(* CODESYS project AnimalCT.project
   Title: AnimalCT
   CompiledLibraryCompatibilityVersion: LeadSysStudio V3.5 SP15 Patch 4

Project tree, tasks and I/O mapping:
  Device : MC508, Leadshine Technology Co., Ltd., order no. 508101, version 3.5.15.40
      settings: RetainMode = 0; RetainStartAddr = 20480; RetainEndAddr = 524288; RetainSize = 524288
    application Application
      libraries: Standard, * (System); CAA CiA 405, 3.5.15.0 (CAA Technical Workgroup); CAA SerialCom, 3.5.15.0 (CAA Technical Workgroup); Serial Communication, 3.5.7.0 (3S - Smart Software Solutions GmbH); LS_SysLib, 1.0.0.9 (Leadshine Technology Co.Ltd); CANopenLib, 1.0.0.5 (Leadshine Technology Co.Ltd); CAA Net Base Services, 3.5.15.0 (CAA Technical Workgroup); Network, 3.5.7.0 (3S - Smart Software Solutions GmbH); CANbus, 3.5.7.0 (3S - Smart Software Solutions GmbH); VisuDialogs, * (System); LS_OmronUtils, 1.0.0.2 (Leadshine Technology Co.Ltd); CAN Low Level Communication, 1.0.0.0 (Leadshine Technology Co.Ltd); CAN API, 1.0.0.0 (Leadshine Technology Co.Ltd); CANopenLib, 1.0.0.5 (Leadshine Technology Co.Ltd)
      task Task_Trigger (cyclic, interval 2 ms, priority 1) calls Trigger_HaoboPannel, Entity_IO
      task MainTask (cyclic, interval 5 ms, priority 1) calls PLC_PRG
      task CanOpen (cyclic, interval 2 ms, priority 1) calls Axis_QJ, Axis_XZ
      DTU/
        Axis/
          data type AxisState
          data type AxisCmd
          data type AxisParameter
        TCP/
          data type PLC_SEND
          data type PLC_RECV
          data type Real_TO_Byte_Convert
        data type E_LampCmd
      GVL/
        global variables GVL_SCAN
        global variables GVL_State
      BasicFBs/
        function block Blink [ST]
        function block ASCII_Chart_N [ST]
        function block RC [ST]
        function block Curve_Cs [ST]
        function block ASCII_Chart_P [ST]
        function block MeanValue [ST]
        function block Cut [ST]
        function block String2Byte [ST]
      Refer/
        program POU_CANopen [ST]: A01_MC_AxisConfi, A04_MC_MoveRelative, A02_MC_Power, A09_ODPara, A03_MC_MoveAbsolute, A06_MC_Home, A10_MC_JOG, A11_MC_ReadStatus_CAN, A08_MC_Reset, A07_MC_Stop, A05_MC_MoveVelocity
      trace Trace (task MainTask): Entity_IO.bTriggerOut, Entity_IO.bTriggerHaobo, Entity_IO.bXaryOne, WorkStation_TCP.PLC_RECV1.m_nSocketType
      global variables PersistentVars
      Init/
        program InitMotor [ST]
      visualisation Motor
      program PLC_PRG [SFC]: _a_SelfCheck_active, _a_MoveXZ_entry, _a_QuickScan_exit, T_JUMP_IDLE, _a_ScoutDR_active, _a_Idle_exit, T_DR, _AutoDR_exit, _a_Idle_entry, _a_SelfCheck_exit, _a_Error_entry, T_QuickScan, _AutoDR_active, _a_QuickScan_entry, _a_Error_active, T_AutoDR, _a_CBCTScan_exit, _a_CBCTScan_active, _a_Homing_active, T_MoveXZ, _a_SelfCheck_entry, _a_MoveXZ_exit, T_CBCT, _a_Emergercy_entry, _AutoDR_entry_0, _a_ScoutScan_entry, _a_ScoutScan_exit, _a_ShutDown_entry, _a_Idle_active, _a_Error_exit, _a_ShutDown_active, _a_Homing_entry, _a_CBCTScan_entry, _a_QuickScan_active, _a_Debug_entry, _a_Init_active, _a_ScoutScan_active, _a_Logic_active, _a_MoveXZ_active, _a_SystemInfo_active, _a_Debug_active, _a_ScoutDR_exit, _a_Homing_exit, _a_ScoutDR_entry, T_Scout, _a_Emergercy_active
      Logic/
        program Trigger_HaoboPannel [ST]
        program WorkMode [ST]
        program Trigger_YrayPannel [ST]
      Motor/
        program Axis_XZ [ST]
        program Axis_QJ [ST]
        program Motor_SJ [ST]
      visualisation Entity_IO
      Communication/
        program CTBOX_RS232 [ST]
        program WorkStation_TCP [ST]: APLC_RECV, APLC_SENG
        program XRAY_RS485 [ST]: AXray
      IOs/
        program Entity_IO [ST]
    Resource Usage
    Device Diagnose
    Network Configuration
      LocalBus Config
    CANbus : CANbus, 3S - Smart Software Solutions GmbH, order no. 
      , version 3.5.15.0
        settings: Baudrate = 1000 kbit/s
      CANopen_Manager : CANopen_Manager, 3S - Smart Software Solutions GmbH, version 3.5.15.0
          settings: Manager is Sync consumer = True; ConfigVersion = 50659584
        ASDA_A3_Drive_QJ : ASDA-A3 Drive, Delta Electronics,INC., order no. 0, version Revision=16#02000001, FileVersion=1.1
            settings: NODEIDSAVED = 2; SDO Timeout = 1000000; PDO_Autoconfig = FALSE; EXPERTSETTINGS = False; Sync-General Parameters.Sync-COBID = 16#00000080; Emergency-General Parameters.Emergency COBID = 16#00000082; PDO 16#1400.COBID = 16#00000202; Process by CANopenManager = TRUE; PDO 16#1401.COBID = 16#00000302; Process by CANopenManager = TRUE; PDO 16#1402.COBID = 16#00000402; Process by CANopenManager = TRUE; PDO 16#1403.COBID = 16#00000502; Process by CANopenManager = TRUE; PDO 16#1800.COBID = 16#00000182; PDO 16#1800.Inhibit Time = 20; Process by CANopenManager = TRUE; PDO 16#1801.COBID = 16#00000282; PDO 16#1801.Inhibit Time = 20; Process by CANopenManager = TRUE; PDO 16#1802.COBID = 16#00000382; PDO 16#1802.Inhibit Time = 100; Process by CANopenManager = TRUE; PDO 16#1803.COBID = 16#00000482; PDO 16#1803.Inhibit Time = 100; Process by CANopenManager = TRUE; Heartbeat-Consuming1.Heartbeat-Time = 300 ms; Controlword.Index = 16#6040; Controlword.Subindex = 16#00; Controlword.ObjectLength = 16; Target Position.Index = 16#607A; Target Position.Subindex = 16#00; Target Position.ObjectLength = 32; Modes of operation.Index = 16#6060; Modes of operation.Subindex = 16#00; Modes of operation.ObjectLength = 8; Profile velocity.Index = 16#6081; Profile velocity.Subindex = 16#00; Profile velocity.ObjectLength = 32; Profile acceleration.Index = 16#6083;
              Profile acceleration.Subindex = 16#00; Profile acceleration.ObjectLength = 32; Target velocity.Index = 16#60FF; Target velocity.Subindex = 16#00; Target velocity.ObjectLength = 32; Profile deceleration.Index = 16#6084; Profile deceleration.Subindex = 16#00; Profile deceleration.ObjectLength = 32; Statusword.Index = 16#6041; Statusword.Subindex = 16#00; Statusword.ObjectLength = 16; Modes of operation display.Index = 16#6061; Modes of operation display.Subindex = 16#00; Modes of operation display.ObjectLength = 8; Position actual value.Index = 16#6064; Position actual value.Subindex = 16#00; Position actual value.ObjectLength = 32; Velocity actual value.Index = 16#606C; Velocity actual value.Subindex = 16#00; Velocity actual value.ObjectLength = 32; Digital inputs.Index = 16#60FD; Digital inputs.Subindex = 16#00; Digital inputs.ObjectLength = 32; SDO List.Set communication cycle period.Index = 16#1006; SDO List.Set communication cycle period.Subindex = 16#00; SDO List.Set communication cycle period.Value = 16#000003E8; SDO List.Set communication cycle period.Size = 32; SDO List.Set communication cycle period.AbortIfError = FALSE; SDO List.Set communication cycle period.JumpToLine = FALSE; SDO List.Set communication cycle period.Line = 0; SDO List.Set Guardtime.Index = 16#100C; SDO List.Set Guardtime.Subindex = 16#00; SDO List.Set Guardtime.Value = 16#00000000; SDO List.Set Guardtime.Size = 16; SDO List.Set Guardtime.AbortIfError = FALSE; SDO List.Set Guardtime.JumpToLine = FALSE; SDO List.Set Guardtime.Line = 0; SDO List.Set Lifetime.Index = 16#100D; SDO List.Set Lifetime.Subindex = 16#00; SDO List.Set Lifetime.Value = 16#00000000;
              SDO List.Set Lifetime.Size = 8; SDO List.Set Lifetime.AbortIfError = FALSE; SDO List.Set Lifetime.JumpToLine = FALSE; SDO List.Set Lifetime.Line = 0; SDO List.Set Heartbeat Consumer.Index = 16#1016; SDO List.Set Heartbeat Consumer.Subindex = 16#01; SDO List.Set Heartbeat Consumer.Value = 16#007F012C; SDO List.Set Heartbeat Consumer.Size = 32; SDO List.Set Heartbeat Consumer.AbortIfError = FALSE; SDO List.Set Heartbeat Consumer.JumpToLine = FALSE; SDO List.Set Heartbeat Consumer.Line = 0; SDO List.Set Heartbeat Producer.Index = 16#1017; SDO List.Set Heartbeat Producer.Subindex = 16#00; SDO List.Set Heartbeat Producer.Value = 16#000000C8; SDO List.Set Heartbeat Producer.Size = 16; SDO List.Set Heartbeat Producer.AbortIfError = FALSE; SDO List.Set Heartbeat Producer.JumpToLine = FALSE; SDO List.Set Heartbeat Producer.Line = 0; SDO List.Disable PDO.Index = 16#1400; SDO List.Disable PDO.Subindex = 16#01; SDO List.Disable PDO.Value = 16#80000202; SDO List.Disable PDO.Size = 32; SDO List.Disable PDO.AbortIfError = FALSE; SDO List.Disable PDO.JumpToLine = FALSE; SDO List.Disable PDO.Line = 0; SDO List.Set transmission type.Index = 16#1400; SDO List.Set transmission type.Subindex = 16#02; SDO List.Set transmission type.Value = 16#FF; SDO List.Set transmission type.Size = 8; SDO List.Set transmission type.AbortIfError = FALSE; SDO List.Set transmission type.JumpToLine = FALSE; SDO List.Set transmission type.Line = 0; SDO List.Clear pdo mapping.Index = 16#1600; SDO List.Clear pdo mapping.Subindex = 16#00; SDO List.Clear pdo mapping.Value = 16#0; SDO List.Clear pdo mapping.Size = 8; SDO List.Clear pdo mapping.AbortIfError = FALSE; SDO List.Clear pdo mapping.JumpToLine = FALSE; SDO List.Clear pdo mapping.Line = 0; SDO List.Set Mapping.Index = 16#1600;
              SDO List.Set Mapping.Subindex = 16#01; SDO List.Set Mapping.Value = 16#60400010; SDO List.Set Mapping.Size = 32; SDO List.Set Mapping.AbortIfError = FALSE; SDO List.Set Mapping.JumpToLine = FALSE; SDO List.Set Mapping.Line = 0; SDO List.Set Mapping.Index = 16#1600; SDO List.Set Mapping.Subindex = 16#02; SDO List.Set Mapping.Value = 16#607A0020; SDO List.Set Mapping.Size = 32; SDO List.Set Mapping.AbortIfError = FALSE; SDO List.Set Mapping.JumpToLine = FALSE; SDO List.Set Mapping.Line = 0; SDO List.Set Mapping.Index = 16#1600; SDO List.Set Mapping.Subindex = 16#03; SDO List.Set Mapping.Value = 16#60600008; SDO List.Set Mapping.Size = 32; SDO List.Set Mapping.AbortIfError = FALSE; SDO List.Set Mapping.JumpToLine = FALSE; SDO List.Set Mapping.Line = 0; SDO List.Set number of mappings.Index = 16#1600; SDO List.Set number of mappings.Subindex = 16#00; SDO List.Set number of mappings.Value = 16#03; SDO List.Set number of mappings.Size = 8; SDO List.Set number of mappings.AbortIfError = FALSE; SDO List.Set number of mappings.JumpToLine = FALSE; SDO List.Set number of mappings.Line = 0; SDO List.Set and enable COB-ID.Index = 16#1400; SDO List.Set and enable COB-ID.Subindex = 16#01; SDO List.Set and enable COB-ID.Value = 16#00000202; SDO List.Set and enable COB-ID.Size = 32; SDO List.Set and enable COB-ID.AbortIfError = FALSE; SDO List.Set and enable COB-ID.JumpToLine = FALSE; SDO List.Set and enable COB-ID.Line = 0; SDO List.Set transmission type.Index = 16#1401; SDO List.Set transmission type.Subindex = 16#02; SDO List.Set transmission type.Value = 16#FF; SDO List.Set transmission type.Size = 8; SDO List.Set transmission type.AbortIfError = FALSE; SDO List.Set transmission type.JumpToLine = FALSE;
              SDO List.Set transmission type.Line = 0; SDO List.Clear pdo mapping.Index = 16#1601; SDO List.Clear pdo mapping.Subindex = 16#00; SDO List.Clear pdo mapping.Value = 16#0; SDO List.Clear pdo mapping.Size = 8; SDO List.Clear pdo mapping.AbortIfError = FALSE; SDO List.Clear pdo mapping.JumpToLine = FALSE; SDO List.Clear pdo mapping.Line = 0; SDO List.Set Mapping.Index = 16#1601; SDO List.Set Mapping.Subindex = 16#01; SDO List.Set Mapping.Value = 16#60810020; SDO List.Set Mapping.Size = 32; SDO List.Set Mapping.AbortIfError = FALSE; SDO List.Set Mapping.JumpToLine = FALSE; SDO List.Set Mapping.Line = 0; SDO List.Set Mapping.Index = 16#1601; SDO List.Set Mapping.Subindex = 16#02; SDO List.Set Mapping.Value = 16#60830020; SDO List.Set Mapping.Size = 32; SDO List.Set Mapping.AbortIfError = FALSE; SDO List.Set Mapping.JumpToLine = FALSE; SDO List.Set Mapping.Line = 0; SDO List.Set number of mappings.Index = 16#1601; SDO List.Set number of mappings.Subindex = 16#00; SDO List.Set number of mappings.Value = 16#02; SDO List.Set number of mappings.Size = 8; SDO List.Set number of mappings.AbortIfError = FALSE; SDO List.Set number of mappings.JumpToLine = FALSE; SDO List.Set number of mappings.Line = 0; SDO List.Set and enable COB-ID.Index = 16#1401; SDO List.Set and enable COB-ID.Subindex = 16#01; SDO List.Set and enable COB-ID.Value = 16#00000302; SDO List.Set and enable COB-ID.Size = 32; SDO List.Set and enable COB-ID.AbortIfError = FALSE; SDO List.Set and enable COB-ID.JumpToLine = FALSE; SDO List.Set and enable COB-ID.Line = 0; SDO List.Set transmission type.Index = 16#1402; SDO List.Set transmission type.Subindex = 16#02; SDO List.Set transmission type.Value = 16#FF; SDO List.Set transmission type.Size = 8;
              SDO List.Set transmission type.AbortIfError = FALSE; SDO List.Set transmission type.JumpToLine = FALSE; SDO List.Set transmission type.Line = 0; SDO List.Clear pdo mapping.Index = 16#1602; SDO List.Clear pdo mapping.Subindex = 16#00; SDO List.Clear pdo mapping.Value = 16#0; SDO List.Clear pdo mapping.Size = 8; SDO List.Clear pdo mapping.AbortIfError = FALSE; SDO List.Clear pdo mapping.JumpToLine = FALSE; SDO List.Clear pdo mapping.Line = 0; SDO List.Set Mapping.Index = 16#1602; SDO List.Set Mapping.Subindex = 16#01; SDO List.Set Mapping.Value = 16#60FF0020; SDO List.Set Mapping.Size = 32; SDO List.Set Mapping.AbortIfError = FALSE; SDO List.Set Mapping.JumpToLine = FALSE; SDO List.Set Mapping.Line = 0; SDO List.Set number of mappings.Index = 16#1602; SDO List.Set number of mappings.Subindex = 16#00; SDO List.Set number of mappings.Value = 16#01; SDO List.Set number of mappings.Size = 8; SDO List.Set number of mappings.AbortIfError = FALSE; SDO List.Set number of mappings.JumpToLine = FALSE; SDO List.Set number of mappings.Line = 0; SDO List.Set and enable COB-ID.Index = 16#1402; SDO List.Set and enable COB-ID.Subindex = 16#01; SDO List.Set and enable COB-ID.Value = 16#00000402; SDO List.Set and enable COB-ID.Size = 32; SDO List.Set and enable COB-ID.AbortIfError = FALSE; SDO List.Set and enable COB-ID.JumpToLine = FALSE; SDO List.Set and enable COB-ID.Line = 0; SDO List.Set transmission type.Index = 16#1403; SDO List.Set transmission type.Subindex = 16#02; SDO List.Set transmission type.Value = 16#FF; SDO List.Set transmission type.Size = 8; SDO List.Set transmission type.AbortIfError = FALSE; SDO List.Set transmission type.JumpToLine = FALSE; SDO List.Set transmission type.Line = 0; SDO List.Clear pdo mapping.Index = 16#1603; SDO List.Clear pdo mapping.Subindex = 16#00;
              SDO List.Clear pdo mapping.Value = 16#0; SDO List.Clear pdo mapping.Size = 8; SDO List.Clear pdo mapping.AbortIfError = FALSE; SDO List.Clear pdo mapping.JumpToLine = FALSE; SDO List.Clear pdo mapping.Line = 0; SDO List.Set Mapping.Index = 16#1603; SDO List.Set Mapping.Subindex = 16#01; SDO List.Set Mapping.Value = 16#60840020; SDO List.Set Mapping.Size = 32; SDO List.Set Mapping.AbortIfError = FALSE; SDO List.Set Mapping.JumpToLine = FALSE; SDO List.Set Mapping.Line = 0; SDO List.Set number of mappings.Index = 16#1603; SDO List.Set number of mappings.Subindex = 16#00; SDO List.Set number of mappings.Value = 16#01; SDO List.Set number of mappings.Size = 8; SDO List.Set number of mappings.AbortIfError = FALSE; SDO List.Set number of mappings.JumpToLine = FALSE; SDO List.Set number of mappings.Line = 0; SDO List.Set and enable COB-ID.Index = 16#1403; SDO List.Set and enable COB-ID.Subindex = 16#01; SDO List.Set and enable COB-ID.Value = 16#00000502; SDO List.Set and enable COB-ID.Size = 32; SDO List.Set and enable COB-ID.AbortIfError = FALSE; SDO List.Set and enable COB-ID.JumpToLine = FALSE; SDO List.Set and enable COB-ID.Line = 0; SDO List.Disable PDO.Index = 16#1800; SDO List.Disable PDO.Subindex = 16#01; SDO List.Disable PDO.Value = 16#80000182; SDO List.Disable PDO.Size = 32; SDO List.Disable PDO.AbortIfError = FALSE; SDO List.Disable PDO.JumpToLine = FALSE; SDO List.Disable PDO.Line = 0; SDO List.Set transmission type.Index = 16#1800; SDO List.Set transmission type.Subindex = 16#02; SDO List.Set transmission type.Value = 16#FF; SDO List.Set transmission type.Size = 8; SDO List.Set transmission type.AbortIfError = FALSE; SDO List.Set transmission type.JumpToLine = FALSE; SDO List.Set transmission type.Line = 0;
              SDO List.Set inhibit time.Index = 16#1800; SDO List.Set inhibit time.Subindex = 16#03; SDO List.Set inhibit time.Value = 16#0014; SDO List.Set inhibit time.Size = 16; SDO List.Set inhibit time.AbortIfError = FALSE; SDO List.Set inhibit time.JumpToLine = FALSE; SDO List.Set inhibit time.Line = 0; SDO List.Set event time.Index = 16#1800; SDO List.Set event time.Subindex = 16#05; SDO List.Set event time.Value = 16#0000; SDO List.Set event time.Size = 16; SDO List.Set event time.AbortIfError = FALSE; SDO List.Set event time.JumpToLine = FALSE; SDO List.Set event time.Line = 0; SDO List.Clear pdo mapping.Index = 16#1A00; SDO List.Clear pdo mapping.Subindex = 16#00; SDO List.Clear pdo mapping.Value = 16#0; SDO List.Clear pdo mapping.Size = 8; SDO List.Clear pdo mapping.AbortIfError = FALSE; SDO List.Clear pdo mapping.JumpToLine = FALSE; SDO List.Clear pdo mapping.Line = 0; SDO List.Set Mapping.Index = 16#1A00; SDO List.Set Mapping.Subindex = 16#01; SDO List.Set Mapping.Value = 16#60410010; SDO List.Set Mapping.Size = 32; SDO List.Set Mapping.AbortIfError = FALSE; SDO List.Set Mapping.JumpToLine = FALSE; SDO List.Set Mapping.Line = 0; SDO List.Set number of mappings.Index = 16#1A00; SDO List.Set number of mappings.Subindex = 16#00; SDO List.Set number of mappings.Value = 16#01; SDO List.Set number of mappings.Size = 8; SDO List.Set number of mappings.AbortIfError = FALSE; SDO List.Set number of mappings.JumpToLine = FALSE; SDO List.Set number of mappings.Line = 0; SDO List.Set and enable COB-ID.Index = 16#1800; SDO List.Set and enable COB-ID.Subindex = 16#01; SDO List.Set and enable COB-ID.Value = 16#00000182; SDO List.Set and enable COB-ID.Size = 32; SDO List.Set and enable COB-ID.AbortIfError = FALSE;
              SDO List.Set and enable COB-ID.JumpToLine = FALSE; SDO List.Set and enable COB-ID.Line = 0; SDO List.Set transmission type.Index = 16#1801; SDO List.Set transmission type.Subindex = 16#02; SDO List.Set transmission type.Value = 16#FF; SDO List.Set transmission type.Size = 8; SDO List.Set transmission type.AbortIfError = FALSE; SDO List.Set transmission type.JumpToLine = FALSE; SDO List.Set transmission type.Line = 0; SDO List.Set inhibit time.Index = 16#1801; SDO List.Set inhibit time.Subindex = 16#03; SDO List.Set inhibit time.Value = 16#0014; SDO List.Set inhibit time.Size = 16; SDO List.Set inhibit time.AbortIfError = FALSE; SDO List.Set inhibit time.JumpToLine = FALSE; SDO List.Set inhibit time.Line = 0; SDO List.Set event time.Index = 16#1801; SDO List.Set event time.Subindex = 16#05; SDO List.Set event time.Value = 16#0000; SDO List.Set event time.Size = 16; SDO List.Set event time.AbortIfError = FALSE; SDO List.Set event time.JumpToLine = FALSE; SDO List.Set event time.Line = 0; SDO List.Clear pdo mapping.Index = 16#1A01; SDO List.Clear pdo mapping.Subindex = 16#00; SDO List.Clear pdo mapping.Value = 16#0; SDO List.Clear pdo mapping.Size = 8; SDO List.Clear pdo mapping.AbortIfError = FALSE; SDO List.Clear pdo mapping.JumpToLine = FALSE; SDO List.Clear pdo mapping.Line = 0; SDO List.Set Mapping.Index = 16#1A01; SDO List.Set Mapping.Subindex = 16#01; SDO List.Set Mapping.Value = 16#60610008; SDO List.Set Mapping.Size = 32; SDO List.Set Mapping.AbortIfError = FALSE; SDO List.Set Mapping.JumpToLine = FALSE; SDO List.Set Mapping.Line = 0; SDO List.Set number of mappings.Index = 16#1A01; SDO List.Set number of mappings.Subindex = 16#00; SDO List.Set number of mappings.Value = 16#01;
              SDO List.Set number of mappings.Size = 8; SDO List.Set number of mappings.AbortIfError = FALSE; SDO List.Set number of mappings.JumpToLine = FALSE; SDO List.Set number of mappings.Line = 0; SDO List.Set and enable COB-ID.Index = 16#1801; SDO List.Set and enable COB-ID.Subindex = 16#01; SDO List.Set and enable COB-ID.Value = 16#00000282; SDO List.Set and enable COB-ID.Size = 32; SDO List.Set and enable COB-ID.AbortIfError = FALSE; SDO List.Set and enable COB-ID.JumpToLine = FALSE; SDO List.Set and enable COB-ID.Line = 0; SDO List.Set transmission type.Index = 16#1802; SDO List.Set transmission type.Subindex = 16#02; SDO List.Set transmission type.Value = 16#FF; SDO List.Set transmission type.Size = 8; SDO List.Set transmission type.AbortIfError = FALSE; SDO List.Set transmission type.JumpToLine = FALSE; SDO List.Set transmission type.Line = 0; SDO List.Set inhibit time.Index = 16#1802; SDO List.Set inhibit time.Subindex = 16#03; SDO List.Set inhibit time.Value = 16#0064; SDO List.Set inhibit time.Size = 16; SDO List.Set inhibit time.AbortIfError = FALSE; SDO List.Set inhibit time.JumpToLine = FALSE; SDO List.Set inhibit time.Line = 0; SDO List.Set event time.Index = 16#1802; SDO List.Set event time.Subindex = 16#05; SDO List.Set event time.Value = 16#0000; SDO List.Set event time.Size = 16; SDO List.Set event time.AbortIfError = FALSE; SDO List.Set event time.JumpToLine = FALSE; SDO List.Set event time.Line = 0; SDO List.Clear pdo mapping.Index = 16#1A02; SDO List.Clear pdo mapping.Subindex = 16#00; SDO List.Clear pdo mapping.Value = 16#0; SDO List.Clear pdo mapping.Size = 8; SDO List.Clear pdo mapping.AbortIfError = FALSE; SDO List.Clear pdo mapping.JumpToLine = FALSE; SDO List.Clear pdo mapping.Line = 0; SDO List.Set Mapping.Index = 16#1A02;
              SDO List.Set Mapping.Subindex = 16#01; SDO List.Set Mapping.Value = 16#60640020; SDO List.Set Mapping.Size = 32; SDO List.Set Mapping.AbortIfError = FALSE; SDO List.Set Mapping.JumpToLine = FALSE; SDO List.Set Mapping.Line = 0; SDO List.Set Mapping.Index = 16#1A02; SDO List.Set Mapping.Subindex = 16#02; SDO List.Set Mapping.Value = 16#606C0020; SDO List.Set Mapping.Size = 32; SDO List.Set Mapping.AbortIfError = FALSE; SDO List.Set Mapping.JumpToLine = FALSE; SDO List.Set Mapping.Line = 0; SDO List.Set number of mappings.Index = 16#1A02; SDO List.Set number of mappings.Subindex = 16#00; SDO List.Set number of mappings.Value = 16#02; SDO List.Set number of mappings.Size = 8; SDO List.Set number of mappings.AbortIfError = FALSE; SDO List.Set number of mappings.JumpToLine = FALSE; SDO List.Set number of mappings.Line = 0; SDO List.Set and enable COB-ID.Index = 16#1802; SDO List.Set and enable COB-ID.Subindex = 16#01; SDO List.Set and enable COB-ID.Value = 16#00000382; SDO List.Set and enable COB-ID.Size = 32; SDO List.Set and enable COB-ID.AbortIfError = FALSE; SDO List.Set and enable COB-ID.JumpToLine = FALSE; SDO List.Set and enable COB-ID.Line = 0; SDO List.Set transmission type.Index = 16#1803; SDO List.Set transmission type.Subindex = 16#02; SDO List.Set transmission type.Value = 16#FF; SDO List.Set transmission type.Size = 8; SDO List.Set transmission type.AbortIfError = FALSE; SDO List.Set transmission type.JumpToLine = FALSE; SDO List.Set transmission type.Line = 0; SDO List.Set inhibit time.Index = 16#1803; SDO List.Set inhibit time.Subindex = 16#03; SDO List.Set inhibit time.Value = 16#0064; SDO List.Set inhibit time.Size = 16; SDO List.Set inhibit time.AbortIfError = FALSE; SDO List.Set inhibit time.JumpToLine = FALSE;
              SDO List.Set inhibit time.Line = 0; SDO List.Set event time.Index = 16#1803; SDO List.Set event time.Subindex = 16#05; SDO List.Set event time.Value = 16#0000; SDO List.Set event time.Size = 16; SDO List.Set event time.AbortIfError = FALSE; SDO List.Set event time.JumpToLine = FALSE; SDO List.Set event time.Line = 0; SDO List.Clear pdo mapping.Index = 16#1A03; SDO List.Clear pdo mapping.Subindex = 16#00; SDO List.Clear pdo mapping.Value = 16#0; SDO List.Clear pdo mapping.Size = 8; SDO List.Clear pdo mapping.AbortIfError = FALSE; SDO List.Clear pdo mapping.JumpToLine = FALSE; SDO List.Clear pdo mapping.Line = 0; SDO List.Set Mapping.Index = 16#1A03; SDO List.Set Mapping.Subindex = 16#01; SDO List.Set Mapping.Value = 16#60FD0020; SDO List.Set Mapping.Size = 32; SDO List.Set Mapping.AbortIfError = FALSE; SDO List.Set Mapping.JumpToLine = FALSE; SDO List.Set Mapping.Line = 0; SDO List.Set number of mappings.Index = 16#1A03; SDO List.Set number of mappings.Subindex = 16#00; SDO List.Set number of mappings.Value = 16#01; SDO List.Set number of mappings.Size = 8; SDO List.Set number of mappings.AbortIfError = FALSE; SDO List.Set number of mappings.JumpToLine = FALSE; SDO List.Set number of mappings.Line = 0; SDO List.Set and enable COB-ID.Index = 16#1803; SDO List.Set and enable COB-ID.Subindex = 16#01; SDO List.Set and enable COB-ID.Value = 16#00000482; SDO List.Set and enable COB-ID.Size = 32; SDO List.Set and enable COB-ID.AbortIfError = FALSE; SDO List.Set and enable COB-ID.JumpToLine = FALSE; SDO List.Set and enable COB-ID.Line = 0; SDO List.Homing method.Index = 16#6098; SDO List.Homing method.Subindex = 16#00; SDO List.Homing method.Value = 16#0000000D; SDO List.Homing method.Size = 8;
              SDO List.Homing method.AbortIfError = FALSE; SDO List.Homing method.JumpToLine = FALSE; SDO List.Homing method.Line = 0; SDO List.Speed during search for switch.Index = 16#6099; SDO List.Speed during search for switch.Subindex = 16#01; SDO List.Speed during search for switch.Value = 5000; SDO List.Speed during search for switch.Size = 32; SDO List.Speed during search for switch.AbortIfError = FALSE; SDO List.Speed during search for switch.JumpToLine = FALSE; SDO List.Speed during search for switch.Line = 0; SDO List.Speed during search for zero.Index = 16#6099; SDO List.Speed during search for zero.Subindex = 16#02; SDO List.Speed during search for zero.Value = 800; SDO List.Speed during search for zero.Size = 32; SDO List.Speed during search for zero.AbortIfError = FALSE; SDO List.Speed during search for zero.JumpToLine = FALSE; SDO List.Speed during search for zero.Line = 0; ConfigVersion = 50659584
            input  QJ_ActPos : DINT  // Position actual value
            input  QJ_ActVel : DINT  // Velocity actual value
            input  bForeMotorMin1 : BOOL  // Digital inputs.Bit0
            input  bForeMotorMax1 : BOOL  // Digital inputs.Bit1
            unmapped channels: Controlword, Target Position, Modes of operation, Profile velocity, Profile acceleration, Target velocity, Profile deceleration, Statusword, Modes of operation display, Digital inputs
        ASDA_A3_Drive_XZ : ASDA-A3 Drive, Delta Electronics,INC., order no. 0, version Revision=16#02000001, FileVersion=1.1
            settings: NODEIDSAVED = 1; SDO Timeout = 1000000; PDO_Autoconfig = FALSE; EXPERTSETTINGS = False; Sync-General Parameters.Sync-COBID = 16#00000080; Sync-General Parameters.Communication Cycle Period = 1000 usec; PDO 16#1400.COBID = 16#00000201; Process by CANopenManager = TRUE; PDO 16#1401.COBID = 16#00000301; Process by CANopenManager = TRUE; PDO 16#1402.COBID = 16#00000401; Process by CANopenManager = TRUE; PDO 16#1403.COBID = 16#00000501; Process by CANopenManager = TRUE; PDO 16#1800.COBID = 16#00000181; PDO 16#1800.Inhibit Time = 20; Process by CANopenManager = TRUE; PDO 16#1801.COBID = 16#00000281; PDO 16#1801.Inhibit Time = 20; Process by CANopenManager = TRUE; PDO 16#1802.COBID = 16#00000381; PDO 16#1802.Inhibit Time = 100; Process by CANopenManager = TRUE; PDO 16#1803.COBID = 16#00000481; PDO 16#1803.Inhibit Time = 100; Process by CANopenManager = TRUE; Heartbeat-Consuming1.Heartbeat-Time = 300 ms; Controlword.Index = 16#6040; Controlword.Subindex = 16#00; Controlword.ObjectLength = 16; Target Position.Index = 16#607A; Target Position.Subindex = 16#00; Target Position.ObjectLength = 32; Modes of operation.Index = 16#6060; Modes of operation.Subindex = 16#00; Modes of operation.ObjectLength = 8; Profile velocity.Index = 16#6081; Profile velocity.Subindex = 16#00; Profile velocity.ObjectLength = 32; Profile acceleration.Index = 16#6083;
              Profile acceleration.Subindex = 16#00; Profile acceleration.ObjectLength = 32; Target velocity.Index = 16#60FF; Target velocity.Subindex = 16#00; Target velocity.ObjectLength = 32; Profile deceleration.Index = 16#6084; Profile deceleration.Subindex = 16#00; Profile deceleration.ObjectLength = 32; Statusword.Index = 16#6041; Statusword.Subindex = 16#00; Statusword.ObjectLength = 16; Modes of operation display.Index = 16#6061; Modes of operation display.Subindex = 16#00; Modes of operation display.ObjectLength = 8; Position actual value.Index = 16#6064; Position actual value.Subindex = 16#00; Position actual value.ObjectLength = 32; Velocity actual value.Index = 16#606C; Velocity actual value.Subindex = 16#00; Velocity actual value.ObjectLength = 32; Digital inputs.Index = 16#60FD; Digital inputs.Subindex = 16#00; Digital inputs.ObjectLength = 32; SDO List.Set communication cycle period.Index = 16#1006; SDO List.Set communication cycle period.Subindex = 16#00; SDO List.Set communication cycle period.Value = 16#000003E8; SDO List.Set communication cycle period.Size = 32; SDO List.Set communication cycle period.AbortIfError = FALSE; SDO List.Set communication cycle period.JumpToLine = FALSE; SDO List.Set communication cycle period.Line = 0; SDO List.Set Guardtime.Index = 16#100C; SDO List.Set Guardtime.Subindex = 16#00; SDO List.Set Guardtime.Value = 16#00000000; SDO List.Set Guardtime.Size = 16; SDO List.Set Guardtime.AbortIfError = FALSE; SDO List.Set Guardtime.JumpToLine = FALSE; SDO List.Set Guardtime.Line = 0; SDO List.Set Lifetime.Index = 16#100D; SDO List.Set Lifetime.Subindex = 16#00; SDO List.Set Lifetime.Value = 16#00000000;
              SDO List.Set Lifetime.Size = 8; SDO List.Set Lifetime.AbortIfError = FALSE; SDO List.Set Lifetime.JumpToLine = FALSE; SDO List.Set Lifetime.Line = 0; SDO List.Set Heartbeat Consumer.Index = 16#1016; SDO List.Set Heartbeat Consumer.Subindex = 16#01; SDO List.Set Heartbeat Consumer.Value = 16#007F012C; SDO List.Set Heartbeat Consumer.Size = 32; SDO List.Set Heartbeat Consumer.AbortIfError = FALSE; SDO List.Set Heartbeat Consumer.JumpToLine = FALSE; SDO List.Set Heartbeat Consumer.Line = 0; SDO List.Set Heartbeat Producer.Index = 16#1017; SDO List.Set Heartbeat Producer.Subindex = 16#00; SDO List.Set Heartbeat Producer.Value = 16#000000C8; SDO List.Set Heartbeat Producer.Size = 16; SDO List.Set Heartbeat Producer.AbortIfError = FALSE; SDO List.Set Heartbeat Producer.JumpToLine = FALSE; SDO List.Set Heartbeat Producer.Line = 0; SDO List.Disable PDO.Index = 16#1400; SDO List.Disable PDO.Subindex = 16#01; SDO List.Disable PDO.Value = 16#80000201; SDO List.Disable PDO.Size = 32; SDO List.Disable PDO.AbortIfError = FALSE; SDO List.Disable PDO.JumpToLine = FALSE; SDO List.Disable PDO.Line = 0; SDO List.Set transmission type.Index = 16#1400; SDO List.Set transmission type.Subindex = 16#02; SDO List.Set transmission type.Value = 16#FF; SDO List.Set transmission type.Size = 8; SDO List.Set transmission type.AbortIfError = FALSE; SDO List.Set transmission type.JumpToLine = FALSE; SDO List.Set transmission type.Line = 0; SDO List.Clear pdo mapping.Index = 16#1600; SDO List.Clear pdo mapping.Subindex = 16#00; SDO List.Clear pdo mapping.Value = 16#0; SDO List.Clear pdo mapping.Size = 8; SDO List.Clear pdo mapping.AbortIfError = FALSE; SDO List.Clear pdo mapping.JumpToLine = FALSE; SDO List.Clear pdo mapping.Line = 0; SDO List.Set Mapping.Index = 16#1600;
              SDO List.Set Mapping.Subindex = 16#01; SDO List.Set Mapping.Value = 16#60400010; SDO List.Set Mapping.Size = 32; SDO List.Set Mapping.AbortIfError = FALSE; SDO List.Set Mapping.JumpToLine = FALSE; SDO List.Set Mapping.Line = 0; SDO List.Set Mapping.Index = 16#1600; SDO List.Set Mapping.Subindex = 16#02; SDO List.Set Mapping.Value = 16#607A0020; SDO List.Set Mapping.Size = 32; SDO List.Set Mapping.AbortIfError = FALSE; SDO List.Set Mapping.JumpToLine = FALSE; SDO List.Set Mapping.Line = 0; SDO List.Set Mapping.Index = 16#1600; SDO List.Set Mapping.Subindex = 16#03; SDO List.Set Mapping.Value = 16#60600008; SDO List.Set Mapping.Size = 32; SDO List.Set Mapping.AbortIfError = FALSE; SDO List.Set Mapping.JumpToLine = FALSE; SDO List.Set Mapping.Line = 0; SDO List.Set number of mappings.Index = 16#1600; SDO List.Set number of mappings.Subindex = 16#00; SDO List.Set number of mappings.Value = 16#03; SDO List.Set number of mappings.Size = 8; SDO List.Set number of mappings.AbortIfError = FALSE; SDO List.Set number of mappings.JumpToLine = FALSE; SDO List.Set number of mappings.Line = 0; SDO List.Set and enable COB-ID.Index = 16#1400; SDO List.Set and enable COB-ID.Subindex = 16#01; SDO List.Set and enable COB-ID.Value = 16#00000201; SDO List.Set and enable COB-ID.Size = 32; SDO List.Set and enable COB-ID.AbortIfError = FALSE; SDO List.Set and enable COB-ID.JumpToLine = FALSE; SDO List.Set and enable COB-ID.Line = 0; SDO List.Set transmission type.Index = 16#1401; SDO List.Set transmission type.Subindex = 16#02; SDO List.Set transmission type.Value = 16#FF; SDO List.Set transmission type.Size = 8; SDO List.Set transmission type.AbortIfError = FALSE; SDO List.Set transmission type.JumpToLine = FALSE;
              SDO List.Set transmission type.Line = 0; SDO List.Clear pdo mapping.Index = 16#1601; SDO List.Clear pdo mapping.Subindex = 16#00; SDO List.Clear pdo mapping.Value = 16#0; SDO List.Clear pdo mapping.Size = 8; SDO List.Clear pdo mapping.AbortIfError = FALSE; SDO List.Clear pdo mapping.JumpToLine = FALSE; SDO List.Clear pdo mapping.Line = 0; SDO List.Set Mapping.Index = 16#1601; SDO List.Set Mapping.Subindex = 16#01; SDO List.Set Mapping.Value = 16#60810020; SDO List.Set Mapping.Size = 32; SDO List.Set Mapping.AbortIfError = FALSE; SDO List.Set Mapping.JumpToLine = FALSE; SDO List.Set Mapping.Line = 0; SDO List.Set Mapping.Index = 16#1601; SDO List.Set Mapping.Subindex = 16#02; SDO List.Set Mapping.Value = 16#60830020; SDO List.Set Mapping.Size = 32; SDO List.Set Mapping.AbortIfError = FALSE; SDO List.Set Mapping.JumpToLine = FALSE; SDO List.Set Mapping.Line = 0; SDO List.Set number of mappings.Index = 16#1601; SDO List.Set number of mappings.Subindex = 16#00; SDO List.Set number of mappings.Value = 16#02; SDO List.Set number of mappings.Size = 8; SDO List.Set number of mappings.AbortIfError = FALSE; SDO List.Set number of mappings.JumpToLine = FALSE; SDO List.Set number of mappings.Line = 0; SDO List.Set and enable COB-ID.Index = 16#1401; SDO List.Set and enable COB-ID.Subindex = 16#01; SDO List.Set and enable COB-ID.Value = 16#00000301; SDO List.Set and enable COB-ID.Size = 32; SDO List.Set and enable COB-ID.AbortIfError = FALSE; SDO List.Set and enable COB-ID.JumpToLine = FALSE; SDO List.Set and enable COB-ID.Line = 0; SDO List.Set transmission type.Index = 16#1402; SDO List.Set transmission type.Subindex = 16#02; SDO List.Set transmission type.Value = 16#FF; SDO List.Set transmission type.Size = 8;
              SDO List.Set transmission type.AbortIfError = FALSE; SDO List.Set transmission type.JumpToLine = FALSE; SDO List.Set transmission type.Line = 0; SDO List.Clear pdo mapping.Index = 16#1602; SDO List.Clear pdo mapping.Subindex = 16#00; SDO List.Clear pdo mapping.Value = 16#0; SDO List.Clear pdo mapping.Size = 8; SDO List.Clear pdo mapping.AbortIfError = FALSE; SDO List.Clear pdo mapping.JumpToLine = FALSE; SDO List.Clear pdo mapping.Line = 0; SDO List.Set Mapping.Index = 16#1602; SDO List.Set Mapping.Subindex = 16#01; SDO List.Set Mapping.Value = 16#60FF0020; SDO List.Set Mapping.Size = 32; SDO List.Set Mapping.AbortIfError = FALSE; SDO List.Set Mapping.JumpToLine = FALSE; SDO List.Set Mapping.Line = 0; SDO List.Set number of mappings.Index = 16#1602; SDO List.Set number of mappings.Subindex = 16#00; SDO List.Set number of mappings.Value = 16#01; SDO List.Set number of mappings.Size = 8; SDO List.Set number of mappings.AbortIfError = FALSE; SDO List.Set number of mappings.JumpToLine = FALSE; SDO List.Set number of mappings.Line = 0; SDO List.Set and enable COB-ID.Index = 16#1402; SDO List.Set and enable COB-ID.Subindex = 16#01; SDO List.Set and enable COB-ID.Value = 16#00000401; SDO List.Set and enable COB-ID.Size = 32; SDO List.Set and enable COB-ID.AbortIfError = FALSE; SDO List.Set and enable COB-ID.JumpToLine = FALSE; SDO List.Set and enable COB-ID.Line = 0; SDO List.Set transmission type.Index = 16#1403; SDO List.Set transmission type.Subindex = 16#02; SDO List.Set transmission type.Value = 16#FF; SDO List.Set transmission type.Size = 8; SDO List.Set transmission type.AbortIfError = FALSE; SDO List.Set transmission type.JumpToLine = FALSE; SDO List.Set transmission type.Line = 0; SDO List.Clear pdo mapping.Index = 16#1603; SDO List.Clear pdo mapping.Subindex = 16#00;
              SDO List.Clear pdo mapping.Value = 16#0; SDO List.Clear pdo mapping.Size = 8; SDO List.Clear pdo mapping.AbortIfError = FALSE; SDO List.Clear pdo mapping.JumpToLine = FALSE; SDO List.Clear pdo mapping.Line = 0; SDO List.Set Mapping.Index = 16#1603; SDO List.Set Mapping.Subindex = 16#01; SDO List.Set Mapping.Value = 16#60840020; SDO List.Set Mapping.Size = 32; SDO List.Set Mapping.AbortIfError = FALSE; SDO List.Set Mapping.JumpToLine = FALSE; SDO List.Set Mapping.Line = 0; SDO List.Set number of mappings.Index = 16#1603; SDO List.Set number of mappings.Subindex = 16#00; SDO List.Set number of mappings.Value = 16#01; SDO List.Set number of mappings.Size = 8; SDO List.Set number of mappings.AbortIfError = FALSE; SDO List.Set number of mappings.JumpToLine = FALSE; SDO List.Set number of mappings.Line = 0; SDO List.Set and enable COB-ID.Index = 16#1403; SDO List.Set and enable COB-ID.Subindex = 16#01; SDO List.Set and enable COB-ID.Value = 16#00000501; SDO List.Set and enable COB-ID.Size = 32; SDO List.Set and enable COB-ID.AbortIfError = FALSE; SDO List.Set and enable COB-ID.JumpToLine = FALSE; SDO List.Set and enable COB-ID.Line = 0; SDO List.Disable PDO.Index = 16#1800; SDO List.Disable PDO.Subindex = 16#01; SDO List.Disable PDO.Value = 16#80000181; SDO List.Disable PDO.Size = 32; SDO List.Disable PDO.AbortIfError = FALSE; SDO List.Disable PDO.JumpToLine = FALSE; SDO List.Disable PDO.Line = 0; SDO List.Set transmission type.Index = 16#1800; SDO List.Set transmission type.Subindex = 16#02; SDO List.Set transmission type.Value = 16#FF; SDO List.Set transmission type.Size = 8; SDO List.Set transmission type.AbortIfError = FALSE; SDO List.Set transmission type.JumpToLine = FALSE; SDO List.Set transmission type.Line = 0;
              SDO List.Set inhibit time.Index = 16#1800; SDO List.Set inhibit time.Subindex = 16#03; SDO List.Set inhibit time.Value = 16#0014; SDO List.Set inhibit time.Size = 16; SDO List.Set inhibit time.AbortIfError = FALSE; SDO List.Set inhibit time.JumpToLine = FALSE; SDO List.Set inhibit time.Line = 0; SDO List.Set event time.Index = 16#1800; SDO List.Set event time.Subindex = 16#05; SDO List.Set event time.Value = 16#0000; SDO List.Set event time.Size = 16; SDO List.Set event time.AbortIfError = FALSE; SDO List.Set event time.JumpToLine = FALSE; SDO List.Set event time.Line = 0; SDO List.Clear pdo mapping.Index = 16#1A00; SDO List.Clear pdo mapping.Subindex = 16#00; SDO List.Clear pdo mapping.Value = 16#0; SDO List.Clear pdo mapping.Size = 8; SDO List.Clear pdo mapping.AbortIfError = FALSE; SDO List.Clear pdo mapping.JumpToLine = FALSE; SDO List.Clear pdo mapping.Line = 0; SDO List.Set Mapping.Index = 16#1A00; SDO List.Set Mapping.Subindex = 16#01; SDO List.Set Mapping.Value = 16#60410010; SDO List.Set Mapping.Size = 32; SDO List.Set Mapping.AbortIfError = FALSE; SDO List.Set Mapping.JumpToLine = FALSE; SDO List.Set Mapping.Line = 0; SDO List.Set number of mappings.Index = 16#1A00; SDO List.Set number of mappings.Subindex = 16#00; SDO List.Set number of mappings.Value = 16#01; SDO List.Set number of mappings.Size = 8; SDO List.Set number of mappings.AbortIfError = FALSE; SDO List.Set number of mappings.JumpToLine = FALSE; SDO List.Set number of mappings.Line = 0; SDO List.Set and enable COB-ID.Index = 16#1800; SDO List.Set and enable COB-ID.Subindex = 16#01; SDO List.Set and enable COB-ID.Value = 16#00000181; SDO List.Set and enable COB-ID.Size = 32; SDO List.Set and enable COB-ID.AbortIfError = FALSE;
              SDO List.Set and enable COB-ID.JumpToLine = FALSE; SDO List.Set and enable COB-ID.Line = 0; SDO List.Set transmission type.Index = 16#1801; SDO List.Set transmission type.Subindex = 16#02; SDO List.Set transmission type.Value = 16#FF; SDO List.Set transmission type.Size = 8; SDO List.Set transmission type.AbortIfError = FALSE; SDO List.Set transmission type.JumpToLine = FALSE; SDO List.Set transmission type.Line = 0; SDO List.Set inhibit time.Index = 16#1801; SDO List.Set inhibit time.Subindex = 16#03; SDO List.Set inhibit time.Value = 16#0014; SDO List.Set inhibit time.Size = 16; SDO List.Set inhibit time.AbortIfError = FALSE; SDO List.Set inhibit time.JumpToLine = FALSE; SDO List.Set inhibit time.Line = 0; SDO List.Set event time.Index = 16#1801; SDO List.Set event time.Subindex = 16#05; SDO List.Set event time.Value = 16#0000; SDO List.Set event time.Size = 16; SDO List.Set event time.AbortIfError = FALSE; SDO List.Set event time.JumpToLine = FALSE; SDO List.Set event time.Line = 0; SDO List.Clear pdo mapping.Index = 16#1A01; SDO List.Clear pdo mapping.Subindex = 16#00; SDO List.Clear pdo mapping.Value = 16#0; SDO List.Clear pdo mapping.Size = 8; SDO List.Clear pdo mapping.AbortIfError = FALSE; SDO List.Clear pdo mapping.JumpToLine = FALSE; SDO List.Clear pdo mapping.Line = 0; SDO List.Set Mapping.Index = 16#1A01; SDO List.Set Mapping.Subindex = 16#01; SDO List.Set Mapping.Value = 16#60610008; SDO List.Set Mapping.Size = 32; SDO List.Set Mapping.AbortIfError = FALSE; SDO List.Set Mapping.JumpToLine = FALSE; SDO List.Set Mapping.Line = 0; SDO List.Set number of mappings.Index = 16#1A01; SDO List.Set number of mappings.Subindex = 16#00; SDO List.Set number of mappings.Value = 16#01;
              SDO List.Set number of mappings.Size = 8; SDO List.Set number of mappings.AbortIfError = FALSE; SDO List.Set number of mappings.JumpToLine = FALSE; SDO List.Set number of mappings.Line = 0; SDO List.Set and enable COB-ID.Index = 16#1801; SDO List.Set and enable COB-ID.Subindex = 16#01; SDO List.Set and enable COB-ID.Value = 16#00000281; SDO List.Set and enable COB-ID.Size = 32; SDO List.Set and enable COB-ID.AbortIfError = FALSE; SDO List.Set and enable COB-ID.JumpToLine = FALSE; SDO List.Set and enable COB-ID.Line = 0; SDO List.Set transmission type.Index = 16#1802; SDO List.Set transmission type.Subindex = 16#02; SDO List.Set transmission type.Value = 16#FF; SDO List.Set transmission type.Size = 8; SDO List.Set transmission type.AbortIfError = FALSE; SDO List.Set transmission type.JumpToLine = FALSE; SDO List.Set transmission type.Line = 0; SDO List.Set inhibit time.Index = 16#1802; SDO List.Set inhibit time.Subindex = 16#03; SDO List.Set inhibit time.Value = 16#0064; SDO List.Set inhibit time.Size = 16; SDO List.Set inhibit time.AbortIfError = FALSE; SDO List.Set inhibit time.JumpToLine = FALSE; SDO List.Set inhibit time.Line = 0; SDO List.Set event time.Index = 16#1802; SDO List.Set event time.Subindex = 16#05; SDO List.Set event time.Value = 16#0000; SDO List.Set event time.Size = 16; SDO List.Set event time.AbortIfError = FALSE; SDO List.Set event time.JumpToLine = FALSE; SDO List.Set event time.Line = 0; SDO List.Clear pdo mapping.Index = 16#1A02; SDO List.Clear pdo mapping.Subindex = 16#00; SDO List.Clear pdo mapping.Value = 16#0; SDO List.Clear pdo mapping.Size = 8; SDO List.Clear pdo mapping.AbortIfError = FALSE; SDO List.Clear pdo mapping.JumpToLine = FALSE; SDO List.Clear pdo mapping.Line = 0; SDO List.Set Mapping.Index = 16#1A02;
              SDO List.Set Mapping.Subindex = 16#01; SDO List.Set Mapping.Value = 16#60640020; SDO List.Set Mapping.Size = 32; SDO List.Set Mapping.AbortIfError = FALSE; SDO List.Set Mapping.JumpToLine = FALSE; SDO List.Set Mapping.Line = 0; SDO List.Set Mapping.Index = 16#1A02; SDO List.Set Mapping.Subindex = 16#02; SDO List.Set Mapping.Value = 16#606C0020; SDO List.Set Mapping.Size = 32; SDO List.Set Mapping.AbortIfError = FALSE; SDO List.Set Mapping.JumpToLine = FALSE; SDO List.Set Mapping.Line = 0; SDO List.Set number of mappings.Index = 16#1A02; SDO List.Set number of mappings.Subindex = 16#00; SDO List.Set number of mappings.Value = 16#02; SDO List.Set number of mappings.Size = 8; SDO List.Set number of mappings.AbortIfError = FALSE; SDO List.Set number of mappings.JumpToLine = FALSE; SDO List.Set number of mappings.Line = 0; SDO List.Set and enable COB-ID.Index = 16#1802; SDO List.Set and enable COB-ID.Subindex = 16#01; SDO List.Set and enable COB-ID.Value = 16#00000381; SDO List.Set and enable COB-ID.Size = 32; SDO List.Set and enable COB-ID.AbortIfError = FALSE; SDO List.Set and enable COB-ID.JumpToLine = FALSE; SDO List.Set and enable COB-ID.Line = 0; SDO List.Set transmission type.Index = 16#1803; SDO List.Set transmission type.Subindex = 16#02; SDO List.Set transmission type.Value = 16#FF; SDO List.Set transmission type.Size = 8; SDO List.Set transmission type.AbortIfError = FALSE; SDO List.Set transmission type.JumpToLine = FALSE; SDO List.Set transmission type.Line = 0; SDO List.Set inhibit time.Index = 16#1803; SDO List.Set inhibit time.Subindex = 16#03; SDO List.Set inhibit time.Value = 16#0064; SDO List.Set inhibit time.Size = 16; SDO List.Set inhibit time.AbortIfError = FALSE; SDO List.Set inhibit time.JumpToLine = FALSE;
              SDO List.Set inhibit time.Line = 0; SDO List.Set event time.Index = 16#1803; SDO List.Set event time.Subindex = 16#05; SDO List.Set event time.Value = 16#0000; SDO List.Set event time.Size = 16; SDO List.Set event time.AbortIfError = FALSE; SDO List.Set event time.JumpToLine = FALSE; SDO List.Set event time.Line = 0; SDO List.Clear pdo mapping.Index = 16#1A03; SDO List.Clear pdo mapping.Subindex = 16#00; SDO List.Clear pdo mapping.Value = 16#0; SDO List.Clear pdo mapping.Size = 8; SDO List.Clear pdo mapping.AbortIfError = FALSE; SDO List.Clear pdo mapping.JumpToLine = FALSE; SDO List.Clear pdo mapping.Line = 0; SDO List.Set Mapping.Index = 16#1A03; SDO List.Set Mapping.Subindex = 16#01; SDO List.Set Mapping.Value = 16#60FD0020; SDO List.Set Mapping.Size = 32; SDO List.Set Mapping.AbortIfError = FALSE; SDO List.Set Mapping.JumpToLine = FALSE; SDO List.Set Mapping.Line = 0; SDO List.Set number of mappings.Index = 16#1A03; SDO List.Set number of mappings.Subindex = 16#00; SDO List.Set number of mappings.Value = 16#01; SDO List.Set number of mappings.Size = 8; SDO List.Set number of mappings.AbortIfError = FALSE; SDO List.Set number of mappings.JumpToLine = FALSE; SDO List.Set number of mappings.Line = 0; SDO List.Set and enable COB-ID.Index = 16#1803; SDO List.Set and enable COB-ID.Subindex = 16#01; SDO List.Set and enable COB-ID.Value = 16#00000481; SDO List.Set and enable COB-ID.Size = 32; SDO List.Set and enable COB-ID.AbortIfError = FALSE; SDO List.Set and enable COB-ID.JumpToLine = FALSE; SDO List.Set and enable COB-ID.Line = 0; SDO List.Homing method.Index = 16#6098; SDO List.Homing method.Subindex = 16#00; SDO List.Homing method.Value = 16#0000000D; SDO List.Homing method.Size = 8;
              SDO List.Homing method.AbortIfError = FALSE; SDO List.Homing method.JumpToLine = FALSE; SDO List.Homing method.Line = 0; SDO List.Speed during search for switch.Index = 16#6099; SDO List.Speed during search for switch.Subindex = 16#01; SDO List.Speed during search for switch.Value = 10000; SDO List.Speed during search for switch.Size = 32; SDO List.Speed during search for switch.AbortIfError = FALSE; SDO List.Speed during search for switch.JumpToLine = FALSE; SDO List.Speed during search for switch.Line = 0; SDO List.Speed during search for zero.Index = 16#6099; SDO List.Speed during search for zero.Subindex = 16#02; SDO List.Speed during search for zero.Value = 1600; SDO List.Speed during search for zero.Size = 32; SDO List.Speed during search for zero.AbortIfError = FALSE; SDO List.Speed during search for zero.JumpToLine = FALSE; SDO List.Speed during search for zero.Line = 0; ConfigVersion = 50659584
            input  XZ_ActPos : DINT  // Position actual value
            input  XZ_ActVel : DINT  // Velocity actual value
            input  bRotateMotorMin1 : BOOL  // Digital inputs.Bit0
            input  bRotateMotorMax1 : BOOL  // Digital inputs.Bit1
            unmapped channels: Controlword, Target Position, Modes of operation, Profile velocity, Profile acceleration, Target velocity, Profile deceleration, Statusword, Modes of operation display, Digital inputs
    LocalBus_Master_Module : LocalBus Master, Leadshine Technology Co., Ltd., version 3.5.15.40
      PM_3200 : PM_3200, Leadshine Technology Co., Ltd., version 3.5.15.40
          settings: 位置号 = 0
          unmapped channels: ErrorCode, INPUT_0, INPUT_1
      PM0016R : PM0016R, Leadshine Technology Co., Ltd., version 3.5.15.40
          settings: 位置号 = 1
          unmapped channels: ErrorCode, OUTPUT_0
      PM_A0400_IV : PM_A0400_IV, Leadshine Technology Co., Ltd., version 3.5.15.40
          settings: 位置号 = 2; AD0 config.Data_Buffer = 5; AD1 config.Data_Buffer = 5; AD2 config.Data_Buffer = 5; AD3 config.Data_Buffer = 5
          unmapped channels: ErrorCode, ADValue, AnalogDiagnose
    Free_Protocol_RS232_COM : Free Protocol RS232 COM, Leadshine Technology Co., Ltd., version 3.5.15.40
        settings: Vendor.Baudrate = 19200; Vendor.Parity = 2; max send data count = 20; max receive data count = 20; com interval = 25
        unmapped channels: receive control, receive data size, send control, send data size, send data buffer, error status, error id, actual receive data size, actual send data size, receive data
    High_Speed_IO_Module : High Speed IO, Leadshine Technology Co., Ltd., version 3.5.15.40
        settings: HS_IO_Mode_0.High In IO Mode 4 = 196611; HS_IO_Mode_0.High In IO Mode 5 = 196611; Counter_Mask = 48; Ioin_Mask = 1792; HS counter 6.Counter_SetWorkMode = 2; InputFilter Para.Time_In8 = 10; InputFilter Para.Time_In9 = 10; InputFilter Para.Time_In10 = 10
        unmapped channels: Genral_IO_IN, Genral_IO_Out
    SoftMotion General Axis Pool
    Free_Protocol_RS485_COM : Free Protocol RS485 COM, Leadshine Technology Co., Ltd., version 3.5.15.40
        settings: Vendor.Baudrate = 19200; Vendor.Parity = 2; max send data count = 10; max receive data count = 10; com interval = 50
        unmapped channels: receive control, receive data size, send control, send data size, send data buffer, error status, error id, actual receive data size, actual send data size, receive data
  text list GlobalTextList
*)

// Device/Application/DTU/TCP/PLC_SEND
TYPE PLC_SEND:
	STRUCT
		m_nSocketType		:UDINT;	//心跳指令，默认为3，留待判断连接状态。
		m_nCurrentAngle		:REAL;	//为设备当前的旋转角度，单位为角度制下的单位，为度。数精度为1度；
		m_nBedHeight		:REAL;	//为床高，单位为毫米，数据范围为0 - 2000mm；
		m_nBedMovePos		:REAL;	//为床移动距离，以床与探测板的垂直面交线为起点，单位为毫米，数据范围为0 - 3000mm；
		m_nExpStates		:UDINT;	//为曝光状态，枚举值，0:idle（空闲） 1:prep（训机） 2: ready（训机结束，准备完成，可以出束） 3: XrayOn（出射线） 4:XrayOff（关射线） 5 error；
		m_nExpCount			:UDINT;	//为曝光的次数，对应曝光的图像张数；
		m_nFocus			:UDINT;	//焦点大小，0为大焦点 1为小焦点， 焦点具体对应的值由plc设置；
		m_nMHuValue			:REAL;	//热容量，单位MHu ，实际热容量*100得到，实际热容量为小数；
		m_nDirectionState	:UDINT;	//当前旋转状态，默认值-1， 0为正转，1为反转，停止为-1
		m_nMoveState		:UDINT;	//起始、终止状态， 默认值-1， 0为当前扫描方案（与常规意义不同，注意区别）处于准备好状态，可以准备扫描；1为当前扫描方案结束，运动过程中值为-1
		m_nError			:UDINT;	//错误码使用，由王（风杰）工具体阐述内容
		m_fSpeed			:REAL;	//为设备的旋转速度，单位为度/秒，精度0.01度/秒；
		m_fKv				:UDINT;	//管电压，单位为kv（千伏），精度1；
		m_fMA				:REAL;	//管电流，单位为mA（毫安），精度0.1；
		m_fMs				:REAL;	//曝光时间，单位为ms（毫秒），精度0.01；
		m_nSamplingRate		:UDINT;	//采样率，有3个选项：2400帧/圈；1200帧/圈；600帧/圈
		m_nScanProType		:UDINT;	//执行扫描方案的类型，0为自动扫描，1为手动扫描，2为无设置意义的值，默认值为2
		PLC_State			:UDINT;	//PLC状态
		XRAY_State			:UDINT;	//X射线源状态
		AxisErrorID			:UDINT;	//电机错误标志位，含2个伺服电机
	END_STRUCT
END_TYPE

// Device/Application/DTU/TCP/PLC_RECV
TYPE PLC_RECV :
	STRUCT
		m_nSocketType		:UDINT;//0为连接判断信息使用，1为发送设备的有具体意义是参数信息。
      	m_nExpId 			:UDINT;//扫描方式 0为不扫描， 1为 2D 扫描，根据默认帧频曝光设定帧数； 2为CBCT扫描；
       	m_nAngleStart 		:REAL;//为曝光起始位置，在2D和多次曝光情况下，机架旋转到m_nAngleStart位置后再开始曝光，机架不动；CBCT状态下，机架旋转到m_nAngleStart位置后开始曝光，机架运动至m_nAngleEnd位置；最小值为0。
      	m_nAngleEnd  		:REAL;//为曝光的终止位置，在2D和多次曝光情况下不使用；在CBCT状态下，机架的运动终止位置；最小值为0，最大值为360。
      	m_nRotateBegin  	:REAL;//为旋转的起始位置（考虑加速过程）
      	m_nRotateEnd  		:REAL;//为旋转的终止位置（考虑减速过程）
      	m_nKv  				:UDINT;//设置的管电压值，单位为kv，正整数；
      	m_nMA  				:REAL;//设置的管电流值，单位为mA，正整数；
      	m_nMS 				:REAL;//设置一次曝光的时间，单位为ms（毫秒）；设置一次曝光的时间，单位为us（微秒）；精度为1
       	m_nFocus 			:UDINT;//焦点大小设置，枚举值，0为大焦点， 1小焦点；
      	m_nAcquireFrame 	:UDINT;//总帧数，正整数；
      	m_nFramePerCirCle	:UDINT;//每圈获得的帧数，正整数，帧/圈；
      	m_nMoveToward  		:UDINT;//扫描方向，0为不移动，1为进床方向，2为出床方向；
     	m_nScanUseType  	:UDINT;//轴扫还是螺旋扫，0为轴扫，1为螺旋扫；
      	m_nMoveStep  		:REAL;//步进长度，轴扫时使用，单位为mm（毫米）；
     	m_nPitchValue   	:REAL;//螺距长度，螺旋扫时使用，单位为mm（毫米）；
      	m_nCircleCount  	:UDINT;//旋转总圈数，由起始角度和终止角度计算获得，正整数。
      	m_nControlState 	:UDINT;//控制状态 0为正常 1为中止扫描， 2为退出扫描，默认为0
       	m_fScanTop 			:REAL;//扫描上界，以动物趴卧头朝里的方向为基准，从脚至头方向为正方向。单位为毫米，精度为0.01；
       	m_fScanBottom 		:REAL;//扫描下界，以动物趴卧头朝里的方向为基准，从脚至头方向为正方向。单位为毫米，精度为0.01；
		m_fSecondPerCicle	:UDINT;//一圈多少秒
      	m_nSamplingRate  	:UDINT;//采样率，有3个选项：2400帧/圈；1200帧/圈；600帧/圈
       	m_nPrepareState 	:UDINT;//是否亮灯1为亮5灯，0 为不亮5灯
        m_nScanMoveType		:UDINT;//扫描模式 0为手动扫描，1为自动扫描，2为子床位扫描
       	m_nCircleIndex 		:UDINT;//当前第几圈
       	m_nPLCMaCoeff 		:REAL;//灯丝电压值
      	m_nLastMsg  		:UDINT;//CBCT扫描最后一次标志位
       	yuliu_1 			:UDINT;//预留
        yuliu_2				:UDINT;//预留
       	yuliu_3 			:UDINT;//预留一共30个数据
	END_STRUCT
END_TYPE

// Device/Application/DTU/E_LampCmd
{attribute 'qualified_only'}
{attribute 'strict'}
TYPE E_LampCmd :
(
	常亮	:=66,
	慢闪	:=22,
	快闪	:=33,
	关闭 	:=55
);
END_TYPE

// Device/Application/DTU/TCP/Real_TO_Byte_Convert
	(*共用体，2个16位WORD和转换为REAL类型*)
	TYPE Real_TO_Byte_Convert :
	UNION
		rData:REAL;					//32字节
		wByte:ARRAY[0..3] OF BYTE;  //8位字节
	END_UNION
	END_TYPE

// Device/Application/DTU/Axis/AxisState
TYPE AxisState :
STRUCT
	bNetState	:BOOL;//网络状态
	bStandStill	:BOOL;//静止状态
	bPowering	:BOOL;//使能状态
	bHoming		:BOOL;//回零状态
	bErrStop	:BOOL;//停止错误
	bStopState	:BOOL;//停止状态
	bAxisErr	:BOOL;//轴故障
	bPowerOff	:BOOL;//轴使能中
	bContinuousMotion:BOOL;//连续运动状态
	bDisCreteMition:BOOL;//离散运动状态
	bSynchronizedMotion:BOOL;//同步运动中
	
	bAxisGoAbsDone	:BOOL;//绝对定位完成10ms后自动复位
	bAxisGoRelDone	:BOOL;//相对定位完成10ms后自动复位
	bResetDone		:BOOL;//复位完成
	
	rActPosition	:REAL; 	//实际位置
	rActVelocity	:REAL; 	//实际速度
	rActTorque		:REAL;	//实际力矩
	rAcc			:REAL;	//加速度数值
	ErrorID			:UDINT;//故障代码
	
END_STRUCT
END_TYPE


(*
	dActPosition	:DINT; 	//实际位置
	dActVelocity	:DINT; 	//实际速度
	dActTorque		:DINT;	//实际力矩
	dAcc			:DINT;	//加速度数值
*)

// Device/Application/DTU/Axis/AxisCmd
TYPE AxisCmd :
STRUCT
	bPower	: BOOL;	//上电使能
	bHome	: BOOL;	//上升沿触发，10ms后自动复位，请勿一致强制ON
	bJogP	: BOOL;	//正向点动
 	bJogN	: BOOL;	//反向点动
	bAbs	: BOOL;	//上升沿触发，10ms后自动复位，请勿一致强制ON
	bRel	: BOOL;	//上升沿触发，10ms后自动复位，请勿一致强制ON
	bVel	: BOOL;  //速度模式 	
	bStop	: BOOL;	//停止
	bReset	: BOOL;//上升沿触发，10ms后自动复位，请勿一致强制ON
	bSetPos	:BOOL;//设置轴当前位置,home
	bSetPosH:BOOL;//setPos
	AxisPara: AxisParameter;
	bSetHomePara:BOOL;//设置回零参数
END_STRUCT
END_TYPE

// Device/Application/DTU/Axis/AxisParameter
TYPE AxisParameter :
STRUCT
	AxisNodeID			: USINT;	
	rZeroOffset			: REAL;//回原点偏移
	rAbsPosition		: REAL;//AxisGoAbs位置
	rAbsVelocity		: REAL;	//AxisGoAbs速度
	rRelVelocity		: REAL;//AxisGoRel速度
	rRelPosition		: REAL;//AxisGoRel位置
	rVelVelocity		: REAL;//AxisVGo速度
	rAccDec				: REAL;//加减速
	rJogVelocity		: REAL;//点动加减速度默认为点动速度10倍
	rSetPosition		: REAL;//设置轴当前位置变量
	
	iHomeMode		:USINT;
	rHomeHighSpeed	:REAL;
	rHomeLowSpeed	:REAL;
	rHomeAcc		:REAL;
END_STRUCT
END_TYPE


(*	
STRUCT
	AxisNodeID			: USINT;	
	dZeroOffset			: UDINT;//回原点偏移
	dAbsPosition		: DINT;//AxisGoAbs位置
	dAbsVelocity		: UDINT;	//AxisGoAbs速度
	dRelVelocity		: UDINT;//AxisGoRel速度
	dRelPosition		: DINT;//AxisGoRel位置
	dVelVelocity		: DINT;//AxisVGo速度
	dAccDec				: UDINT;//加减速
	dJogVelocity		: DINT;//点动加减速度默认为点动速度10倍
	dSetPosition		: UDINT;//设置轴当前位置变量
	
	iHomeMode		:USINT;
	dHomeHighSpeed	:UDINT;
	dHomeLowSpeed	:UDINT;
	dHomeAcc		:UDINT;
END_STRUCT
*)

// Device/Application/GVL/GVL_SCAN
{attribute 'qualified_only'}
VAR_GLOBAL
		bEnableScout: BOOL;//开启定位像自动曝光3次
		bEnableTrigger: BOOL;
		bJumpScan:BOOL;
END_VAR

// Device/Application/PersistentVars
{attribute 'qualified_only'}
VAR_GLOBAL PERSISTENT RETAIN
END_VAR

// Device/Application/GVL/GVL_State
{attribute 'qualified_only'}
VAR_GLOBAL
		iPLC_State:BYTE;
		
		iXray_State:BYTE; 
		
		bEnable_CTBOX:BOOL;
		
		bBooting:BOOL;
		
		bScoutSecond:BOOL;
END_VAR

// Device/Application/Logic/Trigger_HaoboPannel
PROGRAM Trigger_HaoboPannel
VAR
	count:BYTE;
	booting:BOOL:=TRUE;
	iHopePulse:UINT;
	EncoderNum:UDINT;
	EncoderNum1:DINT;
	iValidTrigger:UINT;
	NumTrigger:BYTE:=4;
	NumTrigger1:BYTE:=28; //DR扫，固定角度曝光28次
	
	TOF_Trig,TOF_Scout:Standard.TOF;
	Blink_Scout:Blink;
	F_TRIG1,F_TRIG2:Standard.F_TRIG;
	R_TRIG1,R_TRIG2:Standard.R_TRIG;
	
	iStartTrigger:UDINT;		//记录开始扫描的起始位置，编码器数值
	iStartTrigger1:DINT;		//记录开始扫描的起始位置，编码器数值
	DB_EncoderNum:UDINT;		//差值
	DB_EncoderNum1:DINT;		//差值
	bTiggerEnable:BOOL;
	R_TRIG_EnableHaobo1,R_TRIG_EnableHaobo2:R_TRIG;
	TON1,TON2:TON;
END_VAR

VAR_INPUT
	iSamplingRate:UINT;
	bEnableTrigger:BOOL;
	bEnableScout:BOOL;
END_VAR

VAR_OUTPUT	
	iActNumPulse:UINT;//有效触发次数
	bScoutPulse:BOOL;
END_VAR

(*README*)
(*脉冲触发信号处理,探测器触发勾选0.Polarity_Param 2.i_HVG_Request 下降沿触发 ，不勾选是上升沿触发*)

(*0.心跳*)
	count:=count+1;
	
(*1.初始化函数*)
	IF booting THEN
		booting:=FALSE;
	END_IF
	
(*2.获取上位机发送的采样率*)//
	iSamplingRate:=UDINT_TO_UINT(WorkStation_TCP.PLC_RECV1.m_nSamplingRate);//采样率，有4个选项：2400帧/圈；1200帧/圈；600帧/圈,360帧/圈 recv[21]
	
(*3.处理多少个脉冲输出一个trigger*)
	CASE iSamplingRate OF 
		360:
			iHopePulse:=360;
		600:
			iHopePulse:=216;//215
		1200:
			iHopePulse:=108;
		2400:
			iHopePulse:=54;//52
		ELSE
			iHopePulse:=360;
	END_CASE
	
(*4.获取旋转编码器的数值*)
	EncoderNum1:=Entity_IO.iEncoderPulse;
	
(*6.开启相对位置，记录开始位置*)	
	R_TRIG2(CLK:=GVL_SCAN.bEnableTrigger , Q=> );
	IF R_TRIG2.Q THEN
		iStartTrigger1:=EncoderNum1;
	END_IF
	
(*6.主逻辑，分2个工作模式，1是根据CBCT角度旋转触发，一个是根据定位像连续触发三次，次数可设*)
	TOF_Trig(IN:= GVL_SCAN.bEnableTrigger, PT:=T#1S , Q=> , ET=> 	);	//使能触发
	TOF_Scout(IN:= GVL_SCAN.bEnableScout,  PT:=T#3S , Q=> , ET=> 	);	//定位像自动触发标志
	
	IF GVL_SCAN.bEnableTrigger AND Entity_IO.bXaryOne THEN
		(*---------------------------处理相对脉冲来作为触发--------------------------------------*)
		DB_EncoderNum1:=ABS(EncoderNum1-iStartTrigger1);
		iValidTrigger:=DINT_TO_UINT(DB_EncoderNum1 MOD iHopePulse);
		
		(*--------------------------CBCT扫描，根据角度输出曝光指令-------------------------------*)
		IF GVL_State.iPLC_State=60 THEN
			(*加时间滤波，经分析，发现增量编码器有跳变的情况出现*)
			(*1.10ms判断*)
			TON1(IN:=Entity_IO.bTriggerOut , PT:=T#12MS , Q=> );
			R_TRIG_EnableHaobo1(CLK:=TON1.Q , Q=> );
			R_TRIG_EnableHaobo2(CLK:=Entity_IO.bTriggerOut , Q=> );
			IF R_TRIG_EnableHaobo1.Q THEN
				bTiggerEnable:=TRUE;
			END_IF
			(*2.出射线后才会出图*)
			IF R_TRIG_EnableHaobo2.Q THEN
				bTiggerEnable:=FALSE;
			END_IF
			(*3.正常出射线出图*)
			IF (iActNumPulse)<=(iSamplingRate+2) THEN
				IF (iValidTrigger)<=1*iHopePulse / 3 THEN  //1/3的占空比，这个时间要和上位机下发的扫描时间对应
					Entity_IO.bTriggerOut:=TRUE;
					Entity_IO.bTriggerHaobo:=FALSE;
				ELSE
					Entity_IO.bTriggerOut:=FALSE;
					Entity_IO.bTriggerHaobo:=bTiggerEnable;
				END_IF
			ELSE
				Entity_IO.bTriggerOut:=FALSE;
				Entity_IO.bTriggerHaobo:=FALSE;
			END_IF
			
			(*-----------------------计数器清零操作-----------------------*)
			IF PLC_PRG.Step_CBCT<=70 THEN
				iActNumPulse:=0;
				Entity_IO.bTriggerOut:=FALSE;
				Entity_IO.bTriggerHaobo:=FALSE;
				bTiggerEnable:=FALSE;
			END_IF
		END_IF	
		(*-------------------------定位像扫描，固定角度直接曝光4次--------------------------------*)
		IF GVL_State.iPLC_State=50 THEN
			IF TOF_Scout.Q=TRUE THEN
			(*-----------------三个以内正常输出------曝光4次----------------------*)
				IF iActNumPulse<NumTrigger THEN
					Blink_Scout(ENABLE:= TRUE, TIMELOW:=T#40MS , TIMEHIGH:=T#40MS , OUT=> );	//TIMEHIGH 的时间要小于曝光时间，当前曝光时间是10ms
					Entity_IO.bTriggerOut:=Blink_Scout.OUT;
					Entity_IO.bTriggerHaobo:=NOT(Blink_Scout.OUT);
					bScoutPulse:=TRUE;			//定位像曝光中
				ELSE
					Blink_Scout(ENABLE:= FALSE);
					Entity_IO.bTriggerOut:=FALSE;
					Entity_IO.bTriggerHaobo:=FALSE;
					bScoutPulse:=FALSE;
				END_IF
			ELSE
				Blink_Scout(ENABLE:= FALSE);
				Entity_IO.bTriggerOut:=FALSE;
				Entity_IO.bTriggerHaobo:=FALSE;
				bScoutPulse:=FALSE;
			END_IF
		END_IF
		
		(*-------------------------DR扫描，固定角度直接曝光28次-------------新增DR扫，固定角度曝光33次0616-----------------*)
		IF GVL_State.iPLC_State=55 OR GVL_State.iPLC_State=58 THEN
			IF TOF_Scout.Q=TRUE THEN
			(*-----------------28个以内正常输出------曝光28次----------------------*)
				IF iActNumPulse<NumTrigger1 THEN
					Blink_Scout(ENABLE:= TRUE, TIMELOW:=T#40MS , TIMEHIGH:=T#40MS , OUT=> );	//TIMEHIGH 的时间要小于曝光时间，当前曝光时间是10ms
					Entity_IO.bTriggerOut:=Blink_Scout.OUT;
					Entity_IO.bTriggerHaobo:=NOT(Blink_Scout.OUT);
					bScoutPulse:=TRUE;			//定位像曝光中
				ELSE
					Blink_Scout(ENABLE:= FALSE);
					Entity_IO.bTriggerOut:=FALSE;
					Entity_IO.bTriggerHaobo:=FALSE;
					bScoutPulse:=FALSE;
				END_IF
			ELSE
				Blink_Scout(ENABLE:= FALSE);
				Entity_IO.bTriggerOut:=FALSE;
				Entity_IO.bTriggerHaobo:=FALSE;
				bScoutPulse:=FALSE;
			END_IF
		END_IF
	ELSE
		bTiggerEnable:=FALSE;
		Entity_IO.bTriggerOut:=FALSE;
		Entity_IO.bTriggerHaobo:=FALSE;
	END_IF
	
	(*-----------------计数一共有多少个脉冲输出--------------------*)
	F_TRIG2(CLK:=(Entity_IO.bTriggerHaobo) 
			AND (GVL_State.iPLC_State=50 OR GVL_State.iPLC_State=60 OR GVL_State.iPLC_State=55 OR GVL_State.iPLC_State=65 OR GVL_State.iPLC_State=58) 
			AND (PLC_PRG.Step_Scout<>42 OR PLC_PRG.Step_DR<>42)  , Q=> );
	IF F_TRIG2.Q THEN					(*计数一共输出多少脉冲*)
		iActNumPulse:=iActNumPulse+1;
	END_IF;
	
(*8.计数器清零*)	
	IF GVL_State.iPLC_State=50 THEN
		(*-----------------------计数器清零操作-----------------------*)
		IF PLC_PRG.Step_Scout<=42 OR PLC_PRG.Step_Scout>=70 THEN
			iActNumPulse:=0;
			Entity_IO.bTriggerOut:=FALSE;
			Entity_IO.bTriggerHaobo:=FALSE;
		END_IF
	ELSIF GVL_State.iPLC_State=55 THEN
		IF PLC_PRG.Step_DR<=42 OR PLC_PRG.Step_DR>=70 THEN
			iActNumPulse:=0;
			Entity_IO.bTriggerOut:=FALSE;
			Entity_IO.bTriggerHaobo:=FALSE;
		END_IF
	ELSIF GVL_State.iPLC_State=60 THEN
		(*-----------------------计数器清零操作-----------------------*)
		IF PLC_PRG.Step_CBCT<=70 THEN
			iActNumPulse:=0;
			Entity_IO.bTriggerOut:=FALSE;
			Entity_IO.bTriggerHaobo:=FALSE;
		END_IF
	ELSIF GVL_State.iPLC_State=58 THEN
		(*-----------------------计数器清零操作-----------------------*)
		IF PLC_PRG.Step_AutoDR<=70 THEN
			iActNumPulse:=0;
			Entity_IO.bTriggerOut:=FALSE;
			Entity_IO.bTriggerHaobo:=FALSE;
		END_IF
	ELSIF GVL_State.iPLC_State=40 THEN
		iActNumPulse:=0;
	END_IF

END_PROGRAM

// Device/Application/Communication/WorkStation_TCP
PROGRAM WorkStation_TCP
VAR
	count:BYTE;
	BOOTING:BOOL:=TRUE;
	TCP_Client_1: NBS.TCP_Client;
	TCP_Server_1: NBS.TCP_Server;
	TCP_Connection_1: NBS.TCP_Connection;
	TCP_Read_1: NBS.TCP_Read;
	TCP_Write_1:NBS.TCP_Write;
	IP:NBS.IP_ADDR;
	ServeruiPort:UINT:=8900;
	xTCP_Client_Enable:BOOL;
	hServer:CAA.HANDLE;
	hConn:CAA.HANDLE;
	
	abyWriteData:ARRAY[0..79] OF BYTE;
	abyReadData:ARRAY[0..119] OF BYTE;
	TON1,TON2:TON;BLINK1:Blink;
	TOF1:TOF;//延迟赋值socket 0
	
	RealByte1	:ARRAY[0..12] OF Real_TO_Byte_Convert;
	RealByte2	:ARRAY[0..12] OF Real_TO_Byte_Convert;
	
	bSetServerIP:BOOL;
	iServerIP1,iServerIP2,iServerIP3,iServerIP4:INT;
	TEMP_IP1,TEMP_IP2,TEMP_IP3,TEMP_IP4,TEMP_IP5:STRING;
	
	PLC_RECV_TEMP:PLC_RECV;//增加缓存
END_VAR

VAR_INPUT
	PLC_SEND1:PLC_SEND;
END_VAR

VAR_OUTPUT	
	PLC_RECV1:PLC_RECV;
	Socket:UDINT;
END_VAR

(*-------------------README----------------------*)
(*0.与上位机通讯并进行数据解析功能*)
(*1.PLC是客户机，IP：192.168.8.100：8899*)	//远程主机
(*2.工作站是服务器，IP：192.168.8.188：8900*)
	
(*0.心跳*)
	count:=count+1;
	
	IF BOOTING THEN  //有风险，可能无法写入数值了 iServerIP4<>0
		IP.sAddr:='192.168.10.20';
		BOOTING:=FALSE;
	END_IF
	
	IF hConn=0 THEN
		BLINK1(ENABLE:=TRUE , TIMELOW:=T#2S , TIMEHIGH:=T#4S , OUT=>xTCP_Client_Enable );
	ELSE
		BLINK1(ENABLE:=FALSE);
		xTCP_Client_Enable:=TRUE;
	END_IF
	
(*0.1 设置服务器IP及端口号*)
	IF bSetServerIP THEN
		TEMP_IP1:=Standard.CONCAT(INT_TO_STRING(iServerIP1),'.');
		TEMP_IP2:=Standard.CONCAT(INT_TO_STRING(iServerIP2),'.');
		TEMP_IP3:=Standard.CONCAT(INT_TO_STRING(iServerIP3),'.');
		TEMP_IP4:=Standard.CONCAT(TEMP_IP3,INT_TO_STRING(iServerIP4));
		TEMP_IP5:=Standard.CONCAT(TEMP_IP1,TEMP_IP2);
		IP.sAddr:=Standard.CONCAT(TEMP_IP5,TEMP_IP4);
		ServeruiPort:=ServeruiPort;
	END_IF
	
(*1.与服务器建立连接*)
	TCP_Connection_1(	
				xEnable:= xTCP_Client_Enable, 
				hServer:= hServer,
				xDone=> , 
				xBusy=> , 
				xError=> ,  
				eError=> , 
				xActive=> , 
				hConnection=> );
	
(*2.客户机设置*)
	TCP_Client_1(
				xEnable:= xTCP_Client_Enable , 
				xDone=> , 
				xBusy=> , 
				xError=> , 
				udiTimeOut:=500000 , 
				ipAddr:=IP , 	//客户端所连接的服务器IP地址
				uiPort:= ServeruiPort, //客户端所连接的服务器端口号
				eError=> , 
				xActive=> , 
				hConnection=>hConn );
				
(*3.读取数据*)
	TCP_Read_1(
				xEnable:=TON1.Q AND TCP_Client_1.xBusy , 
				xDone=> , 
				xBusy=> , 
				xError=> , 
				hConnection:= hConn, 
				szSize:= 120, 
				pData:=ADR(abyReadData) , 
				eError=> , 
				xReady=> , 
				szCount=> );
				
(*4.写入数据并发送*)
	TCP_Write_1(
				xExecute:= TON1.Q AND TCP_Client_1.xBusy, 
				udiTimeOut:= 500000, 
				xDone=> , 
				xBusy=> , 
				xError=> , 
				hConnection:= hConn, 
				szSize:= 80, 
				pData:= ADR(abyWriteData), 
				eError=> );
				
(*5.设计发送和接收周期*)				
	TON1(IN:=NOT TON1.Q , PT:=T#500MS , Q=> , ET=> );
	
(*6.启动发送和接收数据*)
	APLC_RECV();
	APLC_SENG();

ACTION APLC_RECV:

(*----------------------PLC接收数据---------------------------*)//大端接收
(*1.//0为连接判断信息使用，1为发送设备的有具体意义是参数信息*)
	PLC_RECV_TEMP.m_nSocketType	:=BYTE_TO_UDINT(abyReadData[0])+ROL(BYTE_TO_UDINT(abyReadData[1]),8)+ROL(BYTE_TO_UDINT(abyReadData[2]),16)+ROL(BYTE_TO_UDINT(abyReadData[3]),24);
	
(*2.//扫描方式 0为不扫描， 1为定位像扫描； 2为CBCT扫描；3为DR扫描，4为快速扫描，5为旋转电机走到零位*)
	PLC_RECV_TEMP.m_nExpId		:=BYTE_TO_UDINT(abyReadData[4])+ROL(BYTE_TO_UDINT(abyReadData[5]),8)+ROL(BYTE_TO_UDINT(abyReadData[6]),16)+ROL(BYTE_TO_UDINT(abyReadData[7]),24);
	
(*3.//为曝光起始位置，在2D和多次曝光情况下，机架旋转到m_nAngleStart位置后再开始曝光，机架不动；CBCT状态下，机架旋转到m_nAngleStart位置后开始曝光，机架运动至m_nAngleEnd位置；最小值为0。*)
	RealByte2[0].wByte[0]:=abyReadData[8];
	RealByte2[0].wByte[1]:=abyReadData[9];
	RealByte2[0].wByte[2]:=abyReadData[10];
	RealByte2[0].wByte[3]:=abyReadData[11];
	PLC_RECV_TEMP.m_nAngleStart	:=RealByte2[0].rData;

(*4.//为曝光的终止位置，在2D和多次曝光情况下不使用；在CBCT状态下，机架的运动终止位置；最小值为0，最大值为360。*)
	RealByte2[1].wByte[0]:=abyReadData[12];
	RealByte2[1].wByte[1]:=abyReadData[13];
	RealByte2[1].wByte[2]:=abyReadData[14];
	RealByte2[1].wByte[3]:=abyReadData[15];
	PLC_RECV_TEMP.m_nAngleEnd	:=RealByte2[1].rData;

(*5.//为旋转的起始位置（考虑加速过程）*)
	RealByte2[2].wByte[0]:=abyReadData[16];
	RealByte2[2].wByte[1]:=abyReadData[17];
	RealByte2[2].wByte[2]:=abyReadData[18];
	RealByte2[2].wByte[3]:=abyReadData[19];
	PLC_RECV_TEMP.m_nRotateBegin	:=RealByte2[2].rData;
	
(*6.//为旋转的终止位置（考虑减速过程）*)
	RealByte2[3].wByte[0]:=abyReadData[20];
	RealByte2[3].wByte[1]:=abyReadData[21];
	RealByte2[3].wByte[2]:=abyReadData[22];
	RealByte2[3].wByte[3]:=abyReadData[23];
	PLC_RECV_TEMP.m_nRotateEnd	:=RealByte2[3].rData;

(*7.//设置的管电压值，单位为kv，正整数；*)
	PLC_RECV_TEMP.m_nKv	:=BYTE_TO_UDINT(abyReadData[24])+ROL(BYTE_TO_UDINT(abyReadData[25]),8)+ROL(BYTE_TO_UDINT(abyReadData[26]),16)+ROL(BYTE_TO_UDINT(abyReadData[27]),24);

(*8.//设置的管电流值，单位为mA，正整数；*)
	RealByte2[5].wByte[0]:=abyReadData[28];
	RealByte2[5].wByte[1]:=abyReadData[29];
	RealByte2[5].wByte[2]:=abyReadData[30];
	RealByte2[5].wByte[3]:=abyReadData[31];
	PLC_RECV_TEMP.m_nMA	:=RealByte2[5].rData;

(*9.//设置一次曝光的时间，单位为MS（毫秒）；*)
	RealByte2[6].wByte[0]:=abyReadData[32];
	RealByte2[6].wByte[1]:=abyReadData[33];
	RealByte2[6].wByte[2]:=abyReadData[34];
	RealByte2[6].wByte[3]:=abyReadData[35];
	PLC_RECV_TEMP.m_nMS	:=RealByte2[6].rData;

(*10.//焦点大小设置，枚举值，0为大焦点， 1小焦点；*)
	PLC_RECV_TEMP.m_nFocus:=BYTE_TO_UDINT(abyReadData[36]);
	
(*11.//总帧数，正整数；*)
	PLC_RECV_TEMP.m_nAcquireFrame 	:=BYTE_TO_UDINT(abyReadData[40])+ROL(BYTE_TO_UDINT(abyReadData[41]),8)+ROL(BYTE_TO_UDINT(abyReadData[42]),16)+ROL(BYTE_TO_UDINT(abyReadData[43]),24);	
	
(*12.//每圈获得的帧数，正整数，帧/圈；*)	
	PLC_RECV_TEMP.m_nFramePerCirCle	:=BYTE_TO_UDINT(abyReadData[44])+ROL(BYTE_TO_UDINT(abyReadData[45]),8)+ROL(BYTE_TO_UDINT(abyReadData[46]),16)+ROL(BYTE_TO_UDINT(abyReadData[47]),24);	
	
(*13.扫描方向，0为不移动，1为进床方向，2为出床方向；*)	
	PLC_RECV_TEMP.m_nMoveToward		:=BYTE_TO_UDINT(abyReadData[48])+ROL(BYTE_TO_UDINT(abyReadData[49]),8)+ROL(BYTE_TO_UDINT(abyReadData[50]),16)+ROL(BYTE_TO_UDINT(abyReadData[51]),24);
	
(*14.//轴扫还是螺旋扫，0为轴扫，1为螺旋扫；*)
	PLC_RECV_TEMP.m_nScanUseType 	:=BYTE_TO_UDINT(abyReadData[52])+ROL(BYTE_TO_UDINT(abyReadData[53]),8)+ROL(BYTE_TO_UDINT(abyReadData[54]),16)+ROL(BYTE_TO_UDINT(abyReadData[55]),24);
	
	
(*15//步进长度，轴扫时使用，单位为mm（毫米）；*)
	RealByte2[4].wByte[0]:=abyReadData[56];
	RealByte2[4].wByte[1]:=abyReadData[57];
	RealByte2[4].wByte[2]:=abyReadData[58];
	RealByte2[4].wByte[3]:=abyReadData[59];
	PLC_RECV_TEMP.m_nMoveStep:=RealByte2[4].rData;
	
(*16//螺距长度，螺旋扫时使用，单位为mm（毫米）；*)
	RealByte2[7].wByte[0]:=abyReadData[60];
	RealByte2[7].wByte[1]:=abyReadData[61];
	RealByte2[7].wByte[2]:=abyReadData[62];
	RealByte2[7].wByte[3]:=abyReadData[63];
	PLC_RECV_TEMP.m_nPitchValue	:=RealByte2[7].rData;
	
(*17//旋转总圈数，由起始角度和终止角度计算获得，正整数。*)
	PLC_RECV_TEMP.m_nCircleCount  	:=BYTE_TO_UDINT(abyReadData[64])+ROL(BYTE_TO_UDINT(abyReadData[65]),8)+ROL(BYTE_TO_UDINT(abyReadData[66]),16)+ROL(BYTE_TO_UDINT(abyReadData[67]),24);
	
(*18//控制状态 0为正常 1为中止扫描， 2为退出扫描，默认为0*)
	PLC_RECV_TEMP.m_nControlState  	:=BYTE_TO_UDINT(abyReadData[68])+ROL(BYTE_TO_UDINT(abyReadData[69]),8)+ROL(BYTE_TO_UDINT(abyReadData[70]),16)+ROL(BYTE_TO_UDINT(abyReadData[71]),24);

(*19//扫描上界，以动物趴卧头朝里的方向为基准，从脚至头方向为正方向。单位为毫米，精度为0.01；*)
	RealByte2[8].wByte[0]:=abyReadData[72];
	RealByte2[8].wByte[1]:=abyReadData[73];
	RealByte2[8].wByte[2]:=abyReadData[74];
	RealByte2[8].wByte[3]:=abyReadData[75];
	PLC_RECV_TEMP.m_fScanTop	:=RealByte2[8].rData;//零点偏移
	
(*20///扫描下界，以动物趴卧头朝里的方向为基准，从脚至头方向为正方向。单位为毫米，精度为0.01；*)
	RealByte2[9].wByte[0]:=abyReadData[76];
	RealByte2[9].wByte[1]:=abyReadData[77];
	RealByte2[9].wByte[2]:=abyReadData[78];
	RealByte2[9].wByte[3]:=abyReadData[79];
	PLC_RECV_TEMP.m_fScanBottom	:=RealByte2[9].rData;//零点偏移;
	
(*21////一圈多少秒*)
	PLC_RECV_TEMP.m_fSecondPerCicle  :=BYTE_TO_UDINT(abyReadData[80])+ROL(BYTE_TO_UDINT(abyReadData[81]),8)+ROL(BYTE_TO_UDINT(abyReadData[82]),16)+ROL(BYTE_TO_UDINT(abyReadData[83]),24);
		
(*22//采样率，有3个选项：2400帧/圈；1200帧/圈；600帧/圈*)
	PLC_RECV_TEMP.m_nSamplingRate  	:=BYTE_TO_UDINT(abyReadData[84])+ROL(BYTE_TO_UDINT(abyReadData[85]),8)+ROL(BYTE_TO_UDINT(abyReadData[86]),16)+ROL(BYTE_TO_UDINT(abyReadData[87]),24);	

(*23//是否亮灯1为亮5灯，0 为不亮5灯*)
	PLC_RECV_TEMP.m_nPrepareState  	:=BYTE_TO_UDINT(abyReadData[88])+ROL(BYTE_TO_UDINT(abyReadData[89]),8)+ROL(BYTE_TO_UDINT(abyReadData[90]),16)+ROL(BYTE_TO_UDINT(abyReadData[91]),24);

(*24////扫描模式 0为手动扫描，1为自动扫描，2为子床位扫描*)
	PLC_RECV_TEMP.m_nScanMoveType  	:=BYTE_TO_UDINT(abyReadData[92])+ROL(BYTE_TO_UDINT(abyReadData[93]),8)+ROL(BYTE_TO_UDINT(abyReadData[94]),16)+ROL(BYTE_TO_UDINT(abyReadData[95]),24);

(*25//当前第几圈*)
	PLC_RECV_TEMP.m_nCircleIndex  	:=BYTE_TO_UDINT(abyReadData[96])+ROL(BYTE_TO_UDINT(abyReadData[97]),8)+ROL(BYTE_TO_UDINT(abyReadData[98]),16)+ROL(BYTE_TO_UDINT(abyReadData[99]),24);
		
(*26//灯丝电压值*)
	RealByte2[10].wByte[0]:=abyReadData[100];
	RealByte2[10].wByte[1]:=abyReadData[101];
	RealByte2[10].wByte[2]:=abyReadData[102];
	RealByte2[10].wByte[3]:=abyReadData[103];
	PLC_RECV_TEMP.m_nPLCMaCoeff	:=RealByte2[10].rData;	

(*27//CBCT扫描最后一次标志位*)
	PLC_RECV_TEMP.m_nLastMsg  	:=BYTE_TO_UDINT(abyReadData[104])+ROL(BYTE_TO_UDINT(abyReadData[105]),8)+ROL(BYTE_TO_UDINT(abyReadData[106]),16)+ROL(BYTE_TO_UDINT(abyReadData[107]),24);
	
(*28//预留*)
	PLC_RECV_TEMP.yuliu_1	:=BYTE_TO_UDINT(abyReadData[108])+ROL(BYTE_TO_UDINT(abyReadData[109]),8)+ROL(BYTE_TO_UDINT(abyReadData[110]),16)+ROL(BYTE_TO_UDINT(abyReadData[111]),24);//预留//预留一共30个数据
	PLC_RECV_TEMP.yuliu_2	:=BYTE_TO_UDINT(abyReadData[112])+ROL(BYTE_TO_UDINT(abyReadData[113]),8)+ROL(BYTE_TO_UDINT(abyReadData[114]),16)+ROL(BYTE_TO_UDINT(abyReadData[115]),24);//预留//预留一共30个数据
	PLC_RECV_TEMP.yuliu_3	:=BYTE_TO_UDINT(abyReadData[116])+ROL(BYTE_TO_UDINT(abyReadData[117]),8)+ROL(BYTE_TO_UDINT(abyReadData[118]),16)+ROL(BYTE_TO_UDINT(abyReadData[119]),24);//预留//预留一共30个数据


(*---------------------------------------缓存处理------------------------------*)
Socket:=PLC_RECV_TEMP.m_nSocketType;
IF PLC_RECV_TEMP.m_nSocketType=1 THEN
    PLC_RECV1:=PLC_RECV_TEMP;
	TOF1(IN:=FALSE);
ELSE
	TOF1(IN:=TRUE , PT:=T#1S, Q=> , ET=> );
	IF TOF1.Q THEN
		PLC_RECV1.m_nSocketType		:=	PLC_RECV_TEMP.m_nSocketType	;
	ELSE
		PLC_RECV1.m_nSocketType		:=	PLC_RECV1.m_nSocketType	;
	END_IF
	
	PLC_RECV1.m_nExpId 			:=  PLC_RECV1.m_nExpId 			;      
	PLC_RECV1.m_nAngleStart 	:=	PLC_RECV1.m_nAngleStart 	;   
	PLC_RECV1.m_nAngleEnd  		:=	PLC_RECV1.m_nAngleEnd  		;   
	PLC_RECV1.m_nRotateBegin  	:=  PLC_RECV1.m_nRotateBegin  	; 
	PLC_RECV1.m_nRotateEnd  	:=	PLC_RECV1.m_nRotateEnd  	;   
	PLC_RECV1.m_nKv  			:=	PLC_RECV1.m_nKv  			;       
	PLC_RECV1.m_nMA  			:=	PLC_RECV1.m_nMA  			;        
	PLC_RECV1.m_nMS 			:=	PLC_RECV1.m_nMS 			;        
	PLC_RECV1.m_nFocus 			:=  PLC_RECV1.m_nFocus 			;     
	PLC_RECV1.m_nAcquireFrame 	:=  PLC_RECV1.m_nAcquireFrame 	;
	PLC_RECV1.m_nFramePerCirCle	:=  PLC_RECV1.m_nFramePerCirCle	;
	PLC_RECV1.m_nMoveToward  	:=	PLC_RECV1.m_nMoveToward  	 ;
	PLC_RECV1.m_nScanUseType  	:=  PLC_RECV1.m_nScanUseType  	 ;
	PLC_RECV1.m_nMoveStep  		:=  PLC_RECV1.m_nMoveStep  		 ;  
	PLC_RECV1.m_nPitchValue   	:=  PLC_RECV1.m_nPitchValue   	 ;
	PLC_RECV1.m_nCircleCount  	:=  PLC_RECV1.m_nCircleCount  	 ;
	PLC_RECV1.m_nControlState 	:=  PLC_RECV1.m_nControlState 	 ;
	PLC_RECV1.m_fScanTop 		:=	PLC_RECV1.m_fScanTop 		 ;    
	PLC_RECV1.m_fScanBottom 	:=	PLC_RECV1.m_fScanBottom 	 ;  
	PLC_RECV1.m_fSecondPerCicle	:=  PLC_RECV1.m_fSecondPerCicle	;
	PLC_RECV1.m_nSamplingRate  	:=  PLC_RECV1.m_nSamplingRate  	;
	PLC_RECV1.m_nPrepareState 	:=  PLC_RECV1.m_nPrepareState 	 ;
	PLC_RECV1.m_nScanMoveType	:=	PLC_RECV1.m_nScanMoveType	;  
	PLC_RECV1.m_nCircleIndex 	:=	PLC_RECV1.m_nCircleIndex 	;  
	PLC_RECV1.m_nPLCMaCoeff 	:=	PLC_RECV1.m_nPLCMaCoeff 	 ;  
	PLC_RECV1.m_nLastMsg  		:=  PLC_RECV1.m_nLastMsg  		;    
	PLC_RECV1.yuliu_1 			:=  PLC_RECV1.yuliu_1 			;       
	PLC_RECV1.yuliu_2			:=	PLC_RECV1.yuliu_2			 ;       
	PLC_RECV1.yuliu_3 			:=  PLC_RECV1.yuliu_3 			 ;      	
END_IF
END_ACTION

ACTION APLC_SENG:

(*---------------------------------PLC发送数据------------------------------------*)//大端发送机制
(*第一部分，发送数据赋值,待补充*)
	IF PLC_RECV1.m_nSocketType=1 THEN
    	PLC_SEND1.m_nSocketType	  := 1;//心跳指令，默认为3，留待判断连接状态。
	ELSE
    	PLC_SEND1.m_nSocketType	  := 3;//心跳指令，默认为3，留待判断连接状态。
	END_IF                                                                            
	PLC_SEND1.m_nCurrentAngle	:= Axis_XZ.XZ_AxisState.rActPosition;//为设备当前的旋转角度，单位为角度制下的单位，为度。数精度为1度；                                                               
	PLC_SEND1.m_nBedHeight		:= Entity_IO.rRealPos; //为床高，单位为毫米，数据范围为0 - 2000mm；                                                                 
	PLC_SEND1.m_nBedMovePos		:= Axis_QJ.QJ_AxisState.rActPosition;//为床移动距离，以床与探测板的垂直面交线为起点，单位为毫米，数据范围为0 - 3000mm；//增加了偏移                                                 
//	PLC_SEND1.m_nExpStates		:= 22;//为曝光状态，枚举值，0:idle（空闲） 1:prep（训机） 2: ready（训机结束，准备完成，可以出束） 3: XrayOn（出射线） 4:XrayOff（关射线） 5 error；
	PLC_SEND1.m_nExpCount		:= Trigger_HaoboPannel.iActNumPulse;//为曝光的次数，对应曝光的图像张数；                                                                              
//	WorkStation_TCP.PLC_SEND1.m_nFocus			:= XRAY_RS485.Feedback_nFocus;//焦点大小，0为大焦点 1为小焦点， 焦点具体对应的值由plc设置；        //修改为按键提示                                                      
	PLC_SEND1.m_nMHuValue		:= XRAY_RS485.Feedback_nMHuValue;//热容量，单位MHu ，实际热容量*100得到，实际热容量为小数；                                                               
//	PLC_SEND1.m_nDirectionState	:= 22;//当前旋转状态，默认值-1， 0为正转，1为反转，停止为-1                                                                  
//	PLC_SEND1.m_nMoveState		:= 22;//起始、终止状态， 默认值-1， 0为当前扫描方案（与常规意义不同，注意区别）处于准备好状态，可以准备扫描；1为当前扫描方案结束，运动过程中值为-1                      
	PLC_SEND1.m_nError			:= XRAY_RS485.iAlarmNum;//错误码使用，由王（风杰）工具体阐述内容                                                                            
	PLC_SEND1.m_fSpeed			:= Axis_XZ.XZ_AxisState.rActVelocity;//为设备的旋转速度，单位为度/秒，精度0.01度/秒；                                                                     
	PLC_SEND1.m_fKv				:= XRAY_RS485.Feedback_Kv;//管电压，单位为kv（千伏），精度0.01；                                                                          
	PLC_SEND1.m_fMA				:= XRAY_RS485.Feedback_mA;//管电流，单位为mA（毫安），精度0.01；                                                                          
	PLC_SEND1.m_fMs				:= XRAY_RS485.Feedback_ms;//曝光时间，单位为ms（毫秒），精度0.01；                                                                         
	PLC_SEND1.m_nSamplingRate	:= PLC_RECV1.m_nFramePerCirCle;//采样率，有3个选项：2400帧/圈；1200帧/圈；600帧/圈                                                               
//	PLC_SEND1.m_nScanProType	:= 22;//执行扫描方案的类型，0为自动扫描，1为手动扫描，2为无设置意义的值，默认值为2                                                        
	PLC_SEND1.PLC_State			:= GVL_State.iPLC_State;//PLC状态机状态                                                                                             
	PLC_SEND1.XRAY_State		:= GVL_State.iXray_State;//射线源状态                                                                                     
	PLC_SEND1.AxisErrorID		:= Axis_QJ.QJ_AxisState.ErrorID+Axis_XZ.XZ_AxisState.ErrorID*65536; //电机错误报警位,各占16位 
                                                                                   
(*第二部分，发送数据发送*)
(*1,//心跳指令，默认为3，留待判断连接状态。*)
	abyWriteData[3]:=UDINT_TO_BYTE(ROR((PLC_SEND1.m_nSocketType AND 16#FF000000),24));
	abyWriteData[2]:=UDINT_TO_BYTE(ROR((PLC_SEND1.m_nSocketType AND 16#FF0000),16));
	abyWriteData[1]:=UDINT_TO_BYTE(ROR((PLC_SEND1.m_nSocketType AND 16#FF00),8));
	abyWriteData[0]:=UDINT_TO_BYTE(PLC_SEND1.m_nSocketType);
	
(*2//为设备当前的旋转角度，单位为角度制下的单位，为度，数精度为1度*)
	RealByte1[0].rData:=PLC_SEND1.m_nCurrentAngle;	
	abyWriteData[4]:=RealByte1[0].wByte[0];
	abyWriteData[5]:=RealByte1[0].wByte[1];
	abyWriteData[6]:=RealByte1[0].wByte[2];
	abyWriteData[7]:=RealByte1[0].wByte[3];
	
(*3//为床高，单位为毫米，数据范围为0 - 2000mm；*)
	RealByte1[1].rData:=PLC_SEND1.m_nBedHeight;	
	abyWriteData[8]:=RealByte1[1].wByte[0];
	abyWriteData[9]:=RealByte1[1].wByte[1];
	abyWriteData[10]:=RealByte1[1].wByte[2];
	abyWriteData[11]:=RealByte1[1].wByte[3];
	
(*4//为床移动距离，以床与探测板的垂直面交线为起点，单位为毫米，数据范围为0 - 3000mm；*)
	RealByte1[2].rData:=PLC_SEND1.m_nBedMovePos;	
	abyWriteData[12]:=RealByte1[2].wByte[0];
	abyWriteData[13]:=RealByte1[2].wByte[1];
	abyWriteData[14]:=RealByte1[2].wByte[2];
	abyWriteData[15]:=RealByte1[2].wByte[3];
	
(*5//为曝光状态，枚举值，0:idle（空闲） 1:prep（训机） 2: ready（训机结束，准备完成，可以出束） 3: XrayOn（出射线） 4:XrayOff（关射线） 5 error；*)
	abyWriteData[19]:=UDINT_TO_BYTE(ROR((PLC_SEND1.m_nExpStates AND 16#FF000000),24));
	abyWriteData[18]:=UDINT_TO_BYTE(ROR((PLC_SEND1.m_nExpStates AND 16#FF0000),16));
	abyWriteData[17]:=UDINT_TO_BYTE(ROR((PLC_SEND1.m_nExpStates AND 16#FF00),8));
	abyWriteData[16]:=UDINT_TO_BYTE(PLC_SEND1.m_nExpStates);
	
(*6//为曝光的次数，对应曝光的图像张数*)
	abyWriteData[23]:=UDINT_TO_BYTE(ROR((PLC_SEND1.m_nExpCount AND 16#FF000000),24));
	abyWriteData[22]:=UDINT_TO_BYTE(ROR((PLC_SEND1.m_nExpCount AND 16#FF0000),16));
	abyWriteData[21]:=UDINT_TO_BYTE(ROR((PLC_SEND1.m_nExpCount AND 16#FF00),8));
	abyWriteData[20]:=UDINT_TO_BYTE(PLC_SEND1.m_nExpCount AND 16#FF);
	
(*7//焦点大小，0为大焦点 1为小焦点， 焦点具体对应的值由plc设置；*)
	abyWriteData[27]:=UDINT_TO_BYTE(ROR((PLC_SEND1.m_nFocus AND 16#FF000000),24));
	abyWriteData[26]:=UDINT_TO_BYTE(ROR((PLC_SEND1.m_nFocus AND 16#FF0000),16));
	abyWriteData[25]:=UDINT_TO_BYTE(ROR((PLC_SEND1.m_nFocus AND 16#FF00),8));
	abyWriteData[24]:=UDINT_TO_BYTE(PLC_SEND1.m_nFocus);

(*8////热容量，单位MHu ，实际热容量*100得到，实际热容量为小数；*)
	RealByte1[3].rData:=PLC_SEND1.m_nMHuValue;	
	abyWriteData[28]:=RealByte1[3].wByte[0];
	abyWriteData[29]:=RealByte1[3].wByte[1];
	abyWriteData[30]:=RealByte1[3].wByte[2];
	abyWriteData[31]:=RealByte1[3].wByte[3];

(*9.;//当前旋转状态，默认值0， 1为正转，2为反转，停止为0*)	
	abyWriteData[35]:=UDINT_TO_BYTE(ROR((PLC_SEND1.m_nDirectionState AND 16#FF000000),24));
	abyWriteData[34]:=UDINT_TO_BYTE(ROR((PLC_SEND1.m_nDirectionState AND 16#FF0000),16));
	abyWriteData[33]:=UDINT_TO_BYTE(ROR((PLC_SEND1.m_nDirectionState AND 16#FF00),8));
	abyWriteData[32]:=UDINT_TO_BYTE(PLC_SEND1.m_nDirectionState);
	
(*10.起始、终止状态， 默认值0， 1为当前扫描方案（与常规意义不同，注意区别）处于准备好状态，可以准备扫描；2为当前扫描方案结束，运动过程中值为0*)
	abyWriteData[39]:=UDINT_TO_BYTE(ROR((PLC_SEND1.m_nMoveState AND 16#FF000000),24));
	abyWriteData[38]:=UDINT_TO_BYTE(ROR((PLC_SEND1.m_nMoveState AND 16#FF0000),16));
	abyWriteData[37]:=UDINT_TO_BYTE(ROR((PLC_SEND1.m_nMoveState AND 16#FF00),8));
	abyWriteData[36]:=UDINT_TO_BYTE(PLC_SEND1.m_nMoveState);
	
(*11.//错误码使用*)
	abyWriteData[43]:=UDINT_TO_BYTE(ROR((PLC_SEND1.m_nError AND 16#FF000000),24));
	abyWriteData[42]:=UDINT_TO_BYTE(ROR((PLC_SEND1.m_nError AND 16#FF0000),16));
	abyWriteData[41]:=UDINT_TO_BYTE(ROR((PLC_SEND1.m_nError AND 16#FF00),8));
	abyWriteData[40]:=UDINT_TO_BYTE(PLC_SEND1.m_nError AND 16#FF);//旋转电机错误码
	
(*12.//为设备的旋转速度，单位为度/秒，精度0.01度/秒；*)
	RealByte1[4].rData:=PLC_SEND1.m_fSpeed;	
	abyWriteData[44]:=RealByte1[4].wByte[0];
	abyWriteData[45]:=RealByte1[4].wByte[1];
	abyWriteData[46]:=RealByte1[4].wByte[2];
	abyWriteData[47]:=RealByte1[4].wByte[3];
	
(*13.//管电压，单位为kv（千伏），精度1；*)
	abyWriteData[51]:=UDINT_TO_BYTE(ROR((PLC_SEND1.m_fKv AND 16#FF000000),24));
	abyWriteData[50]:=UDINT_TO_BYTE(ROR((PLC_SEND1.m_fKv AND 16#FF0000),16));
	abyWriteData[49]:=UDINT_TO_BYTE(ROR((PLC_SEND1.m_fKv AND 16#FF00),8));
	abyWriteData[48]:=UDINT_TO_BYTE(PLC_SEND1.m_fKv AND 16#FF);
	
(*14.//管电流，单位为mA（毫安），精度0.1*)
	RealByte1[6].rData:=PLC_SEND1.m_fMA;	
	abyWriteData[52]:=RealByte1[6].wByte[0];
	abyWriteData[53]:=RealByte1[6].wByte[1];
	abyWriteData[54]:=RealByte1[6].wByte[2];
	abyWriteData[55]:=RealByte1[6].wByte[3];

(*15.//曝光时间，单位为ms（毫秒），精度0.01；*)
	RealByte1[7].rData:=PLC_SEND1.m_fMs;	
	abyWriteData[56]:=RealByte1[7].wByte[0];
	abyWriteData[57]:=RealByte1[7].wByte[1];
	abyWriteData[58]:=RealByte1[7].wByte[2];
	abyWriteData[59]:=RealByte1[7].wByte[3];
	
(*16.//采样率，有3个选项：2400帧/圈；1200帧/圈；600帧/圈*)
	abyWriteData[63]:=UDINT_TO_BYTE(ROR((PLC_SEND1.m_nSamplingRate AND 16#FF000000),24));
	abyWriteData[62]:=UDINT_TO_BYTE(ROR((PLC_SEND1.m_nSamplingRate AND 16#FF0000),16));
	abyWriteData[61]:=UDINT_TO_BYTE(ROR((PLC_SEND1.m_nSamplingRate AND 16#FF00),8));
	abyWriteData[60]:=UDINT_TO_BYTE(PLC_SEND1.m_nSamplingRate AND 16#FF);
	
(*17.//执行扫描方案的类型，0为自动扫描，1为手动扫描，2为无设置意义的值，默认值为2*)
	abyWriteData[67]:=UDINT_TO_BYTE(ROR((PLC_SEND1.m_nScanProType AND 16#FF000000),24));
	abyWriteData[66]:=UDINT_TO_BYTE(ROR((PLC_SEND1.m_nScanProType AND 16#FF0000),16));
	abyWriteData[65]:=UDINT_TO_BYTE(ROR((PLC_SEND1.m_nScanProType AND 16#FF00),8));
	abyWriteData[64]:=UDINT_TO_BYTE(PLC_SEND1.m_nScanProType AND 16#FF);
	
(*18.//PLC工作状态*)
	abyWriteData[71]:=UDINT_TO_BYTE(ROR((PLC_SEND1.PLC_State AND 16#FF000000),24));
	abyWriteData[70]:=UDINT_TO_BYTE(ROR((PLC_SEND1.PLC_State AND 16#FF0000),16));//
	abyWriteData[69]:=UDINT_TO_BYTE(ROR((PLC_SEND1.PLC_State AND 16#FF00),8));	///
	abyWriteData[68]:=UDINT_TO_BYTE(PLC_SEND1.PLC_State AND 16#FF);				//PLC状态机
	
(*19.//XRAY状态*)
	abyWriteData[75]:=UDINT_TO_BYTE(ROR((PLC_SEND1.XRAY_State AND 16#FF000000),24));
	abyWriteData[74]:=UDINT_TO_BYTE(ROR((PLC_SEND1.XRAY_State AND 16#FF0000),16));  
	abyWriteData[73]:=UDINT_TO_BYTE(ROR((PLC_SEND1.XRAY_State AND 16#FF00),8));     
	abyWriteData[72]:=UDINT_TO_BYTE(PLC_SEND1.XRAY_State AND 16#FF);  //射线源状态机              
	
(*20.//电机错误码*)
	abyWriteData[79]:=UDINT_TO_BYTE(ROR((PLC_SEND1.AxisErrorID AND 16#FF000000),24));//旋转电机故障码
	abyWriteData[78]:=UDINT_TO_BYTE(ROR((PLC_SEND1.AxisErrorID AND 16#FF0000),16));//旋转电机故障码
	abyWriteData[77]:=UDINT_TO_BYTE(ROR((PLC_SEND1.AxisErrorID AND 16#FF00),8));//前进电机故障码
	abyWriteData[76]:=UDINT_TO_BYTE(PLC_SEND1.AxisErrorID AND 16#FF);//前进电机故障码
	
	
	
(*	TEST
	PLC_SEND1.m_nSocketType	  	:= 1;//心跳指令，默认为3，留待判断连接状态。                                                                            
	PLC_SEND1.m_nCurrentAngle	:= 2.1;//为设备当前的旋转角度，单位为角度制下的单位，为度。数精度为1度；                                                               
	PLC_SEND1.m_nBedHeight		:= 3.2;//为床高，单位为毫米，数据范围为0 - 2000mm；                                                                  
	PLC_SEND1.m_nBedMovePos		:= 4.3;//为床移动距离，以床与探测板的垂直面交线为起点，单位为毫米，数据范围为0 - 3000mm；                                                  
	PLC_SEND1.m_nExpStates		:= 5;//为曝光状态，枚举值，0:idle（空闲） 1:prep（训机） 2: ready（训机结束，准备完成，可以出束） 3: XrayOn（出射线） 4:XrayOff（关射线） 5 error；
	PLC_SEND1.m_nExpCount		:= 6;//为曝光的次数，对应曝光的图像张数；                                                                              
	PLC_SEND1.m_nFocus			:= 7;//焦点大小，0为大焦点 1为小焦点， 焦点具体对应的值由plc设置；                                                              
	PLC_SEND1.m_nMHuValue		:= 8.1;//热容量，单位MHu ，实际热容量*100得到，实际热容量为小数；                                                               
	PLC_SEND1.m_nDirectionState	:= 9;//当前旋转状态，默认值-1， 0为正转，1为反转，停止为-1                                                                  
	PLC_SEND1.m_nMoveState		:= 10;//起始、终止状态， 默认值-1， 0为当前扫描方案（与常规意义不同，注意区别）处于准备好状态，可以准备扫描；1为当前扫描方案结束，运动过程中值为-1                      
	PLC_SEND1.m_nError			:= 11;//错误码使用，由王（风杰）工具体阐述内容                                                                            
	PLC_SEND1.m_fSpeed			:= 12.2;//为设备的旋转速度，单位为度/秒，精度0.01度/秒；                                                                     
	PLC_SEND1.m_fKv				:= 13;//管电压，单位为kv（千伏），精度0.01；                                                                          
	PLC_SEND1.m_fMA				:= 14.3;//管电流，单位为mA（毫安），精度0.01；                                                                          
	PLC_SEND1.m_fMs				:= 15.3;//曝光时间，单位为ms（毫秒），精度0.01；                                                                         
	PLC_SEND1.m_nSamplingRate	:= 16;//采样率，有3个选项：2400帧/圈；1200帧/圈；600帧/圈                                                               
	PLC_SEND1.m_nScanProType	:= 17;//执行扫描方案的类型，0为自动扫描，1为手动扫描，2为无设置意义的值，默认值为2                                                        
	PLC_SEND1.PLC_State			:= GVL_State.iPLC_State;//PLC状态机状态                                                                                             
	PLC_SEND1.XRAY_State		:= 18;//电机错误报警位,各占16位                                                                                             
	PLC_SEND1.AxisErrorID		:= Axis_QJ.QJ_AxisState.ErrorID+Axis_XZ.XZ_AxisState.ErrorID*65536;//一共20个数据 
*)
END_ACTION

END_PROGRAM

// Device/Application/BasicFBs/Blink
FUNCTION_BLOCK Blink
(* Function block to simulate a turn signal *)
VAR_INPUT
	ENABLE:BOOL;		(* TRUE:run Blink, FALSE: OUT keeps its value*)
	TIMELOW:TIME;		(* Time for OUT=FALSE *)
	TIMEHIGH:TIME;		(* Time for OUT=TRUE *)
END_VAR
VAR_OUTPUT
	OUT:BOOL;			(* output variable, starting with FALSE *)
END_VAR
VAR
	CLOCK:TP;
END_VAR

(*======================== READ_ME ==============================*)
(*功能块：“闪烁”                                               *)
(***输出周期和占空比一定的矩形波                                 *)
(*=========================== END ===============================*)
		CLOCK( );							
	IF CLOCK.Q=FALSE AND ENABLE THEN			
		CLOCK(IN:=FALSE);							
		IF OUT=FALSE THEN
			CLOCK.PT:=TIMEHIGH;
		ELSE
			CLOCK.PT:=TIMELOW;
		END_IF;
		OUT := NOT OUT;									
		CLOCK(IN:=TRUE);
	ELSIF ENABLE=0 THEN	
		OUT :=0;					
	END_IF;

END_FUNCTION_BLOCK

// Device/Application/Motor/Axis_XZ
PROGRAM Axis_XZ
VAR
	fbMC_AxisConfi		:	MC_AxisConfi_CAN;
	fbMC_Power			:	MC_Power_CAN;
	fbMC_Jog			: 	MC_Jog_CAN;
	fbMC_Stop			: 	MC_STOP_CAN;	
	fbMC_Home			:	MC_HOME_CAN;
	fbMC_Reset			:	MC_Reset_CAN;
	fbMC_MoveAbsolute	: 	MC_MoveAbsoluteIme_CAN;
	fbMC_MoveRelative	: 	MC_MoveRelativeIme_CAN;
	fbMC_ReadStatus		:	MC_ReadStatus_CAN;
	fbMC_HomePara		:	MC_HomeSetPara_CAN;
	count:BYTE;
	
	ControlWord 		AT%QW2 : UINT ;  //ControlWord地址  //地址再核实
	StatusWord  		AT%IW14: UINT ;  //StatusWord地址

	XZ_Addr		: POINTER TO _3SCOS.CANRemoteDevice_Diag;   	//从站ISV2_CAN6040的地址
	XZ_State 	:_3SCOS.DEVICE_STATE;    						//从站ISV2_CAN6040状态
	XZ_NodeID	: BYTE;  										//从站ISV2_CAN6040的节点ID
	
	ASDA_A3_Drive_XZ:Str_LTCANopenAxis;
	
	(*要转换的中间变量*)
	dZeroOffset			: UDINT;//回原点偏移
	dAbsPosition		: DINT;//AxisGoAbs位置
	dAbsVelocity		: UDINT;	//AxisGoAbs速度
	dRelVelocity		: UDINT;//AxisGoRel速度
	dRelPosition		: DINT;//AxisGoRel位置
	dVelVelocity		: DINT;//AxisVGo速度
	dAccDec				: UDINT;//加减速
	dJogVelocity		: DINT;//点动加减速度默认为点动速度10倍
	dSetPosition		: UDINT;//设置轴当前位置变量
	dHomeHighSpeed		:UDINT;
	dHomeLowSpeed		:UDINT;
	dHomeAcc			:UDINT;
	rSpeedRotio			:REAL;
	rEncoderRatio:REAL;
	r1:REAL:=50.00000;
	r2:REAL:=22.00000;
	r3:REAL:=340.0000;
	r4:REAL:=21.00000;
	r5:REAL:=48.00000;
END_VAR

VAR_INPUT
	XZ_AxisCmd			:AxisCmd;
END_VAR

VAR_OUTPUT	
	XZ_AxisState 		:AxisState;
END_VAR

(*--------------README----------*)
(*旋转电机运动子程序*)

(*-----------------Readme-------------------*)
(*前进电机运动子程序*)

(*0.心跳*)
	count:=count+1;
	
(*1.设置轴参数指令*)
	fbMC_AxisConfi(
					Axis:= ASDA_A3_Drive_XZ, 
					Enable:= TRUE, 
					NetWork:= 0, 
					NodeID:= 1, //核实ID是否是2
					ControlWord_Address:= ADR(ControlWord), 
					StatusWord_Address:= ADR(StatusWord), 
					Done=> , 
					StateMachine=> , 
					StatusWord=> , 
					Error=> , 
					ErrorID=> );
					
(*2.判断电机轴状态*)
	fbMC_ReadStatus(Axis:= ASDA_A3_Drive_XZ, Enable:= TRUE , //周期刷新
					valid=> , 
					Busy=> , 
					Error=> XZ_AxisState.bAxisErr,   	//轴错误
					ErrorID=> XZ_AxisState.ErrorID,  	//错误ID
					ErrorStop=>XZ_AxisState.bErrStop , 	//轴停止
					Disabled=> XZ_AxisState.bPowerOff, 	//轴未使能
					stopping=> XZ_AxisState.bStopState, //轴紧急停止
					Homing=>XZ_AxisState.bHoming , 		//回零中
					Standstill=> XZ_AxisState.bStandStill, //使能中
					DiscreteMotion=> XZ_AxisState.bDisCreteMition, 		//离散运动中
					ContinuousMotion=>XZ_AxisState.bContinuousMotion );	//持续运动中
					
	// 可通过 ISV2_CAN6040.CANopenState 状态监测从站 ISV2_CAN6040 是否掉线
	XZ_Addr :=ADR(ASDA_A3_Drive_XZ);
	XZ_State := XZ_Addr^.CANopenState;
	XZ_NodeID:= XZ_Addr^.NodeID ;
					
(*3 读取轴当前位置、速度*)//这里要加上数据转换
	IF r4<>0 AND r5<>0 THEN
		rSpeedRotio:=r1*r2*r3/r4/r5;
	END_IF;
	
	IF rSpeedRotio<>0 THEN
		XZ_AxisState.rActPosition:=LREAL_TO_REAL((DINT_TO_LREAL(XZ_ActPos)/349/rSpeedRotio)*360+21.75);  //改了这值一定要改下面的反馈偏移，切记   //位置反馈的UU值/350（一圈）  *360°  /总速比
		XZ_AxisState.rActVelocity:=DINT_TO_REAL(XZ_ActVel)*6/10/rSpeedRotio;
	END_IF;
	
(*4.使能*)
	fbMC_Power(Axis:= ASDA_A3_Drive_XZ, Enable:= XZ_AxisCmd.bPower, Done=> XZ_AxisState.bPowering, Busy=> , Error=> , ErrorID=> );
	
(*5.回零*)
(*5.1 回零参数*)
	fbMC_HomePara(	Axis:= ASDA_A3_Drive_XZ, 
					Exec:= XZ_AxisCmd.bSetHomePara, 
					HomeMode:=XZ_AxisCmd.AxisPara.iHomeMode , 
					HomeHighSpeed:=dHomeHighSpeed , 
					HomeLowSpeed:= dHomeLowSpeed , 
					Acceleration:= dHomeAcc , 
					Done=> , 
					Busy=> , 
					Error=> , 
					Error_CANopenKenel=> , 
					Error_SDO=> );
					
(*5.2 执行回零命令*)
	fbMC_Home(Axis:=  ASDA_A3_Drive_XZ, Execute:=XZ_AxisCmd.bHome , Position:=dSetPosition);
	

(*6.速度模式*)
(*空*)

(*7.轴绝对运动*)
	fbMC_MoveAbsolute(	Axis:=ASDA_A3_Drive_XZ,Execute:=XZ_AxisCmd.bAbs AND (NOT XZ_AxisState.bStopState),
						Position:=dAbsPosition,
						Velocity:=dAbsVelocity,
						Acceleration:=dAccDec,
						Deceleration:=dAccDec,);
						
(*8.轴相对运动*)
	fbMC_MoveRelative(	Axis:=ASDA_A3_Drive_XZ, Execute:=XZ_AxisCmd.bRel , 
						Distance:= dRelPosition,
						Velocity:=dRelVelocity,
						Acceleration:=dAccDec,Deceleration:=dAccDec,); 
						
(*9.轴点动*)
	fbMC_Jog(	Axis:= ASDA_A3_Drive_XZ, 
				JogForward:=  XZ_AxisCmd.bJogP AND (NOT XZ_AxisCmd.bJogN), 
				JogBackword:=  XZ_AxisCmd.bJogN AND (NOT XZ_AxisCmd.bJogP), 
				Velocity:= dJogVelocity, 
				Acceleration:= dAccDec, 
				Deceleration:=dAccDec,);

(*10.轴停止*)
	fbMC_Stop(	Axis:=ASDA_A3_Drive_XZ,
				Execute:= XZ_AxisCmd.bStop);		
				
	IF fbMC_Stop.Done OR fbMC_Stop.Error THEN
		XZ_AxisCmd.bStop:=FALSE;
	END_IF

(*11.轴复位*)
	fbMC_Reset(	Axis:=ASDA_A3_Drive_XZ,
				Execute:=XZ_AxisCmd.bReset,
				Done=>XZ_AxisState.bResetDone);

				
(*------------------------------------单位换算----------特别重要----------------------*)	
(*因CANOPEN电机功能块只能进行脉冲控制，所以需要增加单位换算逻辑*)
	(*8000*48/50/22*)
	IF rSpeedRotio<>0 THEN		
		dZeroOffset		:=REAL_TO_UDINT((XZ_AxisCmd.AxisPara.rSetPosition-21.75)*rSpeedRotio*349/360);		//回原点偏移
		dAbsPosition	:=REAL_TO_DINT((XZ_AxisCmd.AxisPara.rAbsPosition-21.75)*rSpeedRotio*349/360);		//AxisGoAbs位置
		dAbsVelocity	:=REAL_TO_UDINT(XZ_AxisCmd.AxisPara.rAbsVelocity*rSpeedRotio*349/360);		//AxisGoAbs速度rAbsVelocity
		dRelVelocity	:=REAL_TO_UDINT(XZ_AxisCmd.AxisPara.rRelVelocity*rSpeedRotio*349/360);		//AxisGoRel速度rRelVelocity rRelVelocity
		dRelPosition	:=REAL_TO_DINT(XZ_AxisCmd.AxisPara.rRelPosition*rSpeedRotio*349/360);		//AxisGoRel位置 rRelPosition
		dVelVelocity	:=REAL_TO_DINT(XZ_AxisCmd.AxisPara.rVelVelocity*100);		//AxisVGo速度
		dAccDec			:=REAL_TO_UDINT(XZ_AxisCmd.AxisPara.rAccDec*rSpeedRotio);			//加减速 *1
		dJogVelocity	:=REAL_TO_DINT(XZ_AxisCmd.AxisPara.rJogVelocity*rSpeedRotio*10/6);		//点动加减速度默认为点动速度10倍
		dSetPosition	:=REAL_TO_UDINT((XZ_AxisCmd.AxisPara.rSetPosition-21.75)*rSpeedRotio*349/360);		//设置轴当前位置变量    rSetPosition                                                         
		dHomeHighSpeed	:=REAL_TO_UDINT(XZ_AxisCmd.AxisPara.rHomeHighSpeed*100);	
		dHomeLowSpeed	:=REAL_TO_UDINT(XZ_AxisCmd.AxisPara.rHomeLowSpeed*100);	
		dHomeAcc		:=REAL_TO_UDINT(XZ_AxisCmd.AxisPara.rHomeAcc*100);				                                                            
	END_IF;

END_PROGRAM

// Device/Application/IOs/Entity_IO
PROGRAM Entity_IO
VAR
	(*0.MC508本体IO,16DI@16DO*)
	//12路200KHz/4路1KHz
	DIB0 AT %IX0.0:BOOL;	DIB1 AT %IX0.1:BOOL;	DIB2 AT %IX0.2:BOOL;	DIB3 AT %IX0.3:BOOL;
	DIB4 AT %IX0.4:BOOL;	DIB5 AT %IX0.5:BOOL;	DIB6 AT %IX0.6:BOOL;	DIB7 AT %IX0.7:BOOL;
	DIB8 AT %IX1.0:BOOL;	DIB9 AT %IX1.1:BOOL;	DIB10 AT %IX1.2:BOOL;	DIB11 AT %IX1.3:BOOL;
	DIB12 AT %IX1.4:BOOL;	DIB13 AT %IX1.5:BOOL;	DIB14 AT %IX1.6:BOOL;	DIB15 AT %IX1.7:BOOL;
	//12路200KHz/4路10KHz
	DOB0 AT %QX0.0:BOOL;	DOB1 AT %QX0.1:BOOL;	DOB2 AT %QX0.2:BOOL;	DOB3 AT %QX0.3:BOOL;
	DOB4 AT %QX0.4:BOOL;	DOB5 AT %QX0.5:BOOL;	DOB6 AT %QX0.6:BOOL;	DOB7 AT %QX0.7:BOOL;
	DOB8 AT %QX1.0:BOOL;	DOB9 AT %QX1.1:BOOL;	DOB10 AT %QX1.2:BOOL;	DOB11 AT %QX1.3:BOOL;
	DOB12 AT %QX1.4:BOOL;	DOB13 AT %QX1.5:BOOL;	DOB14 AT %QX1.6:BOOL;	DOB15 AT %QX1.7:BOOL;
	
	(*1.PM3200 32路DI输入*)
	DIX0 AT %IX4.0:BOOL;DIX1 AT %IX4.1:BOOL;DIX2 AT %IX4.2:BOOL;DIX3 AT %IX4.3:BOOL;
	DIX4 AT %IX4.4:BOOL;DIX5 AT %IX4.5:BOOL;DIX6 AT %IX4.6:BOOL;DIX7 AT %IX4.7:BOOL;
	DIX8 AT %IX5.0:BOOL;DIX9 AT %IX5.1:BOOL;DIX10 AT %IX5.2:BOOL;DIX11 AT %IX5.3:BOOL;
	DIX12 AT %IX5.4:BOOL;DIX13 AT %IX5.5:BOOL;DIX14 AT %IX5.6:BOOL;DIX15 AT %IX5.7:BOOL;
	DIX16 AT %IX6.0:BOOL;DIX17 AT %IX6.1:BOOL;DIX18 AT %IX6.2:BOOL;DIX19 AT %IX6.3:BOOL;
	DIX20 AT %IX6.4:BOOL;DIX21 AT %IX6.5:BOOL;DIX22 AT %IX6.6:BOOL;DIX23 AT %IX6.7:BOOL;
	DIX24 AT %IX7.0:BOOL;DIX25 AT %IX7.1:BOOL;DIX26 AT %IX7.2:BOOL;DIX27 AT %IX7.3:BOOL;
	DIX28 AT %IX7.4:BOOL;DIX29 AT %IX7.5:BOOL;DIX30 AT %IX7.6:BOOL;DIX31 AT %IX7.7:BOOL;
	
	(*2.PM0016-R 16路开关量输出*)
	DOX0 AT %QX2.0:BOOL;DOX1 AT %QX2.1:BOOL;DOX2 AT %QX2.2:BOOL;DOX3 AT %QX2.3:BOOL;
	DOX4 AT %QX2.4:BOOL;DOX5 AT %QX2.5:BOOL;DOX6 AT %QX2.6:BOOL;DOX7 AT %QX2.7:BOOL;
	DOX8 AT %QX3.0:BOOL;DOX9 AT %QX3.1:BOOL;DOX10 AT %QX3.2:BOOL;DOX11 AT %QX3.3:BOOL;
	DOX12 AT %QX3.4:BOOL;DOX13 AT %QX3.5:BOOL;DOX14 AT %QX3.6:BOOL;DOX15 AT %QX3.7:BOOL;
	
	(*3.PM-A0400-IV扩展模块AI*)
	AIX0 AT %IW6:INT;		AIX1 AT %IW7:INT;		AIX2 AT %IW8:INT;		AIX3 AT %IW9:INT;
	
	(*4.内部变量*)
	count: BYTE;
	AIX0_TEMP:INT;
	LS_Counter_0,LS_Counter_1			:LS_Counter;  	//计数器指令实例化
	LS_PresetValue_0,LS_PresetValue_1	:LS_PresetValue;//计数器预设值
	bCalibrate:BOOL;//升降电机标定
	rZeroPos_TEMP:INT;
	
END_VAR

VAR_INPUT
	bLeftPannel_LED1,bLeftPannel_LED2,bRightPannel_LED1,bRightPannel_LED2: BOOL;//LED灯
	bXaryOne,bXaryTwo:BOOL;//X射线一档二档信号
	bLaserOut:BOOL;//激光灯控制
	bTriggerOut:BOOL;				//射线源Trigger信号
	bTriggerHaobo:BOOL;				//昊博trigger
	bTriggerPannel:BOOL;			//探测器trigger-4
	bTriggerPannel_NOT:BOOL;//探测器trigger-14
	bUpMotorPos,bUpMotorNeg:BOOL;	//升降电机上升下降控制
	bDelayPower:BOOL;				//延迟断电继电器输出
	bLightYellow:BOOL;				//出束黄色指示灯控制
	bBrakeOut:BOOL;					//前进电机抱闸控制
END_VAR

VAR_OUTPUT	
	(*左右面板输入*)
	LeftPannel_BedUp,LeftPannel_BedDown,LeftPannel_BedFore,LeftPannel_BedBack,LeftPannel_LaserButton,LeftPannel_DistanceMove,LeftPannel_RecordPos,LeftPannel_MoveRecordPos: BOOL;
	RightPannel_BedUp,RightPannel_BedDown,RightPannel_BedFore,RightPannel_BedBack,RightPannel_LaserButton,RightPannel_DistanceMove,RightPannel_RecordPos,RightPannel_MoveRecordPos: BOOL;
	(*前进电机和旋转电机限位*)
	bForeMotorMin,bForeMotorMax,bRotateMotorMin,bRotateMotorMax,bUpMotorMin,bUpMotorZero: BOOL;
	(*急停和门连锁及钥匙开关*)
	bEmergencyStop,bDoorLock,bKeySwitch,bForceBrake:BOOL;
	(*PLC本体输入*)
	bXrayOutState:BOOL;//射线源二档信号
	bXrayBuckey:BOOL;//射线源Buckey信号
	bXray2,bXray3,bXray4:BOOL;//预留经过12V转24V模块后给PLC板的信号
	iEncoderPulse,iEncoderZ:DINT;(*编码器脉冲信号，4倍频率*)
	rRealPos	:REAL;//升降电机位置实际数值
	bXrayFeedback:BOOL;
END_VAR

(*----------------------README--------------------*)
(*0.心跳*)
	count:=count+1;

(*1.左和右PANNEL面板输入*)
	LeftPannel_BedUp		:=DIX3;//床升
	LeftPannel_BedDown		:=DIX4;//床降
	LeftPannel_BedFore		:=DIX5;//床进
	LeftPannel_BedBack		:=DIX2;//床出
	LeftPannel_LaserButton	:=DIX1;//激光灯开关 
	LeftPannel_DistanceMove	:=DIX7;//固定距离进床
	LeftPannel_RecordPos	:=DIX0;//记录预设位置
	LeftPannel_MoveRecordPos:=DIX6;//运动到预设位置
	
	RightPannel_BedUp		:=DIX11;//床升     
	RightPannel_BedDown		:=DIX12;//床降     
	RightPannel_BedFore		:=DIX13;//床进     
	RightPannel_BedBack		:=DIX10;//床出     
	RightPannel_LaserButton	:=DIX15;//激光灯开关  
	RightPannel_DistanceMove:=DIX9; //固定距离进床 
	RightPannel_RecordPos	:=DIX14;//记录预设位置 
	RightPannel_MoveRecordPos:=DIX8;//运动到预设位置
	
(*2.Pannel面板指示灯，左下角D10是LED1,右下角D11是LED2*)
	DOB0:=bTriggerOut	;		//射线源触发信号
	DOB1:=bTriggerHaobo	;		//射线源触发信号
	
	DOB6:=bTriggerPannel	;	//射线源触发信号-14
	DOB7:=bTriggerPannel_NOT;	//射线源触发信号-4

	DOB8:=bLeftPannel_LED1;		//左面板LED1灯，对应激光灯按钮
	DOB9:=bLeftPannel_LED2;		//左面板LED2灯，对应固定距离进床
	DOB10:=bRightPannel_LED1;	//右面板LED1灯，对应固定距离进床
	DOB11:=bRightPannel_LED2;	//右面板LED2灯，对应激光灯按钮


(*3.限位信号及急停门连锁信号*)
	(*以下4个限位信号只能接入驱动器，不支持同时接入PLC，PLC获取开关信息从PDO中获得*)
	bForeMotorMin	:=bForeMotorMin1;//前进电机最小限位
	bForeMotorMax	:=bForeMotorMax1;//前进电机最大限位
	bRotateMotorMin	:=bRotateMotorMin1;//旋转电机最小限位DI1-
	bRotateMotorMax	:=bRotateMotorMax1;//旋转电机最大限位DI2-
	bDoorLock		:=DIX20;//门连锁信号
	bEmergencyStop	:=NOT(DIX21);//急停停止信号
	bUpMotorZero	:=NOT(DIX22);//升降电机上限位，零位信号
	bUpMotorMin		:=NOT(DIX23);//升降电机下限位，下限位信号
	bForceBrake		:=DIX24;//抱闸强制打开信号
	bKeySwitch		:=DIX25;//钥匙开关开机信号
	bXrayFeedback	:=DIX26;//透视信号反馈信号（过门）

(*4.PLC本体输入*)
	bXray2			:=DIB0;	//射线源出射线指示
	bXrayBuckey		:=DIB1;	//射线源Start指示
	bXrayOutState	:=DIB2;	//预留经过12V转24V模块后给PLC板的信号
	bXray3			:=DIB3;
	
(*5.编码器信号输入，4倍频率*)
	LS_Counter_0(xEnable:=TRUE , eChannel:= 4 , xValid=> , xError=> , eErrorID=> , diValue=>iEncoderPulse );
	LS_Counter_1(xEnable:=TRUE , eChannel:= 5 , xValid=> , xError=> , eErrorID=> , diValue=>iEncoderZ );
	(*LS_PresetValue_1(xExecute:= , eChannel:= , eTriggerEdge:= , diPresetValue:= , xDone=> , xBusy=> , xError=> , eErrorID=> );*)

(*6.模拟量采集输入*)
	IF AIX0<=0 THEN
		AIX0_TEMP:=0;
	ELSIF AIX0>=32000 THEN
		AIX0_TEMP:=32000;
	ELSE
		AIX0_TEMP:=AIX0;
	END_IF

	(*6.1.标定*)
	IF bCalibrate THEN 
		rZeroPos_TEMP:=LIMIT(0 ,AIX0 ,32000);
		bCalibrate:=FALSE;
	END_IF
	
	(*6.2.计算实际高度*)
	rRealPos:=400*INT_TO_REAL(AIX0-rZeroPos_TEMP)/INT_TO_REAL(32000-rZeroPos_TEMP);
	
(*7.开关量输出管脚分配*)
	DOX0:=bUpMotorPos	;		//电机上升控制
	DOX1:=bUpMotorNeg	;		//电机下降控制
	DOX2:=bLightYellow	;		//出束黄色指示灯控制
	DOX4:=bXaryOne		;		//X射线透视启动信号
	DOX5:=bLaserOut	  	;		//激光灯输出
	DOX8:=bDelayPower	;		//延迟断电继电器控制
	DOX9:=bBrakeOut	 	;		//抱闸控制

(*8.黄色报警等逻辑*)	
	IF bXaryOne THEN
		bLightYellow:=TRUE;
	ELSE
		bLightYellow:=FALSE;
	END_IF

END_PROGRAM

// Device/Application/Motor/Axis_QJ
PROGRAM Axis_QJ
VAR
	fbMC_AxisConfi		:	MC_AxisConfi_CAN;
	fbMC_Power			:	MC_Power_CAN;
	fbMC_Jog			: 	MC_Jog_CAN;
	fbMC_Stop			: 	MC_STOP_CAN;	
	fbMC_Home			:	MC_HOME_CAN;
	fbMC_Reset			:	MC_Reset_CAN;
	fbMC_MoveAbsolute	: 	MC_MoveAbsoluteIme_CAN;
	fbMC_MoveRelative	: 	MC_MoveRelativeIme_CAN;
	fbMC_ReadStatus		:	MC_ReadStatus_CAN;
	fbMC_HomePara		:	MC_HomeSetPara_CAN;
	fbMC_SetPosition	:	MC_SetPosition;
	
	count:BYTE;
	
	(*要转换的中间变量*)
	dZeroOffset			: UDINT;//回原点偏移
	dAbsPosition		: DINT;//AxisGoAbs位置
	dAbsVelocity		: UDINT;	//AxisGoAbs速度
	dRelVelocity		: UDINT;//AxisGoRel速度
	dRelPosition		: DINT;//AxisGoRel位置
	dVelVelocity		: DINT;//AxisVGo速度
	dAccDec				: UDINT;//加减速
	dJogVelocity		: DINT;//点动加减速度默认为点动速度10倍
	dSetPosition		: UDINT;//设置轴当前位置变量
	dHomeHighSpeed		:UDINT;
	dHomeLowSpeed		:UDINT;
	dHomeAcc			:UDINT;
	
	ControlWord 		AT%QW16 : UINT ;  //ControlWord地址  //地址再核实
	StatusWord  		AT%IW22 : UINT ;  //StatusWord地址

	QJ_Addr		: POINTER TO _3SCOS.CANRemoteDevice_Diag;   	//从站ISV2_CAN6040的地址
	QJ_State 	:_3SCOS.DEVICE_STATE;    						//从站ISV2_CAN6040状态
	QJ_NodeID	: BYTE;  										//从站ISV2_CAN6040的节点ID

	ASDA_A3_Drive_QJ		:Str_LTCANopenAxis;		
END_VAR

VAR_INPUT
	QJ_AxisCmd			:AxisCmd;
END_VAR

VAR_OUTPUT	
	QJ_AxisState 		:AxisState;
END_VAR

(*-----------------Readme-------------------*)
(*前进电机运动子程序,注意增加抱闸控制*)

(*0.心跳*)
	count:=count+1;
	
(*1.设置轴参数指令*)
	fbMC_AxisConfi(
					Axis:= ASDA_A3_Drive_QJ, 
					Enable:= TRUE, 
					NetWork:= 0, 
					NodeID:= 2, //核实ID是否是2
					ControlWord_Address:= ADR(ControlWord), 
					StatusWord_Address:= ADR(StatusWord), 
					Done=> , 
					StateMachine=> , 
					StatusWord=> , 
					Error=> , 
					ErrorID=> );
					
(*2.判断电机轴状态*)
	fbMC_ReadStatus(Axis:= ASDA_A3_Drive_QJ, Enable:= TRUE , //周期刷新
					valid=> , 
					Busy=> , 
					Error=> QJ_AxisState.bAxisErr,   //轴错误
					ErrorID=> QJ_AxisState.ErrorID,  //错误ID
					ErrorStop=>QJ_AxisState.bErrStop , //轴停止
					Disabled=> QJ_AxisState.bPowerOff, //轴未使能
					stopping=> QJ_AxisState.bStopState, //轴紧急停止
					Homing=>QJ_AxisState.bHoming , 			//回零中
					Standstill=> QJ_AxisState.bStandStill, //使能中
					DiscreteMotion=> QJ_AxisState.bDisCreteMition, 		//离散运动中
					ContinuousMotion=>QJ_AxisState.bContinuousMotion );	//持续运动中
					
	// 可通过 ISV2_CAN6040.CANopenState 状态监测从站 ISV2_CAN6040 是否掉线
	QJ_Addr :=ADR(ASDA_A3_Drive_QJ);
	QJ_State := QJ_Addr^.CANopenState;
	QJ_NodeID:= QJ_Addr^.NodeID ;
					
(*3 读取轴当前位置、速度*)
	QJ_AxisState.rActPosition:=DINT_TO_REAL(QJ_ActPos)*10/8000+150.00;//改了这值一定要改下面的反馈偏移，切记      //最终要转换为实际的数据，而不是脉冲数据  10-螺距。8000-第二编码器一圈数值
	QJ_AxisState.rActVelocity:=DINT_TO_REAL(QJ_ActVel)/120;//最终要转换为实际的数据，而不是脉冲数据  *2（速比）*10螺距/8000脉冲
				
(*4.使能*)
	fbMC_Power(Axis:= ASDA_A3_Drive_QJ, Enable:= QJ_AxisCmd.bPower, Done=> QJ_AxisState.bPowering, Busy=> , Error=> , ErrorID=> );
	
(*5.回零*)
(*5.1 回零参数*)
	fbMC_HomePara(	Axis:= ASDA_A3_Drive_QJ, 
					Exec:= QJ_AxisCmd.bSetHomePara, 
					HomeMode:=35,//QJ_AxisCmd.AxisPara.iHomeMode , 
					HomeHighSpeed:=30,//dHomeHighSpeed , 
					HomeLowSpeed:= 10,//dHomeLowSpeed , 
					Acceleration:= 50,//dHomeAcc , 
					Done=> , 
					Busy=> , 
					Error=> , 
					Error_CANopenKenel=> , 
					Error_SDO=> );


(*5.2 执行回零命令*)
	fbMC_Home(Axis:=  ASDA_A3_Drive_QJ, Execute:=QJ_AxisCmd.bHome , Position:=dSetPosition);

(*6.速度模式*)
(*空*)

(*7.轴绝对运动*)
	fbMC_MoveAbsolute(	Axis:=ASDA_A3_Drive_QJ,Execute:=QJ_AxisCmd.bAbs ,//AND (NOT QJ_AxisState.bStopState),
						Position:=dAbsPosition,
						Velocity:=dAbsVelocity,
						Acceleration:=dAccDec,
						Deceleration:=dAccDec,);
						
(*8.轴相对运动*)
	fbMC_MoveRelative(	Axis:=ASDA_A3_Drive_QJ, Execute:= QJ_AxisCmd.bRel , 
						Distance:= dRelPosition,
						Velocity:= dRelVelocity,
						Acceleration:=dAccDec,Deceleration:=dAccDec,); 
						
(*9.轴点动*)
	fbMC_Jog(	Axis:= ASDA_A3_Drive_QJ, 
				JogForward:=  QJ_AxisCmd.bJogP AND (NOT QJ_AxisCmd.bJogN) ,
				JogBackword:=  QJ_AxisCmd.bJogN AND (NOT QJ_AxisCmd.bJogP), 
				Velocity:= dJogVelocity, 
				Acceleration:= dAccDec, 
				Deceleration:= dAccDec,);

(*10.轴停止*)
	fbMC_Stop(	Axis:=ASDA_A3_Drive_QJ,
				Execute:= QJ_AxisCmd.bStop);		
				
	IF fbMC_Stop.Done OR fbMC_Stop.Error THEN
		QJ_AxisCmd.bStop:=FALSE;
	END_IF

(*11.轴复位*)
	fbMC_Reset(	Axis:=ASDA_A3_Drive_QJ,
				Execute:=QJ_AxisCmd.bReset,
				Done=>QJ_AxisState.bResetDone);		
	
(*------------------------------------单位换算--------------------------------*)	//只有位置控制是脉冲，其他是0.1rpm 100000 4000
(*因CANOPEN电机功能块只能进行脉冲控制，所以需要增加单位换算逻辑*)
	dZeroOffset		:=REAL_TO_UDINT((QJ_AxisCmd.AxisPara.rSetPosition-150))*800;		//回原点偏移
	dAbsPosition	:=REAL_TO_DINT((QJ_AxisCmd.AxisPara.rAbsPosition-150))*800;		//AxisGoAbs位置
	dAbsVelocity	:=REAL_TO_UDINT(QJ_AxisCmd.AxisPara.rAbsVelocity)*800;		//AxisGoAbs速度
	dRelVelocity	:=REAL_TO_UDINT(QJ_AxisCmd.AxisPara.rRelVelocity)*800;		//AxisGoRel速度
	dRelPosition	:=REAL_TO_DINT(QJ_AxisCmd.AxisPara.rRelPosition)*800;		//AxisGoRel位置
	dVelVelocity	:=REAL_TO_DINT(QJ_AxisCmd.AxisPara.rVelVelocity*60);		//AxisVGo速度
	dAccDec			:=REAL_TO_UDINT(QJ_AxisCmd.AxisPara.rAccDec)*36;			//加减速
	dJogVelocity	:=REAL_TO_DINT(QJ_AxisCmd.AxisPara.rJogVelocity*120);		//点动加减速度默认为点动速度10倍，最小0.1rpm
	dSetPosition	:=REAL_TO_UDINT(QJ_AxisCmd.AxisPara.rSetPosition)*800;		//设置轴当前位置变量                                                             
	dHomeHighSpeed	:=REAL_TO_UDINT(QJ_AxisCmd.AxisPara.rHomeHighSpeed)*60;	
	dHomeLowSpeed	:=REAL_TO_UDINT(QJ_AxisCmd.AxisPara.rHomeLowSpeed)*60;	
	dHomeAcc		:=REAL_TO_UDINT(QJ_AxisCmd.AxisPara.rHomeAcc)*3600;

END_PROGRAM

// Device/Application/Communication/XRAY_RS485
PROGRAM XRAY_RS485
VAR
	Open_0: COM.Open;Hulala:BOOL;
	Write_0: COM.Write;
	Read_0: COM.Read;
	Close_0: COM.Close;
	xOpen_Exe:BOOL;
	hComHandle:CAA.HANDLE;
	byWrite2:ARRAY [0..3] OF BYTE;
	byWrite3:ARRAY [0..4] OF BYTE;
	byWrite4:ARRAY [0..5] OF BYTE;
	byWrite5:ARRAY [0..6] OF BYTE;
	byWrite6:ARRAY [0..7] OF BYTE;
	byWrite7:ARRAY [0..8] OF BYTE;
	byWrite8:ARRAY [0..9] OF BYTE;
	byWrite9:ARRAY [0..10] OF BYTE;
	xWrite_Exe:BOOL;
	xRead_Exe:BOOL;
    byReadData:ARRAY [0..39] OF BYTE;
    xClose_Exe:BOOL;
	aParamsB19200 : ARRAY [1..7] OF COM.PARAMETER := [
    (udiParameterId := COM.CAA_Parameter_Constants.udiPort,udiValue := 3), 					//指令端口2,3,4,5分别对应硬件接口com2、com0、com1、com3
    (udiParameterId := COM.CAA_Parameter_Constants.udiBaudrate,udiValue := 19200),			//波特率，设置为19200
    (udiParameterId := COM.CAA_Parameter_Constants.udiParity,udiValue := COM.PARITY.NONE),	//校验，设置为无校验
    (udiParameterId := COM.CAA_Parameter_Constants.udiStopBits,udiValue := COM.STOPBIT.ONESTOPBIT),//停止位，1位
    (udiParameterId := COM.CAA_Parameter_Constants.udiTimeout,udiValue := 500),				//超时时间，设置成500ms
    (udiParameterId := COM.CAA_Parameter_Constants.udiByteSize,udiValue := 8),				//数据位
    (udiParameterId := COM.CAA_Parameter_Constants.udiBinary, udiValue := 1)				//二进制参数，启用二进制模式
];		
	TON1,TON2:Standard.TON;
	bSend:BOOL;
	iSize	:INT;
	String2Byte1:String2Byte;
	sSendString:STRING;//
	BLINK1,BLINK2:Blink;
//	Main_Step,Init_Step,DefaultPara_Step,Standby_Step,Rad_Step,Lookup_Step:UINT;
	sRecvString:ARRAY [0..9] OF STRING;	
	sRecvByte:ARRAY [0..39] OF BYTE;	
	i:INT;
	RecvNum,RecvNum1:INT;
	ASCII_Chart_N1:ARRAY [0..9] OF ASCII_Chart_N;
	sRecvStringA1,sRecvStringA2,sRecvStringA3,sRecvStringA4:STRING;
	sRecvStringA5,sRecvStringA6,sRecvStringA7,sRecvStringA0:STRING;
	R_TRIG1:Standard.R_TRIG;
	R30_0,R30_1,R30_2,R30_3,R30_4,R30_5,R30_6:Standard.R_TRIG;
	R10,R20,R30,R40,R50,R60:Standard.R_TRIG;
	TON0_20,TON30_0,TON30_20,TON30_30:Standard.TON;
	f10:F_TRIG;
	BLINK1_ST,BLINK11: BLINK;
	TEMP_MA:UINT;
	TEMP_MS: UINT;
	TON3,TON_ST,TON40,TON_FLR:TON;
	ASCII_Chart_N2:ARRAY[0..30] OF ASCII_Chart_N;
	ASCII_Chart_N_Alarm:ARRAY[0..5] OF ASCII_Chart_N;
	TEMP_FLX1:BOOL;
	TON22:TON;
	R_JUMP20:R_TRIG;
	TON33: TON;
	TON_DelayPara:TON;
	HULALA111:BOOL;
	
	TON11,TON12:TON;
	TON_KV,TON_MA:Standard.TON; //参数设置不对后，延迟进行报警处理0228
	Booting: BOOL;
	hlaldjlk: BOOL;
	Feedback_mA1:REAL;
	Feedback_Kv1:UDINT;
	TON_DELAY:TON;
END_VAR

VAR_INPUT
	
END_VAR

VAR_OUTPUT
	Main_Step,Init_Step,DefaultPara_Step,Standby_Step,Rad_Step,Lookup_Step:UINT;
	Feedback_Kv:UDINT;
	Feedback_mA:REAL;
	Feedback_ms:REAL;
	Feedback_nFocus:UDINT;
	Feedback_nMHuValue:REAL;
	Feedback_AccTime:REAL;
	iAlarmNum:UINT;		//射线源部分的报警位
END_VAR

(*README*)
(*射线源通讯子功能块*)

(*---------------------------------------------------第一部分：串口参数设置------------------------------------------------*)
(*1.open*)
	TON1(IN:=TRUE , PT:=T#5S);//开机后5秒打开串口
	Open_0(xExecute:=TON1.Q , xDone=> , xBusy=> , xError=> , usiListLength:=20 , pParameterList:=ADR(aParamsB19200) , eError=> , hCom=>hComHandle );

(*2.Write*)
	Write_0(
			xExecute:= Open_0.xDone AND bSend, 
			xAbort:= , 
			udiTimeOut:=500 , 
			xDone=> , 
			xBusy=> , 
			xError=> , 
			xAborted=> , 
			hCom:= hComHandle, 
			pBuffer:= , //后面写的
			szSize:= , 
			eError=> );	
			
(*3.Read*)
	TON2(IN:=NOT TON2.Q , PT:=T#20MS , Q=> , ET=> );	//射线源周期100ms
	Read_0(
			xExecute:= Open_0.xDone AND TON2.Q AND NOT(bSend),
			xAbort:= , 
			udiTimeOut:= 500, 
			xDone=> , 
			xBusy=> , 
			xError=> , 
			xAborted=> , 
			hCom:= hComHandle, 
			pBuffer:= ADR(byReadData), 
			szBuffer:= 10, 
			eError=> , 
			szSize=> );
	
(*4.Close*)
	Close_0(
			xExecute:= xClose_Exe, 
			xDone=> , 
			xBusy=> , 
			xError=> , 
			hCom:= hComHandle, 
			eError=> );

(*--------------------------------------------第二部分，数据处理--------------------------------------------------*)
(*2.1 写入命令处理*)
	iSize:=LIMIT(0,LEN(sSendString),10); 		//获取写入的字符串长度	已增加03H结束符+CheckSum和校验	
	String2Byte1(sXrayString:=sSendString , sByte=> );
	Write_0.szSize:=INT_TO_USINT(iSize)+2;
	CASE iSize OF 
	2:
		(*2个字符的命令*)	
		byWrite2[0]:=String2Byte1.sByte[1];
		byWrite2[1]:=String2Byte1.sByte[2];
		byWrite2[2]:=16#03;
		byWrite2[3]:=byWrite2[0]+byWrite2[1]+byWrite2[2];
		Write_0.pBuffer:=ADR(byWrite2);
	3:	
		(*3个字符的命令*)	
		byWrite3[0]:=String2Byte1.sByte[1];
		byWrite3[1]:=String2Byte1.sByte[2];
		byWrite3[2]:=String2Byte1.sByte[3];
		byWrite3[3]:=16#03;
		byWrite3[4]:=byWrite3[0]+byWrite3[1]+byWrite3[2]+byWrite3[3];
		Write_0.pBuffer:=ADR(byWrite3);
	
	4:
		(*4个字符的命令*)	
		byWrite4[0]:=String2Byte1.sByte[1];
		byWrite4[1]:=String2Byte1.sByte[2];
		byWrite4[2]:=String2Byte1.sByte[3];
		byWrite4[3]:=String2Byte1.sByte[4];
		byWrite4[4]:=16#03;
		byWrite4[5]:=byWrite4[0]+byWrite4[1]+byWrite4[2]+byWrite4[3]+byWrite4[4];
		Write_0.pBuffer:=ADR(byWrite4);
	
	5:
		(*5个字符的命令*)	
		byWrite5[0]:=String2Byte1.sByte[1];
		byWrite5[1]:=String2Byte1.sByte[2];
		byWrite5[2]:=String2Byte1.sByte[3];
		byWrite5[3]:=String2Byte1.sByte[4];
		byWrite5[4]:=String2Byte1.sByte[5];
		byWrite5[5]:=16#03;
		byWrite5[6]:=byWrite5[0]+byWrite5[1]+byWrite5[2]+byWrite5[3]+byWrite5[4]+byWrite5[5];
		Write_0.pBuffer:=ADR(byWrite5);
		
	6:
		(*6个字符的命令*)	
		byWrite6[0]:=String2Byte1.sByte[1];
		byWrite6[1]:=String2Byte1.sByte[2];
		byWrite6[2]:=String2Byte1.sByte[3];
		byWrite6[3]:=String2Byte1.sByte[4];
		byWrite6[4]:=String2Byte1.sByte[5];
		byWrite6[5]:=String2Byte1.sByte[6];
		byWrite6[6]:=16#03;
		byWrite6[7]:=byWrite6[0]+byWrite6[1]+byWrite6[2]+byWrite6[3]+byWrite6[4]+byWrite6[5]+byWrite6[6];
		Write_0.pBuffer:=ADR(byWrite6);		
	7:
		(*7个字符的命令*)	
		byWrite7[0]:=String2Byte1.sByte[1];
		byWrite7[1]:=String2Byte1.sByte[2];
		byWrite7[2]:=String2Byte1.sByte[3];
		byWrite7[3]:=String2Byte1.sByte[4];
		byWrite7[4]:=String2Byte1.sByte[5];
		byWrite7[5]:=String2Byte1.sByte[6];
		byWrite7[6]:=String2Byte1.sByte[7];
		byWrite7[7]:=16#03;
		byWrite7[8]:=byWrite7[0]+byWrite7[1]+byWrite7[2]+byWrite7[3]+byWrite7[4]+byWrite7[5]+byWrite7[6]+byWrite7[7];
		Write_0.pBuffer:=ADR(byWrite7);
		
	8:(*8个字符的命令*)	
		byWrite8[0]:=String2Byte1.sByte[1];
		byWrite8[1]:=String2Byte1.sByte[2];
		byWrite8[2]:=String2Byte1.sByte[3];
		byWrite8[3]:=String2Byte1.sByte[4];
		byWrite8[4]:=String2Byte1.sByte[5];
		byWrite8[5]:=String2Byte1.sByte[6];
		byWrite8[6]:=String2Byte1.sByte[7];
		byWrite8[7]:=String2Byte1.sByte[8];
		byWrite8[8]:=16#03;
		byWrite8[9]:=byWrite8[0]+byWrite8[1]+byWrite8[2]+byWrite8[3]+byWrite8[4]+byWrite8[5]+byWrite8[6]+byWrite8[7]+byWrite8[8];
		Write_0.pBuffer:=ADR(byWrite8);
	ELSE
		;//输入错误
	END_CASE
	
(*2.2 读取命令*)
	sRecvByte:=byReadData;

	R_TRIG1(CLK:=Read_0.xDone AND Read_0.szSize<>0, Q=> );		//获取读到了多少个字符
	IF R_TRIG1.Q THEN
		RecvNum:=LIMIT(0,__UXINT_TO_INT(Read_0.szSize)-2,9);	//限制了一下字符0124
	END_IF;

	FOR i:=0 TO RecvNum BY 1 DO 
		ASCII_Chart_N1[i](byASCII:=sRecvByte[i] , sOut_Single=>sRecvString[i] );//需要调用功能块才能有输出
	END_FOR 

	CASE RecvNum OF 		//最长8个字符,如遇到RS和RR的反馈，就自己数字节吧，这里给反馈命令使用
		0:
			sRecvStringA0:='NULL';
		1:
			sRecvStringA0:=sRecvString[0];
		2:
			sRecvStringA0:=CONCAT(STR1:=sRecvString[0] , STR2:= sRecvString[1]);
		3:
			sRecvStringA1:=CONCAT(STR1:=sRecvString[0] , STR2:= sRecvString[1]);
			sRecvStringA0:=CONCAT(STR1:=sRecvStringA1 , STR2:= sRecvString[2]);
		4:
			sRecvStringA1:=CONCAT(STR1:=sRecvString[0] , STR2:= sRecvString[1]);
			sRecvStringA2:=CONCAT(STR1:=sRecvString[2] , STR2:= sRecvString[3]);
			sRecvStringA0:=CONCAT(STR1:=sRecvStringA1 , STR2:= sRecvStringA2);
		5:
			sRecvStringA1:=CONCAT(STR1:=sRecvString[0] , STR2:= sRecvString[1]);
			sRecvStringA2:=CONCAT(STR1:=sRecvString[2] , STR2:= sRecvString[3]);
			sRecvStringA3:=CONCAT(STR1:=sRecvStringA1 , STR2:= sRecvStringA2);
			sRecvStringA0:=CONCAT(STR1:=sRecvStringA3 , STR2:= sRecvString[4]);
		6:
			sRecvStringA1:=CONCAT(STR1:=sRecvString[0] , STR2:= sRecvString[1]);
			sRecvStringA2:=CONCAT(STR1:=sRecvString[2] , STR2:= sRecvString[3]);
			sRecvStringA3:=CONCAT(STR1:=sRecvString[4] , STR2:= sRecvString[5]);
			sRecvStringA4:=CONCAT(STR1:=sRecvStringA1 , STR2:= sRecvStringA2);
			sRecvStringA0:=CONCAT(STR1:=sRecvStringA4 , STR2:= sRecvStringA3);
		7:
			sRecvStringA1:=CONCAT(STR1:=sRecvString[0] , STR2:= sRecvString[1]);
			sRecvStringA2:=CONCAT(STR1:=sRecvString[2] , STR2:= sRecvString[3]);
			sRecvStringA3:=CONCAT(STR1:=sRecvString[4] , STR2:= sRecvString[5]);
			sRecvStringA4:=CONCAT(STR1:=sRecvStringA1 , STR2:= sRecvStringA2);
			sRecvStringA5:=CONCAT(STR1:=sRecvStringA4 , STR2:= sRecvStringA3);
			sRecvStringA0:=CONCAT(STR1:=sRecvStringA5 , STR2:= sRecvString[6]);
		8:
			sRecvStringA1:=CONCAT(STR1:=sRecvString[0] , STR2:= sRecvString[1]);
			sRecvStringA2:=CONCAT(STR1:=sRecvString[2] , STR2:= sRecvString[3]);
			sRecvStringA3:=CONCAT(STR1:=sRecvString[4] , STR2:= sRecvString[5]);
			sRecvStringA4:=CONCAT(STR1:=sRecvString[6] , STR2:= sRecvString[7]);
			sRecvStringA5:=CONCAT(STR1:=sRecvStringA1 , STR2:= sRecvStringA2);
			sRecvStringA6:=CONCAT(STR1:=sRecvStringA3 , STR2:= sRecvStringA4);
			sRecvStringA0:=CONCAT(STR1:=sRecvStringA5 , STR2:= sRecvStringA6);
		9:
			sRecvStringA1:=CONCAT(STR1:=sRecvString[0] , STR2:= sRecvString[1]);
			sRecvStringA2:=CONCAT(STR1:=sRecvString[2] , STR2:= sRecvString[3]);
			sRecvStringA3:=CONCAT(STR1:=sRecvString[4] , STR2:= sRecvString[5]);
			sRecvStringA4:=CONCAT(STR1:=sRecvString[6] , STR2:= sRecvString[7]);
			sRecvStringA5:=CONCAT(STR1:=sRecvStringA1 , STR2:= sRecvStringA2);
			sRecvStringA6:=CONCAT(STR1:=sRecvStringA3 , STR2:= sRecvStringA4);
			sRecvStringA7:=CONCAT(STR1:=sRecvStringA5 , STR2:= sRecvStringA6);
			sRecvStringA0:=CONCAT(STR1:=sRecvStringA7 , STR2:= sRecvString[8]);
		ELSE
			sRecvStringA0:='Too Long';
	END_CASE

(*3.射线源状态机处理*)	
	AXray( );
	GVL_State.iXray_State:=UINT_TO_BYTE(Main_Step);//获取射线源状态

ACTION AXray:

(*---------------------------------------------第三部分：射线源状态机---------------------------------------------------*)
(*0.公共部分*)
	BLINK1(ENABLE:=TON1.Q , TIMELOW:=T#300MS , TIMEHIGH:=T#200MS , OUT=> );
	BLINK1_ST(ENABLE:=TON1.Q , TIMELOW:=T#2S , TIMEHIGH:=T#2S , OUT=> );
	
	(*1.初始化阶段，Initialization Phase*)
			CASE Main_Step OF 
				0:	(*1.初始化阶段，Initialization Phase*)
				IF (sRecvByte[0]= 16#45 AND sRecvByte[1]= 16#4C) OR sRecvStringA0='ST008' THEN //收到ER或EL,确认收到了错误信号，ER可以理解为可恢复，EL为不可恢复 收到EL信号可复位，ER信号只是显示
						Main_Step:=40;
				ELSE
					CASE Init_Step OF 
					0:	//参数初始化
						bSend			:=FALSE;
						DefaultPara_Step:=0;
						Standby_Step	:=0;
						Rad_Step		:=0;//射线步骤复位
						TON11(IN:= TRUE, PT:=T#3S);//开机延迟
						IF TON11.Q THEN
							Init_Step		:=10;
						END_IF
						
					10:	//建立通讯
						TON11(IN:= FALSE);
						sSendString:='ST';
						bSend:=BLINK1_ST.OUT;  
						IF sRecvStringA0='ST001' OR sRecvStringA0='ST002' THEN //收到ST000，通讯正常//此版本是001，所有状态都加1，文档状态说明都加1
							Init_Step:=20;
						ELSE
							iAlarmNum:=301;		//通讯错误
						END_IF
						
					20://检查错误,如果有错误，就复位，没错误，延迟2秒跳转
						iAlarmNum:=0;		//通讯
						IF sRecvByte[0]= 16#45 AND (sRecvByte[1]= 16#4C) THEN //收到ER或EL,确认收到了错误信号，EL可以理解为可恢复，ER为不可恢复 收到EL信号可复位，ER信号只是显示
							sSendString:=sRecvStringA0;
							bSend:=BLINK1.OUT;
							TON0_20(IN:=FALSE);
						ELSE
							TON0_20(IN:=TRUE , PT:=T#2S);//2秒内无报错
							IF TON0_20.Q THEN
								sSendString:='ST';
								bSend:=BLINK1.OUT;
								IF sRecvStringA0='ST002' OR sRecvStringA0='ST001' THEN //收到ST002，通讯正常//此版本是001，所有状态都加1
									Init_Step:=66;
								END_IF
							END_IF;
						END_IF
					66:
						Main_Step:=10;
					ELSE
						;
					END_CASE
				END_IF;
				
				10:	(*写入默认参数，开机只写一次*)	
					IF (sRecvByte[0]= 16#45 AND sRecvByte[1]= 16#4C) OR sRecvStringA0='ST008' THEN //收到ER或EL,确认收到了错误信号，ER可以理解为可恢复，EL为不可恢复 收到EL信号可复位，ER信号只是显示
						Main_Step:=40;
					ELSE
						CASE DefaultPara_Step OF 
						0:
							bSend:=FALSE;
							TON_DelayPara(IN:=FALSE);
							DefaultPara_Step:=5;
					
						5:
							TON_DelayPara(IN:=TRUE , PT:=T#5S , Q=> , ET=> );//写默认参数的时候需要等等射线源一些时间
							IF TON_DelayPara.Q THEN
								DefaultPara_Step:=10;
							END_IF
							
						10://1.关闭AEC
							TON_DelayPara(IN:=FALSE);
							sSendString:='FI000';
							bSend:=BLINK1.OUT;
							IF sRecvStringA0='FI000' THEN
								DefaultPara_Step:=20;
							END_IF
							
						20:
							sSendString:='ET1';
							bSend:=BLINK1.OUT;
							IF sRecvStringA0='ET1' THEN
								DefaultPara_Step:=30;
							END_IF
							
						30://工作模式选择
							sSendString:='WS1';
							bSend:=BLINK1.OUT;
							IF sRecvStringA0='WS1' THEN
								DefaultPara_Step:=40;
							END_IF
						40:
							bSend:=FALSE;
							Main_Step:=20;
						ELSE 
							;
						END_CASE
					END_IF;
		
				20:	(*静止等待状态，Standby Phase*)//注意增加ST，每5秒的周期
					Rad_Step	:=0;
					IF (sRecvByte[0]= 16#45 AND sRecvByte[1]= 16#4C) OR sRecvStringA0='ST008' THEN //收到ER或EL,确认收到了错误信号，ER可以理解为可恢复，EL为不可恢复 收到EL信号可复位，ER信号只是显示
						Main_Step:=40;	
					ELSE
						iAlarmNum:=0;//复位故障	
						IF GVL_State.iPLC_State=40 AND GVL_State.bBooting THEN
							Standby_Step:=10;
						ELSE
							CASE Standby_Step OF
								0:
									bSend		:=FALSE;
									Rad_Step	:=0;//射线步骤复位
									Standby_Step:=9;
									TON33(IN:= FALSE);
									
								9:
									IF sRecvStringA0='FLP0' THEN
										sSendString:='FLP0';
									ELSE
										;
									END_IF	
									R30_0(CLK:=(sRecvStringA0='FLP0') AND Read_0.xDone, Q=> );
									bSend:=R30_0.Q;
		
									TON33(IN:= TRUE, PT:= T#300MS, Q=> , ET=> );
									IF TON33.Q THEN
										Standby_Step:=10;
									END_IF
									
								10://查询指令
									TON33(IN:= FALSE);
									IF (WorkStation_TCP.PLC_RECV1.m_nSocketType=0)  		//=0的时候不写参数
										OR (WorkStation_TCP.PLC_RECV1.m_nControlState>=1 AND WorkStation_TCP.PLC_RECV1.m_nSocketType=1)	//强制退出的时候不写参数
										OR (WorkStation_TCP.PLC_RECV1.m_nExpId=5 		 AND WorkStation_TCP.PLC_RECV1.m_nSocketType=1)	//状态=5的时候不写参数 250701
											 THEN  //开启查询，5秒不能断//可以在这里增加空气校正的条件，例如 OR GVL_State.iPLC_State=控制校正
										CASE Lookup_Step OF 
											0:
												sSendString:='ST';//
												IF BLINK1_ST.OUT THEN
													Lookup_Step:=1;
												END_IF
											1:
												sSendString:='FLK?';//当前电压
												IF BLINK1_ST.OUT THEN
													Lookup_Step:=2;
												END_IF
											2:
												sSendString:='FLM?';//当前电流
												IF BLINK1_ST.OUT THEN
													Lookup_Step:=3;
												END_IF
											3:
												sSendString:='FLT?';//当前透视累计时间
												IF BLINK1_ST.OUT THEN
													Lookup_Step:=4;
												END_IF
											4:
												sSendString:='HE?';//当前球管热量HE
												IF BLINK1_ST.OUT THEN
													Lookup_Step:=5;
												END_IF
											5:
												sSendString:='RF';//当前球管热量HE
												IF BLINK1_ST.OUT THEN
													Lookup_Step:=0;
												END_IF
										END_CASE
										bSend:=BLINK1_ST.OUT;	//2秒查询一次	
										(*数据解析*)
										IF sRecvByte[0]=16#46 AND sRecvByte[1]=16#4C AND sRecvByte[2]=16#4B THEN //FLK 电压
											ASCII_Chart_N2[0](byASCII:= sRecvByte[3], sOut_Single=> );
											ASCII_Chart_N2[1](byASCII:= sRecvByte[4], sOut_Single=> );
											ASCII_Chart_N2[2](byASCII:= sRecvByte[5], sOut_Single=> );
											Feedback_Kv1:=STRING_TO_UDINT(ASCII_Chart_N2[0].sOut_Single)*100+STRING_TO_UDINT(ASCII_Chart_N2[1].sOut_Single)*10+STRING_TO_UDINT(ASCII_Chart_N2[2].sOut_Single);
										END_IF
										
										IF sRecvByte[0]=16#46 AND sRecvByte[1]=16#4C AND sRecvByte[2]=16#4D THEN //FLM 电流
											ASCII_Chart_N2[0](byASCII:= sRecvByte[3], sOut_Single=> );
											ASCII_Chart_N2[1](byASCII:= sRecvByte[4], sOut_Single=> );
											ASCII_Chart_N2[2](byASCII:= sRecvByte[5], sOut_Single=> );
											Feedback_mA1:=STRING_TO_REAL(ASCII_Chart_N2[0].sOut_Single)*10+STRING_TO_REAL(ASCII_Chart_N2[1].sOut_Single)*1+STRING_TO_REAL(ASCII_Chart_N2[2].sOut_Single)*0.1;
										END_IF 
										
										IF sRecvByte[0]=16#46 AND sRecvByte[1]=16#4C AND sRecvByte[2]=16#54 THEN //FLT 累计时间
											ASCII_Chart_N2[0](byASCII:= sRecvByte[3], sOut_Single=> );
											ASCII_Chart_N2[1](byASCII:= sRecvByte[4], sOut_Single=> );
											ASCII_Chart_N2[2](byASCII:= sRecvByte[5], sOut_Single=> );
											Feedback_AccTime:=STRING_TO_REAL(ASCII_Chart_N2[0].sOut_Single)*10+STRING_TO_REAL(ASCII_Chart_N2[1].sOut_Single)*1+STRING_TO_REAL(ASCII_Chart_N2[2].sOut_Single)*0.1;
										END_IF 
										
										IF sRecvByte[0]=16#48 AND sRecvByte[1]=16#45 THEN //HE 球管热量
											ASCII_Chart_N2[0](byASCII:= sRecvByte[2], sOut_Single=> );
											ASCII_Chart_N2[1](byASCII:= sRecvByte[3], sOut_Single=> );
											ASCII_Chart_N2[2](byASCII:= sRecvByte[4], sOut_Single=> );
											Feedback_nMHuValue:=STRING_TO_REAL(ASCII_Chart_N2[0].sOut_Single)*100+STRING_TO_REAL(ASCII_Chart_N2[1].sOut_Single)*10+STRING_TO_REAL(ASCII_Chart_N2[2].sOut_Single);
										END_IF
										TON_KV(IN:=FALSE);
										TON_MA(IN:=FALSE);
										
										IF sRecvByte[0]=16#46 AND sRecvByte[1]=16#4C AND sRecvByte[2]=16#4B THEN // RF的FLK电压反馈
											ASCII_Chart_N2[0](byASCII:= sRecvByte[3], sOut_Single=> );
											ASCII_Chart_N2[1](byASCII:= sRecvByte[4], sOut_Single=> );
											ASCII_Chart_N2[2](byASCII:= sRecvByte[5], sOut_Single=> );
											Feedback_Kv:=STRING_TO_UDINT(ASCII_Chart_N2[0].sOut_Single)*100+STRING_TO_UDINT(ASCII_Chart_N2[1].sOut_Single)*10+STRING_TO_UDINT(ASCII_Chart_N2[2].sOut_Single);
										END_IF
										
										IF sRecvByte[7]=16#46 AND sRecvByte[8]=16#4C AND sRecvByte[9]=16#4D THEN //RF的FLM电流反馈
											ASCII_Chart_N2[0](byASCII:= sRecvByte[10], sOut_Single=> );
											ASCII_Chart_N2[1](byASCII:= sRecvByte[11], sOut_Single=> );
											ASCII_Chart_N2[2](byASCII:= sRecvByte[12], sOut_Single=> );
											Feedback_mA:=STRING_TO_REAL(ASCII_Chart_N2[0].sOut_Single)*10+STRING_TO_REAL(ASCII_Chart_N2[1].sOut_Single)*1+STRING_TO_REAL(ASCII_Chart_N2[2].sOut_Single)*0.1;
										END_IF 
										 
									ELSE
										TON22(IN:= FALSE);
										Standby_Step:=24;
									END_IF
									
								20:	
									sSendString:='ET1';
									bSend:=BLINK1.OUT;
									IF sRecvStringA0='ET1' THEN
										Standby_Step:=21;
									END_IF
									
								21:
									sSendString:=CONCAT('FO',UDINT_TO_STRING(WorkStation_TCP.PLC_RECV1.m_nFocus));
									bSend:=BLINK1.OUT;
									IF sRecvStringA0=sSendString THEN
										Standby_Step:=22;
									END_IF
									
								22:
									sSendString:='EC9';
									bSend:=BLINK1.OUT;
									IF sRecvStringA0='EC9' THEN
										Standby_Step:=23;
									END_IF
									
								23:
									sSendString:='FLF0';
									bSend:=BLINK1.OUT;
									IF sRecvStringA0='FLF0' THEN
										Standby_Step:=24;
									END_IF
									
								24:
									TON_KV(IN:=FALSE);TON_MA(IN:=FALSE);
									sSendString:='FLS100';
									bSend:=BLINK1.OUT;
									IF sRecvStringA0='FLS100' THEN
										Standby_Step:=25;
									END_IF
									
								25:
									(*FLF2,脉冲透视模式，FLF1,连续脉冲模式，电流限制在0.5mA到6mA之间，80kV对应6mA,125KV对应4mA*)
									IF WorkStation_TCP.PLC_RECV1.m_nExpId=4 THEN	//新增脉冲连续模式0610
										sSendString:='FLF1';
									ELSE
										sSendString:='FLF2';
									END_IF
									bSend:=BLINK1.OUT;
									TON_FLR(IN:=FALSE);
									IF sRecvStringA0='FLF2' OR sRecvStringA0='FLF1' THEN
										Standby_Step:=28;
									END_IF
									
								28:	//清除累计时间指令
									sSendString:='FLR1';
									bSend:=BLINK1.OUT;
									TON_FLR(IN:=TRUE , PT:=T#1S , Q=> , ET=> );
									IF TON_FLR.Q OR sRecvStringA0='FLR' THEN
										Standby_Step:=40;
									END_IF
									
								40://写入管电压 小于100最高位补零
									IF WorkStation_TCP.PLC_RECV1.m_nKv>=100 THEN
										sSendString:=CONCAT('FLK',UDINT_TO_STRING(WorkStation_TCP.PLC_RECV1.m_nKv));
									ELSE
										sSendString:=CONCAT('FLK0',UDINT_TO_STRING(WorkStation_TCP.PLC_RECV1.m_nKv));
									END_IF
									bSend:=BLINK1.OUT;
									TEMP_MA:=0;
									
									IF sRecvStringA0=sSendString THEN
										Standby_Step:=50;
									END_IF	
									
									TON_KV(IN:=(sRecvStringA0<>sSendString) , PT:=T#5S , Q=> , ET=> );
									IF TON_KV.Q THEN
										WorkStation_TCP.PLC_SEND1.m_nExpStates	:=5;		//参数写入错误
									END_IF
									
									
								50://写入管电流 5位数字,0.1mA
									TEMP_MA:=LIMIT(1,REAL_TO_UINT(WorkStation_TCP.PLC_RECV1.m_nMA*10),10000);//获取发送过来的数，舍弃×10后的小数
									IF TEMP_MA>=10000 THEN
										sSendString:=CONCAT('FLM',UINT_TO_STRING(TEMP_MA));
									ELSIF TEMP_MA>=1000 AND TEMP_MA<10000 THEN
										sSendString:=CONCAT('FLM',UINT_TO_STRING(TEMP_MA));
									ELSIF TEMP_MA>=100 AND TEMP_MA<1000 THEN
										sSendString:=CONCAT('FLM',UINT_TO_STRING(TEMP_MA));
									ELSIF TEMP_MA>=10 AND TEMP_MA<100 THEN
										sSendString:=CONCAT('FLM0',UINT_TO_STRING(TEMP_MA));
									ELSIF TEMP_MA>=1 AND TEMP_MA<10 THEN
										sSendString:=CONCAT('FLM00',UINT_TO_STRING(TEMP_MA));
									ELSE
										sSendString:='NULL';
									END_IF
									bSend:=BLINK1.OUT;
								
									IF sRecvStringA0=sSendString THEN
										Standby_Step:=60;
									END_IF
									
									TON_MA(IN:=(sRecvStringA0<>sSendString) , PT:=T#5S , Q=> , ET=> );
									IF TON_MA.Q THEN
										WorkStation_TCP.PLC_SEND1.m_nExpStates	:=5;	//参数写入错误
									END_IF				

								60://收到透视信号，跳转到射线阶段
									bSend:=FALSE;
									GVL_State.bScoutSecond:=FALSE;//FUWEI
									IF Entity_IO.bXaryOne THEN
										Standby_Step:=66;
									END_IF;	
									
									sSendString:='ST';		//当前电流
									bSend:=BLINK1_ST.OUT;	//2秒查询一次	
									WorkStation_TCP.PLC_SEND1.m_nExpStates	:=6; 			//参数写入正确
								66:
									TON_DELAY(IN:=FALSE );
									WorkStation_TCP.PLC_SEND1.m_nExpStates	:=7; 			//参数写入后赋其他值
									bSend:=FALSE;
									Main_Step:=30;	
								ELSE
									;
								END_CASE
							END_IF;
						END_IF;
						
						(*-----------------------------------------ER故障无需软件恢复-------------------------------------------------------*)
						IF (sRecvByte[0]= 16#45 AND sRecvByte[1]= 16#52)   THEN //收到ER，只显示故障码，不发送  //16#52  52是ER
							(*处理故障代码显示*)
							CASE RecvNum OF //最多3位故障代码
								3:
									ASCII_Chart_N_Alarm[0](byASCII:=sRecvByte[2] , sOut_Single=> );
									iAlarmNum:=STRING_TO_BYTE(ASCII_Chart_N_Alarm[0].sOut_Single);
								4:
									ASCII_Chart_N_Alarm[1](byASCII:=sRecvByte[2] , sOut_Single=> );
									ASCII_Chart_N_Alarm[2](byASCII:=sRecvByte[3] , sOut_Single=> );
									iAlarmNum:=STRING_TO_BYTE(ASCII_Chart_N_Alarm[1].sOut_Single)*10+STRING_TO_BYTE(ASCII_Chart_N_Alarm[2].sOut_Single);
								5:
									ASCII_Chart_N_Alarm[3](byASCII:=sRecvByte[2] , sOut_Single=> );
									ASCII_Chart_N_Alarm[4](byASCII:=sRecvByte[3] , sOut_Single=> );
									ASCII_Chart_N_Alarm[5](byASCII:=sRecvByte[4] , sOut_Single=> );
									iAlarmNum:=STRING_TO_BYTE(ASCII_Chart_N_Alarm[3].sOut_Single)*100+STRING_TO_BYTE(ASCII_Chart_N_Alarm[4].sOut_Single)*10+STRING_TO_BYTE(ASCII_Chart_N_Alarm[5].sOut_Single);
								ELSE
									iAlarmNum:=iAlarmNum;
							END_CASE	
						END_IF;
							
				30:(*射线准备，出射线阶段*)
					Standby_Step:=0;
					IF (sRecvByte[0]= 16#45 AND sRecvByte[1]= 16#4C) OR sRecvStringA0='ST008' THEN //收到ER或EL,确认收到了错误信号，ER可以理解为可恢复，EL为不可恢复 收到EL信号可复位，ER信号只是显示
						Main_Step:=40;	
					ELSE
						iAlarmNum:=0;//复位故障
						//查询球管热量
						IF sRecvByte[0]=16#48 AND sRecvByte[1]=16#45 THEN //HE 球管热量
							ASCII_Chart_N2[0](byASCII:= sRecvByte[2], sOut_Single=> );
							ASCII_Chart_N2[1](byASCII:= sRecvByte[3], sOut_Single=> );
							ASCII_Chart_N2[2](byASCII:= sRecvByte[4], sOut_Single=> );
							Feedback_nMHuValue:=STRING_TO_REAL(ASCII_Chart_N2[0].sOut_Single)*100+STRING_TO_REAL(ASCII_Chart_N2[1].sOut_Single)*10+STRING_TO_REAL(ASCII_Chart_N2[2].sOut_Single);
						END_IF
						
						IF GVL_State.iPLC_State=40 AND GVL_State.bBooting THEN
							Main_Step		:=20; 				//系统待机下回到射线源待机状态
							Standby_Step	:=10;
							Rad_Step		:=0;
							GVL_State.bBooting:=FALSE;
						ELSE
							(*---------------------------曝光状态---------------------------------*)
							CASE Rad_Step OF
								0://初始化阶段
									TON_DELAY(IN:=FALSE);
									TON_ST(IN:=FALSE);
									Rad_Step:=10;
								10:
									IF sRecvStringA0='FLP1' THEN
										Rad_Step	:=20;
									END_IF;	
									
									IF sRecvStringA0='FLP0' THEN
										Rad_Step	:=40;
									END_IF;	
									
								20://FLX1
									IF sRecvStringA0='FLX1' THEN //OR Entity_IO.bXrayBuckey THEN
										Rad_Step	:=30;
									END_IF;
									
									IF sRecvStringA0='FLP0' THEN
										Rad_Step	:=40;
									END_IF;	
									
								
								30://允许出束阶段
									TON_ST(IN:=FALSE);
									IF sRecvStringA0='FLX0' OR sRecvStringA0='FLP0' THEN //收到FLX0或FLP0，曝光结束
										Rad_Step	:=40;
									ELSE
										;
									END_IF
									
								 40://结束
								 	TON_DELAY(IN:=TRUE , PT:=T#12S , Q=> , ET=> );
									IF TON_DELAY.Q THEN
										Standby_Step:=0;
										Rad_Step	:=88;
										Main_Step	:=20;
									END_IF;
								ELSE
									;
							END_CASE
						END_IF
					END_IF;
					
					(*-----------------------------------------ER故障无需软件恢复-------------------------------------------------------*)
					IF (sRecvByte[0]= 16#45 AND sRecvByte[1]= 16#52)   THEN //收到ER，只显示故障码，不发送  //16#52  52是ER
						(*处理故障代码显示*)
						CASE RecvNum OF //最多3位故障代码
							3:
								ASCII_Chart_N_Alarm[0](byASCII:=sRecvByte[2] , sOut_Single=> );
								iAlarmNum:=STRING_TO_BYTE(ASCII_Chart_N_Alarm[0].sOut_Single);
							4:
								ASCII_Chart_N_Alarm[1](byASCII:=sRecvByte[2] , sOut_Single=> );
								ASCII_Chart_N_Alarm[2](byASCII:=sRecvByte[3] , sOut_Single=> );
								iAlarmNum:=STRING_TO_BYTE(ASCII_Chart_N_Alarm[1].sOut_Single)*10+STRING_TO_BYTE(ASCII_Chart_N_Alarm[2].sOut_Single);
							5:
								ASCII_Chart_N_Alarm[3](byASCII:=sRecvByte[2] , sOut_Single=> );
								ASCII_Chart_N_Alarm[4](byASCII:=sRecvByte[3] , sOut_Single=> );
								ASCII_Chart_N_Alarm[5](byASCII:=sRecvByte[4] , sOut_Single=> );
								iAlarmNum:=STRING_TO_BYTE(ASCII_Chart_N_Alarm[3].sOut_Single)*100+STRING_TO_BYTE(ASCII_Chart_N_Alarm[4].sOut_Single)*10+STRING_TO_BYTE(ASCII_Chart_N_Alarm[5].sOut_Single);
							ELSE
								iAlarmNum:=iAlarmNum;
						END_CASE	
					END_IF;
						
				40:	//错误状态下只显示EL故障
					IF (sRecvByte[0]= 16#45 AND sRecvByte[1]= 16#4C) OR sRecvStringA0='ST008'  THEN 	//收到ER或EL,确认收到了错误信号，ER可以理解为可恢复，EL为不可恢复 收到EL信号可复位，ER信号只是显示
						IF sRecvStringA0='ST008' THEN
							sSendString:='EL ？';
							bSend:=BLINK1.OUT;
						END_IF 
							
						IF Read_0.xDone AND (sRecvByte[0]= 16#45 AND sRecvByte[1]= 16#4C) THEN
							sSendString:=sRecvStringA0;							//收到EL，发送故障码，同时发送EL恢复故障
							f10(CLK:=(sRecvByte[0]= 16#45 AND sRecvByte[1]= 16#4C) AND Read_0.xDone  , Q=> bSend);//发一次回一次
						ELSE
							f10(CLK:=FALSE  , Q=> bSend);//发一次回一次
						END_IF;
						
						BLINK2(ENABLE:=TRUE , TIMELOW:=T#1S , TIMEHIGH:=T#1S , OUT=> );
						IF BLINK2.OUT THEN
							sSendString:='ST';//查询ST状态
							bSend:=BLINK2.OUT AND NOT(f10.Q);
						END_IF
					
						(*处理EL故障代码显示*)
						CASE RecvNum OF //最多3位故障代码
							3:
								ASCII_Chart_N_Alarm[0](byASCII:=sRecvByte[2] , sOut_Single=> );
								iAlarmNum:=STRING_TO_BYTE(ASCII_Chart_N_Alarm[0].sOut_Single);
							4:
								ASCII_Chart_N_Alarm[1](byASCII:=sRecvByte[2] , sOut_Single=> );
								ASCII_Chart_N_Alarm[2](byASCII:=sRecvByte[3] , sOut_Single=> );
								iAlarmNum:=STRING_TO_BYTE(ASCII_Chart_N_Alarm[1].sOut_Single)*10+STRING_TO_BYTE(ASCII_Chart_N_Alarm[2].sOut_Single);
							5:
								ASCII_Chart_N_Alarm[3](byASCII:=sRecvByte[2] , sOut_Single=> );
								ASCII_Chart_N_Alarm[4](byASCII:=sRecvByte[3] , sOut_Single=> );
								ASCII_Chart_N_Alarm[5](byASCII:=sRecvByte[4] , sOut_Single=> );
								iAlarmNum:=STRING_TO_BYTE(ASCII_Chart_N_Alarm[3].sOut_Single)*100+STRING_TO_BYTE(ASCII_Chart_N_Alarm[4].sOut_Single)*10+STRING_TO_BYTE(ASCII_Chart_N_Alarm[5].sOut_Single);
							ELSE
								iAlarmNum:=iAlarmNum;
						END_CASE
						TON40(IN:=FALSE);
					ELSE
						TON40(IN:=TRUE , PT:= T#2S, Q=> , ET=> );
						IF TON40.Q THEN
							Main_Step	:=20;
						END_IF;
					END_IF
				END_CASE
				
			IF 	Entity_IO.bXrayBuckey THEN
				hlaldjlk:=TRUE;
			END_IF
END_ACTION

END_PROGRAM

// Device/Application/BasicFBs/String2Byte
FUNCTION_BLOCK String2Byte
VAR_INPUT
	 sXrayString:STRING;
END_VAR
VAR_OUTPUT
	 sByte	:ARRAY[0..9] OF BYTE;
END_VAR
VAR
	iSize	:INT;
	k		:INT:=1;
	s1		:STRING;
	sString	:ARRAY[0..9] OF STRING;
	ASCII_Chart1:ASCII_Chart_P;
END_VAR



	iSize:=LIMIT(0,LEN(sXrayString),10); //获取字符串长度
	
	(*获取每个字符，并放入字符序列中*)
	FOR k:=0 TO iSize BY 1 DO 
		s1:=MID(STR:= sXrayString, LEN:=1 , POS:=k );
		sString[k]:=s1;
		ASCII_Chart1(sASCII_IN:=s1 , byASCII=>sByte[k] );
	END_FOR

END_FUNCTION_BLOCK

// Device/Application/BasicFBs/ASCII_Chart_P
FUNCTION_BLOCK ASCII_Chart_P
VAR_INPUT
	sASCII_IN:STRING;
END_VAR
VAR_OUTPUT
	byASCII:BYTE;
END_VAR
VAR
	sIn_Single:STRING;
END_VAR

(*字符转换为16进制数字，BYTE数据类型*)

	sIn_Single:=LEFT(STR:=sASCII_IN , SIZE:=1 );//保证就一个字符
	
	IF    sIn_Single='A' THEN 	byASCII:=16#41;
	ELSIF sIn_Single='B' THEN  	byASCII:=16#42;
	ELSIF sIn_Single='C' THEN  	byASCII:=16#43;
	ELSIF sIn_Single='D' THEN	byASCII:=16#44;
	ELSIF sIn_Single='E' THEN	byASCII:=16#45;
	ELSIF sIn_Single='F' THEN	byASCII:=16#46;
	ELSIF sIn_Single='G' THEN	byASCII:=16#47;
	ELSIF sIn_Single='H' THEN	byASCII:=16#48;
	ELSIF sIn_Single='I' THEN	byASCII:=16#49;
	ELSIF sIn_Single='J' THEN	byASCII:=16#4A;
	ELSIF sIn_Single='K' THEN	byASCII:=16#4B;
	ELSIF sIn_Single='L' THEN	byASCII:=16#4C;
	ELSIF sIn_Single='M' THEN	byASCII:=16#4D;
	ELSIF sIn_Single='N' THEN	byASCII:=16#4E;
	ELSIF sIn_Single='O' THEN	byASCII:=16#4F;
	ELSIF sIn_Single='P' THEN	byASCII:=16#50;
	ELSIF sIn_Single='Q' THEN	byASCII:=16#51;
	ELSIF sIn_Single='R' THEN	byASCII:=16#52;
	ELSIF sIn_Single='S' THEN	byASCII:=16#53;
	ELSIF sIn_Single='T' THEN	byASCII:=16#54;
	ELSIF sIn_Single='U' THEN	byASCII:=16#55;
	ELSIF sIn_Single='V' THEN	byASCII:=16#56;
	ELSIF sIn_Single='W' THEN	byASCII:=16#57;
	ELSIF sIn_Single='X' THEN	byASCII:=16#58;
	ELSIF sIn_Single='Y' THEN	byASCII:=16#59;
	ELSIF sIn_Single='Z' THEN	byASCII:=16#5A;
	ELSIF sIn_Single='[' THEN	byASCII:=16#5B;
	ELSIF sIn_Single='\' THEN	byASCII:=16#5C;
	ELSIF sIn_Single=']' THEN	byASCII:=16#5D;
	ELSIF sIn_Single='^' THEN	byASCII:=16#5E;
	ELSIF sIn_Single='_' THEN	byASCII:=16#5F;
	ELSIF sIn_Single='`' THEN	byASCII:=16#60;
	
	ELSIF sIn_Single='a' THEN	byASCII:=16#61;	
	ELSIF sIn_Single='b' THEN  	byASCII:=16#62;
	ELSIF sIn_Single='c' THEN  	byASCII:=16#63;
	ELSIF sIn_Single='d' THEN	byASCII:=16#64;
	ELSIF sIn_Single='e' THEN	byASCII:=16#65;
	ELSIF sIn_Single='f' THEN	byASCII:=16#66;
	ELSIF sIn_Single='g' THEN	byASCII:=16#67;
	ELSIF sIn_Single='h' THEN	byASCII:=16#68;
	ELSIF sIn_Single='i' THEN	byASCII:=16#69;
	ELSIF sIn_Single='j' THEN	byASCII:=16#6A;
	ELSIF sIn_Single='k' THEN	byASCII:=16#6B;
	ELSIF sIn_Single='l' THEN	byASCII:=16#6C;
	ELSIF sIn_Single='m' THEN	byASCII:=16#6D;
	ELSIF sIn_Single='n' THEN	byASCII:=16#6E;
	ELSIF sIn_Single='o' THEN	byASCII:=16#6F;
	ELSIF sIn_Single='p' THEN	byASCII:=16#70;
	ELSIF sIn_Single='q' THEN	byASCII:=16#71;
	ELSIF sIn_Single='r' THEN	byASCII:=16#72;
	ELSIF sIn_Single='s' THEN	byASCII:=16#73;
	ELSIF sIn_Single='t' THEN	byASCII:=16#74;
	ELSIF sIn_Single='u' THEN	byASCII:=16#75;
	ELSIF sIn_Single='v' THEN	byASCII:=16#76;
	ELSIF sIn_Single='w' THEN	byASCII:=16#77;
	ELSIF sIn_Single='x' THEN	byASCII:=16#78;
	ELSIF sIn_Single='y' THEN	byASCII:=16#79;
	ELSIF sIn_Single='z' THEN	byASCII:=16#7A;
	ELSIF sIn_Single='{' THEN	byASCII:=16#7B;
	ELSIF sIn_Single='|' THEN	byASCII:=16#7C;
	ELSIF sIn_Single='}' THEN	byASCII:=16#7D;
	
	ELSIF sIn_Single='0' THEN  	byASCII:=16#30;
	ELSIF sIn_Single='1' THEN  	byASCII:=16#31;
	ELSIF sIn_Single='2' THEN	byASCII:=16#32;
	ELSIF sIn_Single='3' THEN	byASCII:=16#33;
	ELSIF sIn_Single='4' THEN	byASCII:=16#34;
	ELSIF sIn_Single='5' THEN	byASCII:=16#35;
	ELSIF sIn_Single='6' THEN	byASCII:=16#36;
	ELSIF sIn_Single='7' THEN	byASCII:=16#37;
	ELSIF sIn_Single='8' THEN	byASCII:=16#38;
	ELSIF sIn_Single='9' THEN	byASCII:=16#39;
	ELSIF sIn_Single=':' THEN	byASCII:=16#3A;
	ELSIF sIn_Single=';' THEN	byASCII:=16#3B;
	ELSIF sIn_Single='<' THEN	byASCII:=16#3C;
	ELSIF sIn_Single='=' THEN	byASCII:=16#3D;
	ELSIF sIn_Single='>' THEN	byASCII:=16#3E;
	ELSIF sIn_Single='?' THEN	byASCII:=16#3F;
	ELSIF sIn_Single='@' THEN	byASCII:=16#40;
		
	ELSIF sIn_Single='!' THEN	byASCII:=16#21;
	ELSIF sIn_Single='"' THEN	byASCII:=16#22;
	ELSIF sIn_Single='#' THEN	byASCII:=16#23;
//	ELSIF sIn_Single='$' THEN	byASCII:=16#24;
	ELSIF sIn_Single='%' THEN	byASCII:=16#25;
	ELSIF sIn_Single='&' THEN	byASCII:=16#26;
//	ELSIF sIn_Single=''' THEN	byASCII:=16#27;
	ELSIF sIn_Single='(' THEN	byASCII:=16#28;
	ELSIF sIn_Single=')' THEN	byASCII:=16#29;
	ELSIF sIn_Single='*' THEN	byASCII:=16#2A;
	ELSIF sIn_Single='+' THEN	byASCII:=16#2B;
	ELSIF sIn_Single=',' THEN	byASCII:=16#2C;
	ELSIF sIn_Single='-' THEN	byASCII:=16#2D;
	ELSIF sIn_Single='.' THEN	byASCII:=16#2E;
	ELSIF sIn_Single='/' THEN	byASCII:=16#2F;
	ELSE
		byASCII:=16#FF;	 //错误标志
	END_IF

END_FUNCTION_BLOCK

// Device/Application/BasicFBs/ASCII_Chart_N
FUNCTION_BLOCK ASCII_Chart_N
VAR_INPUT
	byASCII		:BYTE;
END_VAR
VAR_OUTPUT
	sOut_Single	:STRING;
END_VAR
VAR
	
END_VAR

(*ASCII码转化为字符*)
	
	IF    byASCII=16#41 THEN 	sOut_Single:='A';
	ELSIF byASCII=16#42 THEN  	sOut_Single:='B';
	ELSIF byASCII=16#43 THEN  	sOut_Single:='C';
	ELSIF byASCII=16#44 THEN	sOut_Single:='D';
	ELSIF byASCII=16#45 THEN	sOut_Single:='E';
	ELSIF byASCII=16#46 THEN	sOut_Single:='F';
	ELSIF byASCII=16#47 THEN	sOut_Single:='G';
	ELSIF byASCII=16#48 THEN	sOut_Single:='H';
	ELSIF byASCII=16#49 THEN	sOut_Single:='I';
	ELSIF byASCII=16#4A THEN	sOut_Single:='J';
	ELSIF byASCII=16#4B THEN	sOut_Single:='K';
	ELSIF byASCII=16#4C THEN	sOut_Single:='L';
	ELSIF byASCII=16#4D THEN	sOut_Single:='M';
	ELSIF byASCII=16#4E THEN	sOut_Single:='N';
	ELSIF byASCII=16#4F THEN	sOut_Single:='O';
	ELSIF byASCII=16#50 THEN	sOut_Single:='P';
	ELSIF byASCII=16#51 THEN	sOut_Single:='Q';
	ELSIF byASCII=16#52 THEN	sOut_Single:='R';
	ELSIF byASCII=16#53 THEN	sOut_Single:='S';
	ELSIF byASCII=16#54 THEN	sOut_Single:='T';
	ELSIF byASCII=16#55 THEN	sOut_Single:='U';
	ELSIF byASCII=16#56 THEN	sOut_Single:='V';
	ELSIF byASCII=16#57 THEN	sOut_Single:='W';
	ELSIF byASCII=16#58 THEN	sOut_Single:='X';
	ELSIF byASCII=16#59 THEN	sOut_Single:='Y';
	ELSIF byASCII=16#5A THEN	sOut_Single:='Z';
	ELSIF byASCII=16#5B THEN	sOut_Single:='[';
	ELSIF byASCII=16#5C THEN	sOut_Single:='\';
	ELSIF byASCII=16#5D THEN	sOut_Single:=']';
	ELSIF byASCII=16#5E THEN	sOut_Single:='^';
	ELSIF byASCII=16#5F THEN	sOut_Single:='_';
	ELSIF byASCII=16#60 THEN	sOut_Single:='`';
	                                         
